// TIA Portal V17 export
// export: Created 2025-07-01T09:59:02.8263122Z, ExportSetting WithDefaults, DisplayName Totally Integrated Automation Portal, DisplayVersion V17 Update 8, DisplayName TIA Portal Openness, DisplayVersion V17 Update 8, DisplayName TIA Portal Version Control Interface, DisplayVersion V17, DisplayName SINAMICS Startdrive Advanced, DisplayVersion V17 SP2, DisplayName SINAMICS Startdrive G110M, G120, G120C, G120D, G120P, G115D, DisplayVersion V17 SP2, DisplayName SINAMICS Startdrive G130, G150, S120, S150, SINAMICS MV, S210, DisplayVersion V17 SP2, DisplayName STEP 7 Professional, DisplayVersion V17 Update 8, DisplayName SINUMERIK ONE STEP 7 Toolbox, DisplayVersion V17 Update 12, DisplayName SINUMERIK ONE PLC Basic Program Plus, DisplayVersion V17 Update 12, DisplayName SINUMERIK 840D sl STEP 7 Toolbox, DisplayVersion V17 Update 12, DisplayName STEP 7 Safety, DisplayVersion V17 Update 6, DisplayName WinCC Advanced, DisplayVersion V17 Update 8
FUNCTION "FC16012_METHOD_CALLS_U1_STA3_COAXIAL" : Void   // FC16012, LAD
{ S7_Optimized_Access := 'FALSE' }
VERSION : 0.1
// PC status values:
// 0-> Idle
// 1-> LaserCalibrating
// 2-> NozzleCalibrating
// 3-> JetCalibrating
// 4-> CladdingCalibrating
// 5-> NozzleAnalysis
// 6-> JetAnalysis
// 7-> CladdingAnalysis
// -1-> Error
// stored: AutoNumber false, IsIECCheckEnabled false, SetENOAutomatically false, UDAEnableTagReadback false
   VAR_TEMP
      AUX_WSTRING_PART_ID_STA3 : WString;
      AUX_WCHARS : Array[0..63] of WChar;
      index : Int;
      ALARM_AUX : Bool;
      STATUS_BLKMOV : Int;   // STATUS BLKMOV
      ZERO : Int;
      retval : Word;
   END_VAR
   VAR CONSTANT
      VERSIONS_MAJOR : UInt := 2;
      VERSIONS_MINOR : UInt := 0;
      FC_NUMBER : DInt := 16012;
   END_VAR
   VAR_TEMP   // added for the SCL form of the ladder/FBD networks
      _w1 : Bool;
      _w2 : Bool;
   END_VAR
BEGIN

REGION Network 1 (SCL): TRANSFORM TO WCHARS
   FOR #index := 0 TO 63 DO
       #AUX_WCHARS[#index] := CHAR_TO_WCHAR("DB8000_PART_STATUS".UNIT_1.STATION_3.PART_A.PART_ID[#index]);
   END_FOR;
END_REGION

REGION Network 2: TRANSFORM TO WSTRING
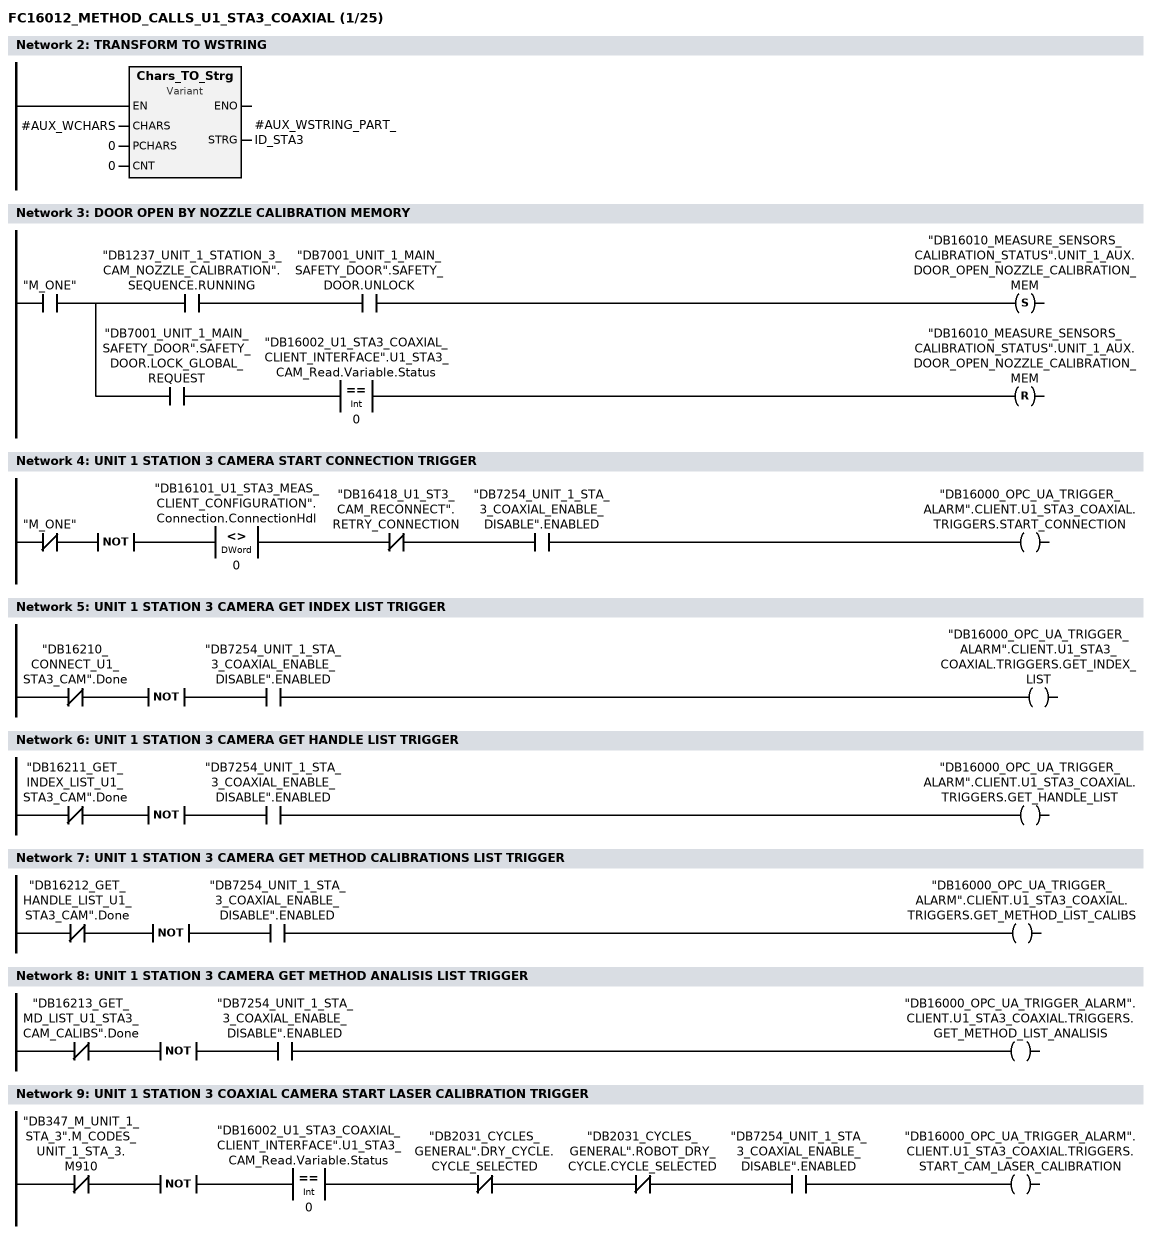
   RUNG wire#powerrail
      { S7_Templates := "[ptr_type := Variant, str_type := WString]" } Chars_TO_Strg(Chars := #AUX_WCHARS, pChars := 0, Cnt := 0, Strg => #AUX_WSTRING_PART_ID_STA3)
   END_RUNG
   // the same network as SCL:
   Chars_TO_Strg(Chars := #AUX_WCHARS, pChars := 0, Cnt := 0, Strg => #AUX_WSTRING_PART_ID_STA3);
END_REGION

REGION Network 3: DOOR OPEN BY NOZZLE CALIBRATION MEMORY
   RUNG wire#powerrail
      Contact( "M_ONE" )
      wire#w1
      Contact( "DB1237_UNIT_1_STATION_3_CAM_NOZZLE_CALIBRATION".SEQUENCE.RUNNING )
      Contact( "DB7001_UNIT_1_MAIN_SAFETY_DOOR".SAFETY_DOOR.UNLOCK )
      S_Coil( "DB16010_MEASURE_SENSORS_CALIBRATION_STATUS".UNIT_1_AUX.DOOR_OPEN_NOZZLE_CALIBRATION_MEM )
   END_RUNG
   RUNG wire#w1
      Contact( "DB7001_UNIT_1_MAIN_SAFETY_DOOR".SAFETY_DOOR.LOCK_GLOBAL_REQUEST )
      { S7_Templates := "SrcType := Int" } EQ_Contact(in1 := "DB16002_U1_STA3_COAXIAL_CLIENT_INTERFACE".U1_STA3_CAM_Read.Variable.Status, in2 := 0)
      R_Coil( "DB16010_MEASURE_SENSORS_CALIBRATION_STATUS".UNIT_1_AUX.DOOR_OPEN_NOZZLE_CALIBRATION_MEM )
   END_RUNG
   // the same network as SCL:
   IF "M_ONE" AND "DB1237_UNIT_1_STATION_3_CAM_NOZZLE_CALIBRATION".SEQUENCE.RUNNING AND "DB7001_UNIT_1_MAIN_SAFETY_DOOR".SAFETY_DOOR.UNLOCK THEN
       "DB16010_MEASURE_SENSORS_CALIBRATION_STATUS".UNIT_1_AUX.DOOR_OPEN_NOZZLE_CALIBRATION_MEM := TRUE;
   END_IF;
   IF "M_ONE" AND "DB7001_UNIT_1_MAIN_SAFETY_DOOR".SAFETY_DOOR.LOCK_GLOBAL_REQUEST AND ("DB16002_U1_STA3_COAXIAL_CLIENT_INTERFACE".U1_STA3_CAM_Read.Variable.Status = 0) THEN
       "DB16010_MEASURE_SENSORS_CALIBRATION_STATUS".UNIT_1_AUX.DOOR_OPEN_NOZZLE_CALIBRATION_MEM := FALSE;
   END_IF;
END_REGION

REGION Network 4: UNIT 1 STATION 3 CAMERA START CONNECTION TRIGGER
   RUNG wire#powerrail
      I_Contact( "M_ONE" )
      Not()
      { S7_Templates := "SrcType := DWord" } NE_Contact(in1 := "DB16101_U1_STA3_MEAS_CLIENT_CONFIGURATION".Connection.ConnectionHdl, in2 := 0)
      I_Contact( "DB16418_U1_ST3_CAM_RECONNECT".RETRY_CONNECTION )
      Contact( "DB7254_UNIT_1_STA_3_COAXIAL_ENABLE_DISABLE".ENABLED )
      Coil( "DB16000_OPC_UA_TRIGGER_ALARM".CLIENT.U1_STA3_COAXIAL.TRIGGERS.START_CONNECTION )
   END_RUNG
   // the same network as SCL:
   "DB16000_OPC_UA_TRIGGER_ALARM".CLIENT.U1_STA3_COAXIAL.TRIGGERS.START_CONNECTION := NOT (NOT "M_ONE") AND ("DB16101_U1_STA3_MEAS_CLIENT_CONFIGURATION".Connection.ConnectionHdl <> 0) AND NOT "DB16418_U1_ST3_CAM_RECONNECT".RETRY_CONNECTION AND "DB7254_UNIT_1_STA_3_COAXIAL_ENABLE_DISABLE".ENABLED;
END_REGION

REGION Network 5: UNIT 1 STATION 3 CAMERA GET INDEX LIST TRIGGER
   RUNG wire#powerrail
      I_Contact( "DB16210_CONNECT_U1_STA3_CAM".Done )
      Not()
      Contact( "DB7254_UNIT_1_STA_3_COAXIAL_ENABLE_DISABLE".ENABLED )
      Coil( "DB16000_OPC_UA_TRIGGER_ALARM".CLIENT.U1_STA3_COAXIAL.TRIGGERS.GET_INDEX_LIST )
   END_RUNG
   // the same network as SCL:
   "DB16000_OPC_UA_TRIGGER_ALARM".CLIENT.U1_STA3_COAXIAL.TRIGGERS.GET_INDEX_LIST := NOT (NOT "DB16210_CONNECT_U1_STA3_CAM".Done) AND "DB7254_UNIT_1_STA_3_COAXIAL_ENABLE_DISABLE".ENABLED;
END_REGION

REGION Network 6: UNIT 1 STATION 3 CAMERA GET HANDLE LIST TRIGGER
   RUNG wire#powerrail
      I_Contact( "DB16211_GET_INDEX_LIST_U1_STA3_CAM".Done )
      Not()
      Contact( "DB7254_UNIT_1_STA_3_COAXIAL_ENABLE_DISABLE".ENABLED )
      Coil( "DB16000_OPC_UA_TRIGGER_ALARM".CLIENT.U1_STA3_COAXIAL.TRIGGERS.GET_HANDLE_LIST )
   END_RUNG
   // the same network as SCL:
   "DB16000_OPC_UA_TRIGGER_ALARM".CLIENT.U1_STA3_COAXIAL.TRIGGERS.GET_HANDLE_LIST := NOT (NOT "DB16211_GET_INDEX_LIST_U1_STA3_CAM".Done) AND "DB7254_UNIT_1_STA_3_COAXIAL_ENABLE_DISABLE".ENABLED;
END_REGION

REGION Network 7: UNIT 1 STATION 3 CAMERA GET METHOD CALIBRATIONS LIST TRIGGER
   RUNG wire#powerrail
      I_Contact( "DB16212_GET_HANDLE_LIST_U1_STA3_CAM".Done )
      Not()
      Contact( "DB7254_UNIT_1_STA_3_COAXIAL_ENABLE_DISABLE".ENABLED )
      Coil( "DB16000_OPC_UA_TRIGGER_ALARM".CLIENT.U1_STA3_COAXIAL.TRIGGERS.GET_METHOD_LIST_CALIBS )
   END_RUNG
   // the same network as SCL:
   "DB16000_OPC_UA_TRIGGER_ALARM".CLIENT.U1_STA3_COAXIAL.TRIGGERS.GET_METHOD_LIST_CALIBS := NOT (NOT "DB16212_GET_HANDLE_LIST_U1_STA3_CAM".Done) AND "DB7254_UNIT_1_STA_3_COAXIAL_ENABLE_DISABLE".ENABLED;
END_REGION

REGION Network 8: UNIT 1 STATION 3 CAMERA GET METHOD ANALISIS LIST TRIGGER
   RUNG wire#powerrail
      I_Contact( "DB16213_GET_MD_LIST_U1_STA3_CAM_CALIBS".Done )
      Not()
      Contact( "DB7254_UNIT_1_STA_3_COAXIAL_ENABLE_DISABLE".ENABLED )
      Coil( "DB16000_OPC_UA_TRIGGER_ALARM".CLIENT.U1_STA3_COAXIAL.TRIGGERS.GET_METHOD_LIST_ANALISIS )
   END_RUNG
   // the same network as SCL:
   "DB16000_OPC_UA_TRIGGER_ALARM".CLIENT.U1_STA3_COAXIAL.TRIGGERS.GET_METHOD_LIST_ANALISIS := NOT (NOT "DB16213_GET_MD_LIST_U1_STA3_CAM_CALIBS".Done) AND "DB7254_UNIT_1_STA_3_COAXIAL_ENABLE_DISABLE".ENABLED;
END_REGION

REGION Network 9: UNIT 1 STATION 3 COAXIAL CAMERA START LASER CALIBRATION TRIGGER
   RUNG wire#powerrail
      I_Contact( "DB347_M_UNIT_1_STA_3".M_CODES_UNIT_1_STA_3.M910 )
      Not()
      { S7_Templates := "SrcType := Int" } EQ_Contact(in1 := "DB16002_U1_STA3_COAXIAL_CLIENT_INTERFACE".U1_STA3_CAM_Read.Variable.Status, in2 := 0)
      I_Contact( "DB2031_CYCLES_GENERAL".DRY_CYCLE.CYCLE_SELECTED )
      I_Contact( "DB2031_CYCLES_GENERAL".ROBOT_DRY_CYCLE.CYCLE_SELECTED )
      Contact( "DB7254_UNIT_1_STA_3_COAXIAL_ENABLE_DISABLE".ENABLED )
      Coil( "DB16000_OPC_UA_TRIGGER_ALARM".CLIENT.U1_STA3_COAXIAL.TRIGGERS.START_CAM_LASER_CALIBRATION )
   END_RUNG
   // the same network as SCL:
   "DB16000_OPC_UA_TRIGGER_ALARM".CLIENT.U1_STA3_COAXIAL.TRIGGERS.START_CAM_LASER_CALIBRATION := NOT (NOT "DB347_M_UNIT_1_STA_3".M_CODES_UNIT_1_STA_3.M910) AND ("DB16002_U1_STA3_COAXIAL_CLIENT_INTERFACE".U1_STA3_CAM_Read.Variable.Status = 0) AND NOT "DB2031_CYCLES_GENERAL".DRY_CYCLE.CYCLE_SELECTED AND NOT "DB2031_CYCLES_GENERAL".ROBOT_DRY_CYCLE.CYCLE_SELECTED AND "DB7254_UNIT_1_STA_3_COAXIAL_ENABLE_DISABLE".ENABLED;
END_REGION

REGION Network 10: UNIT 1 STATION 3 COAXIAL CAMERA START NOZZLE CALIBRATION TRIGGER
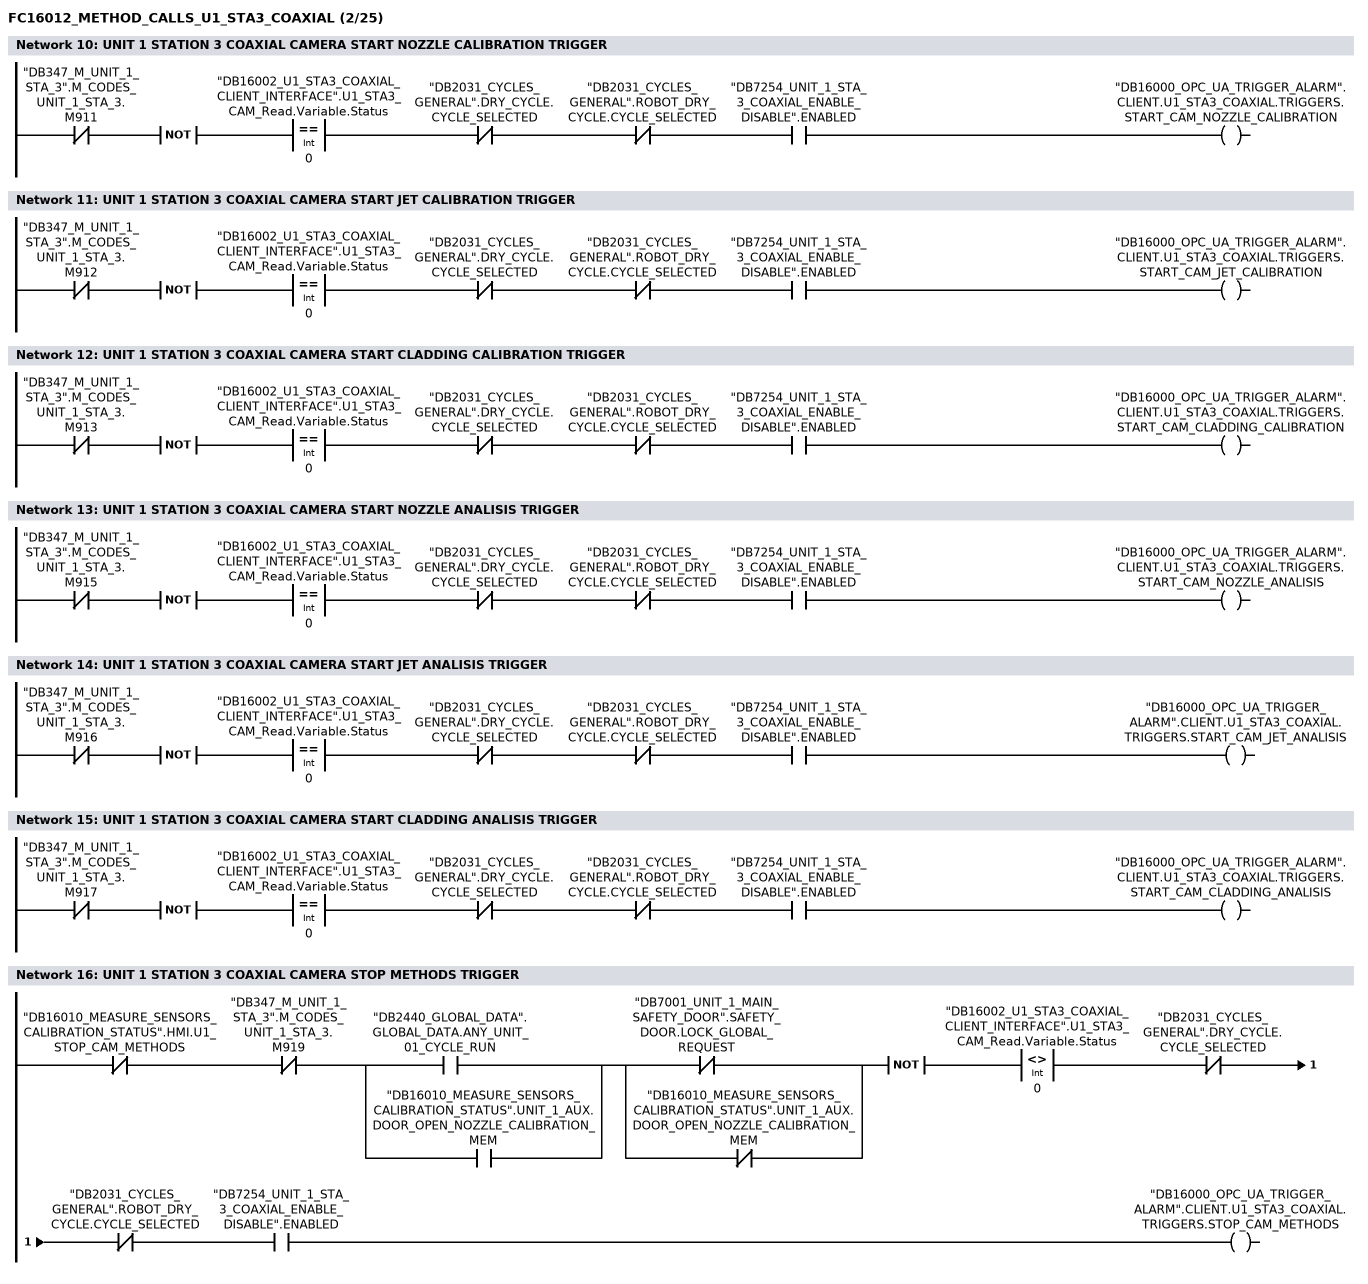
   RUNG wire#powerrail
      I_Contact( "DB347_M_UNIT_1_STA_3".M_CODES_UNIT_1_STA_3.M911 )
      Not()
      { S7_Templates := "SrcType := Int" } EQ_Contact(in1 := "DB16002_U1_STA3_COAXIAL_CLIENT_INTERFACE".U1_STA3_CAM_Read.Variable.Status, in2 := 0)
      I_Contact( "DB2031_CYCLES_GENERAL".DRY_CYCLE.CYCLE_SELECTED )
      I_Contact( "DB2031_CYCLES_GENERAL".ROBOT_DRY_CYCLE.CYCLE_SELECTED )
      Contact( "DB7254_UNIT_1_STA_3_COAXIAL_ENABLE_DISABLE".ENABLED )
      Coil( "DB16000_OPC_UA_TRIGGER_ALARM".CLIENT.U1_STA3_COAXIAL.TRIGGERS.START_CAM_NOZZLE_CALIBRATION )
   END_RUNG
   // the same network as SCL:
   "DB16000_OPC_UA_TRIGGER_ALARM".CLIENT.U1_STA3_COAXIAL.TRIGGERS.START_CAM_NOZZLE_CALIBRATION := NOT (NOT "DB347_M_UNIT_1_STA_3".M_CODES_UNIT_1_STA_3.M911) AND ("DB16002_U1_STA3_COAXIAL_CLIENT_INTERFACE".U1_STA3_CAM_Read.Variable.Status = 0) AND NOT "DB2031_CYCLES_GENERAL".DRY_CYCLE.CYCLE_SELECTED AND NOT "DB2031_CYCLES_GENERAL".ROBOT_DRY_CYCLE.CYCLE_SELECTED AND "DB7254_UNIT_1_STA_3_COAXIAL_ENABLE_DISABLE".ENABLED;
END_REGION

REGION Network 11: UNIT 1 STATION 3 COAXIAL CAMERA START JET CALIBRATION TRIGGER
   RUNG wire#powerrail
      I_Contact( "DB347_M_UNIT_1_STA_3".M_CODES_UNIT_1_STA_3.M912 )
      Not()
      { S7_Templates := "SrcType := Int" } EQ_Contact(in1 := "DB16002_U1_STA3_COAXIAL_CLIENT_INTERFACE".U1_STA3_CAM_Read.Variable.Status, in2 := 0)
      I_Contact( "DB2031_CYCLES_GENERAL".DRY_CYCLE.CYCLE_SELECTED )
      I_Contact( "DB2031_CYCLES_GENERAL".ROBOT_DRY_CYCLE.CYCLE_SELECTED )
      Contact( "DB7254_UNIT_1_STA_3_COAXIAL_ENABLE_DISABLE".ENABLED )
      Coil( "DB16000_OPC_UA_TRIGGER_ALARM".CLIENT.U1_STA3_COAXIAL.TRIGGERS.START_CAM_JET_CALIBRATION )
   END_RUNG
   // the same network as SCL:
   "DB16000_OPC_UA_TRIGGER_ALARM".CLIENT.U1_STA3_COAXIAL.TRIGGERS.START_CAM_JET_CALIBRATION := NOT (NOT "DB347_M_UNIT_1_STA_3".M_CODES_UNIT_1_STA_3.M912) AND ("DB16002_U1_STA3_COAXIAL_CLIENT_INTERFACE".U1_STA3_CAM_Read.Variable.Status = 0) AND NOT "DB2031_CYCLES_GENERAL".DRY_CYCLE.CYCLE_SELECTED AND NOT "DB2031_CYCLES_GENERAL".ROBOT_DRY_CYCLE.CYCLE_SELECTED AND "DB7254_UNIT_1_STA_3_COAXIAL_ENABLE_DISABLE".ENABLED;
END_REGION

REGION Network 12: UNIT 1 STATION 3 COAXIAL CAMERA START CLADDING CALIBRATION TRIGGER
   RUNG wire#powerrail
      I_Contact( "DB347_M_UNIT_1_STA_3".M_CODES_UNIT_1_STA_3.M913 )
      Not()
      { S7_Templates := "SrcType := Int" } EQ_Contact(in1 := "DB16002_U1_STA3_COAXIAL_CLIENT_INTERFACE".U1_STA3_CAM_Read.Variable.Status, in2 := 0)
      I_Contact( "DB2031_CYCLES_GENERAL".DRY_CYCLE.CYCLE_SELECTED )
      I_Contact( "DB2031_CYCLES_GENERAL".ROBOT_DRY_CYCLE.CYCLE_SELECTED )
      Contact( "DB7254_UNIT_1_STA_3_COAXIAL_ENABLE_DISABLE".ENABLED )
      Coil( "DB16000_OPC_UA_TRIGGER_ALARM".CLIENT.U1_STA3_COAXIAL.TRIGGERS.START_CAM_CLADDING_CALIBRATION )
   END_RUNG
   // the same network as SCL:
   "DB16000_OPC_UA_TRIGGER_ALARM".CLIENT.U1_STA3_COAXIAL.TRIGGERS.START_CAM_CLADDING_CALIBRATION := NOT (NOT "DB347_M_UNIT_1_STA_3".M_CODES_UNIT_1_STA_3.M913) AND ("DB16002_U1_STA3_COAXIAL_CLIENT_INTERFACE".U1_STA3_CAM_Read.Variable.Status = 0) AND NOT "DB2031_CYCLES_GENERAL".DRY_CYCLE.CYCLE_SELECTED AND NOT "DB2031_CYCLES_GENERAL".ROBOT_DRY_CYCLE.CYCLE_SELECTED AND "DB7254_UNIT_1_STA_3_COAXIAL_ENABLE_DISABLE".ENABLED;
END_REGION

REGION Network 13: UNIT 1 STATION 3 COAXIAL CAMERA START NOZZLE ANALISIS TRIGGER
   RUNG wire#powerrail
      I_Contact( "DB347_M_UNIT_1_STA_3".M_CODES_UNIT_1_STA_3.M915 )
      Not()
      { S7_Templates := "SrcType := Int" } EQ_Contact(in1 := "DB16002_U1_STA3_COAXIAL_CLIENT_INTERFACE".U1_STA3_CAM_Read.Variable.Status, in2 := 0)
      I_Contact( "DB2031_CYCLES_GENERAL".DRY_CYCLE.CYCLE_SELECTED )
      I_Contact( "DB2031_CYCLES_GENERAL".ROBOT_DRY_CYCLE.CYCLE_SELECTED )
      Contact( "DB7254_UNIT_1_STA_3_COAXIAL_ENABLE_DISABLE".ENABLED )
      Coil( "DB16000_OPC_UA_TRIGGER_ALARM".CLIENT.U1_STA3_COAXIAL.TRIGGERS.START_CAM_NOZZLE_ANALISIS )
   END_RUNG
   // the same network as SCL:
   "DB16000_OPC_UA_TRIGGER_ALARM".CLIENT.U1_STA3_COAXIAL.TRIGGERS.START_CAM_NOZZLE_ANALISIS := NOT (NOT "DB347_M_UNIT_1_STA_3".M_CODES_UNIT_1_STA_3.M915) AND ("DB16002_U1_STA3_COAXIAL_CLIENT_INTERFACE".U1_STA3_CAM_Read.Variable.Status = 0) AND NOT "DB2031_CYCLES_GENERAL".DRY_CYCLE.CYCLE_SELECTED AND NOT "DB2031_CYCLES_GENERAL".ROBOT_DRY_CYCLE.CYCLE_SELECTED AND "DB7254_UNIT_1_STA_3_COAXIAL_ENABLE_DISABLE".ENABLED;
END_REGION

REGION Network 14: UNIT 1 STATION 3 COAXIAL CAMERA START JET ANALISIS TRIGGER
   RUNG wire#powerrail
      I_Contact( "DB347_M_UNIT_1_STA_3".M_CODES_UNIT_1_STA_3.M916 )
      Not()
      { S7_Templates := "SrcType := Int" } EQ_Contact(in1 := "DB16002_U1_STA3_COAXIAL_CLIENT_INTERFACE".U1_STA3_CAM_Read.Variable.Status, in2 := 0)
      I_Contact( "DB2031_CYCLES_GENERAL".DRY_CYCLE.CYCLE_SELECTED )
      I_Contact( "DB2031_CYCLES_GENERAL".ROBOT_DRY_CYCLE.CYCLE_SELECTED )
      Contact( "DB7254_UNIT_1_STA_3_COAXIAL_ENABLE_DISABLE".ENABLED )
      Coil( "DB16000_OPC_UA_TRIGGER_ALARM".CLIENT.U1_STA3_COAXIAL.TRIGGERS.START_CAM_JET_ANALISIS )
   END_RUNG
   // the same network as SCL:
   "DB16000_OPC_UA_TRIGGER_ALARM".CLIENT.U1_STA3_COAXIAL.TRIGGERS.START_CAM_JET_ANALISIS := NOT (NOT "DB347_M_UNIT_1_STA_3".M_CODES_UNIT_1_STA_3.M916) AND ("DB16002_U1_STA3_COAXIAL_CLIENT_INTERFACE".U1_STA3_CAM_Read.Variable.Status = 0) AND NOT "DB2031_CYCLES_GENERAL".DRY_CYCLE.CYCLE_SELECTED AND NOT "DB2031_CYCLES_GENERAL".ROBOT_DRY_CYCLE.CYCLE_SELECTED AND "DB7254_UNIT_1_STA_3_COAXIAL_ENABLE_DISABLE".ENABLED;
END_REGION

REGION Network 15: UNIT 1 STATION 3 COAXIAL CAMERA START CLADDING ANALISIS TRIGGER
   RUNG wire#powerrail
      I_Contact( "DB347_M_UNIT_1_STA_3".M_CODES_UNIT_1_STA_3.M917 )
      Not()
      { S7_Templates := "SrcType := Int" } EQ_Contact(in1 := "DB16002_U1_STA3_COAXIAL_CLIENT_INTERFACE".U1_STA3_CAM_Read.Variable.Status, in2 := 0)
      I_Contact( "DB2031_CYCLES_GENERAL".DRY_CYCLE.CYCLE_SELECTED )
      I_Contact( "DB2031_CYCLES_GENERAL".ROBOT_DRY_CYCLE.CYCLE_SELECTED )
      Contact( "DB7254_UNIT_1_STA_3_COAXIAL_ENABLE_DISABLE".ENABLED )
      Coil( "DB16000_OPC_UA_TRIGGER_ALARM".CLIENT.U1_STA3_COAXIAL.TRIGGERS.START_CAM_CLADDING_ANALISIS )
   END_RUNG
   // the same network as SCL:
   "DB16000_OPC_UA_TRIGGER_ALARM".CLIENT.U1_STA3_COAXIAL.TRIGGERS.START_CAM_CLADDING_ANALISIS := NOT (NOT "DB347_M_UNIT_1_STA_3".M_CODES_UNIT_1_STA_3.M917) AND ("DB16002_U1_STA3_COAXIAL_CLIENT_INTERFACE".U1_STA3_CAM_Read.Variable.Status = 0) AND NOT "DB2031_CYCLES_GENERAL".DRY_CYCLE.CYCLE_SELECTED AND NOT "DB2031_CYCLES_GENERAL".ROBOT_DRY_CYCLE.CYCLE_SELECTED AND "DB7254_UNIT_1_STA_3_COAXIAL_ENABLE_DISABLE".ENABLED;
END_REGION

REGION Network 16: UNIT 1 STATION 3 COAXIAL CAMERA STOP METHODS TRIGGER
   RUNG wire#powerrail
      I_Contact( "DB16010_MEASURE_SENSORS_CALIBRATION_STATUS".HMI.U1_STOP_CAM_METHODS )
      I_Contact( "DB347_M_UNIT_1_STA_3".M_CODES_UNIT_1_STA_3.M919 )
      wire#w1
      Contact( "DB2440_GLOBAL_DATA".GLOBAL_DATA.ANY_UNIT_01_CYCLE_RUN )
      wire#w2
      I_Contact( "DB7001_UNIT_1_MAIN_SAFETY_DOOR".SAFETY_DOOR.LOCK_GLOBAL_REQUEST )
      wire#w3
      Not()
      { S7_Templates := "SrcType := Int" } NE_Contact(in1 := "DB16002_U1_STA3_COAXIAL_CLIENT_INTERFACE".U1_STA3_CAM_Read.Variable.Status, in2 := 0)
      I_Contact( "DB2031_CYCLES_GENERAL".DRY_CYCLE.CYCLE_SELECTED )
      I_Contact( "DB2031_CYCLES_GENERAL".ROBOT_DRY_CYCLE.CYCLE_SELECTED )
      Contact( "DB7254_UNIT_1_STA_3_COAXIAL_ENABLE_DISABLE".ENABLED )
      Coil( "DB16000_OPC_UA_TRIGGER_ALARM".CLIENT.U1_STA3_COAXIAL.TRIGGERS.STOP_CAM_METHODS )
   END_RUNG
   RUNG wire#w1
      Contact( "DB16010_MEASURE_SENSORS_CALIBRATION_STATUS".UNIT_1_AUX.DOOR_OPEN_NOZZLE_CALIBRATION_MEM )
   END_RUNG wire#w2
   RUNG wire#w2
      I_Contact( "DB16010_MEASURE_SENSORS_CALIBRATION_STATUS".UNIT_1_AUX.DOOR_OPEN_NOZZLE_CALIBRATION_MEM )
   END_RUNG wire#w3
   // the same network as SCL:
   "DB16000_OPC_UA_TRIGGER_ALARM".CLIENT.U1_STA3_COAXIAL.TRIGGERS.STOP_CAM_METHODS := NOT (NOT "DB16010_MEASURE_SENSORS_CALIBRATION_STATUS".HMI.U1_STOP_CAM_METHODS AND NOT "DB347_M_UNIT_1_STA_3".M_CODES_UNIT_1_STA_3.M919 AND ("DB2440_GLOBAL_DATA".GLOBAL_DATA.ANY_UNIT_01_CYCLE_RUN OR "DB16010_MEASURE_SENSORS_CALIBRATION_STATUS".UNIT_1_AUX.DOOR_OPEN_NOZZLE_CALIBRATION_MEM) AND (NOT "DB7001_UNIT_1_MAIN_SAFETY_DOOR".SAFETY_DOOR.LOCK_GLOBAL_REQUEST OR NOT "DB16010_MEASURE_SENSORS_CALIBRATION_STATUS".UNIT_1_AUX.DOOR_OPEN_NOZZLE_CALIBRATION_MEM)) AND ("DB16002_U1_STA3_COAXIAL_CLIENT_INTERFACE".U1_STA3_CAM_Read.Variable.Status <> 0) AND NOT "DB2031_CYCLES_GENERAL".DRY_CYCLE.CYCLE_SELECTED AND NOT "DB2031_CYCLES_GENERAL".ROBOT_DRY_CYCLE.CYCLE_SELECTED AND "DB7254_UNIT_1_STA_3_COAXIAL_ENABLE_DISABLE".ENABLED;
END_REGION

REGION Network 17: UNIT 1 STATION 3 COAXIAL CAMERA RESET PC TRIGGER
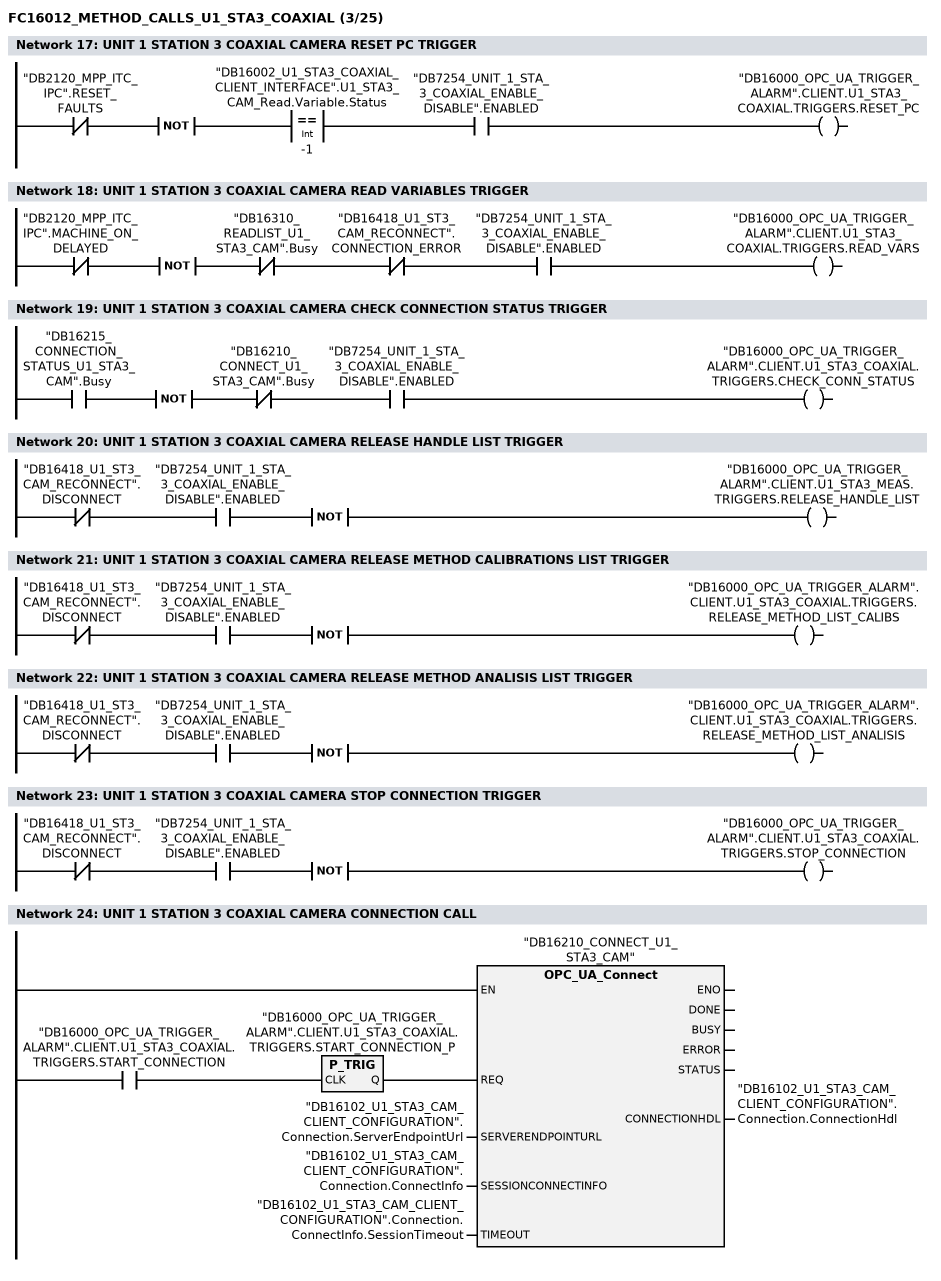
   RUNG wire#powerrail
      I_Contact( "DB2120_MPP_ITC_IPC".RESET_FAULTS )
      Not()
      { S7_Templates := "SrcType := Int" } EQ_Contact(in1 := "DB16002_U1_STA3_COAXIAL_CLIENT_INTERFACE".U1_STA3_CAM_Read.Variable.Status, in2 := -1)
      Contact( "DB7254_UNIT_1_STA_3_COAXIAL_ENABLE_DISABLE".ENABLED )
      Coil( "DB16000_OPC_UA_TRIGGER_ALARM".CLIENT.U1_STA3_COAXIAL.TRIGGERS.RESET_PC )
   END_RUNG
   // the same network as SCL:
   "DB16000_OPC_UA_TRIGGER_ALARM".CLIENT.U1_STA3_COAXIAL.TRIGGERS.RESET_PC := NOT (NOT "DB2120_MPP_ITC_IPC".RESET_FAULTS) AND ("DB16002_U1_STA3_COAXIAL_CLIENT_INTERFACE".U1_STA3_CAM_Read.Variable.Status = (-1)) AND "DB7254_UNIT_1_STA_3_COAXIAL_ENABLE_DISABLE".ENABLED;
END_REGION

REGION Network 18: UNIT 1 STATION 3 COAXIAL CAMERA READ VARIABLES TRIGGER
   RUNG wire#powerrail
      I_Contact( "DB2120_MPP_ITC_IPC".MACHINE_ON_DELAYED )
      Not()
      I_Contact( "DB16310_READLIST_U1_STA3_CAM".Busy )
      I_Contact( "DB16418_U1_ST3_CAM_RECONNECT".CONNECTION_ERROR )
      Contact( "DB7254_UNIT_1_STA_3_COAXIAL_ENABLE_DISABLE".ENABLED )
      Coil( "DB16000_OPC_UA_TRIGGER_ALARM".CLIENT.U1_STA3_COAXIAL.TRIGGERS.READ_VARS )
   END_RUNG
   // the same network as SCL:
   "DB16000_OPC_UA_TRIGGER_ALARM".CLIENT.U1_STA3_COAXIAL.TRIGGERS.READ_VARS := NOT (NOT "DB2120_MPP_ITC_IPC".MACHINE_ON_DELAYED) AND NOT "DB16310_READLIST_U1_STA3_CAM".Busy AND NOT "DB16418_U1_ST3_CAM_RECONNECT".CONNECTION_ERROR AND "DB7254_UNIT_1_STA_3_COAXIAL_ENABLE_DISABLE".ENABLED;
END_REGION

REGION Network 19: UNIT 1 STATION 3 COAXIAL CAMERA CHECK CONNECTION STATUS TRIGGER
   RUNG wire#powerrail
      Contact( "DB16215_CONNECTION_STATUS_U1_STA3_CAM".Busy )
      Not()
      I_Contact( "DB16210_CONNECT_U1_STA3_CAM".Busy )
      Contact( "DB7254_UNIT_1_STA_3_COAXIAL_ENABLE_DISABLE".ENABLED )
      Coil( "DB16000_OPC_UA_TRIGGER_ALARM".CLIENT.U1_STA3_COAXIAL.TRIGGERS.CHECK_CONN_STATUS )
   END_RUNG
   // the same network as SCL:
   "DB16000_OPC_UA_TRIGGER_ALARM".CLIENT.U1_STA3_COAXIAL.TRIGGERS.CHECK_CONN_STATUS := NOT "DB16215_CONNECTION_STATUS_U1_STA3_CAM".Busy AND NOT "DB16210_CONNECT_U1_STA3_CAM".Busy AND "DB7254_UNIT_1_STA_3_COAXIAL_ENABLE_DISABLE".ENABLED;
END_REGION

REGION Network 20: UNIT 1 STATION 3 COAXIAL CAMERA RELEASE HANDLE LIST TRIGGER
   RUNG wire#powerrail
      I_Contact( "DB16418_U1_ST3_CAM_RECONNECT".DISCONNECT )
      Contact( "DB7254_UNIT_1_STA_3_COAXIAL_ENABLE_DISABLE".ENABLED )
      Not()
      Coil( "DB16000_OPC_UA_TRIGGER_ALARM".CLIENT.U1_STA3_MEAS.TRIGGERS.RELEASE_HANDLE_LIST )
   END_RUNG
   // the same network as SCL:
   "DB16000_OPC_UA_TRIGGER_ALARM".CLIENT.U1_STA3_MEAS.TRIGGERS.RELEASE_HANDLE_LIST := NOT (NOT "DB16418_U1_ST3_CAM_RECONNECT".DISCONNECT AND "DB7254_UNIT_1_STA_3_COAXIAL_ENABLE_DISABLE".ENABLED);
END_REGION

REGION Network 21: UNIT 1 STATION 3 COAXIAL CAMERA RELEASE METHOD CALIBRATIONS LIST TRIGGER
   RUNG wire#powerrail
      I_Contact( "DB16418_U1_ST3_CAM_RECONNECT".DISCONNECT )
      Contact( "DB7254_UNIT_1_STA_3_COAXIAL_ENABLE_DISABLE".ENABLED )
      Not()
      Coil( "DB16000_OPC_UA_TRIGGER_ALARM".CLIENT.U1_STA3_COAXIAL.TRIGGERS.RELEASE_METHOD_LIST_CALIBS )
   END_RUNG
   // the same network as SCL:
   "DB16000_OPC_UA_TRIGGER_ALARM".CLIENT.U1_STA3_COAXIAL.TRIGGERS.RELEASE_METHOD_LIST_CALIBS := NOT (NOT "DB16418_U1_ST3_CAM_RECONNECT".DISCONNECT AND "DB7254_UNIT_1_STA_3_COAXIAL_ENABLE_DISABLE".ENABLED);
END_REGION

REGION Network 22: UNIT 1 STATION 3 COAXIAL CAMERA RELEASE METHOD ANALISIS LIST TRIGGER
   RUNG wire#powerrail
      I_Contact( "DB16418_U1_ST3_CAM_RECONNECT".DISCONNECT )
      Contact( "DB7254_UNIT_1_STA_3_COAXIAL_ENABLE_DISABLE".ENABLED )
      Not()
      Coil( "DB16000_OPC_UA_TRIGGER_ALARM".CLIENT.U1_STA3_COAXIAL.TRIGGERS.RELEASE_METHOD_LIST_ANALISIS )
   END_RUNG
   // the same network as SCL:
   "DB16000_OPC_UA_TRIGGER_ALARM".CLIENT.U1_STA3_COAXIAL.TRIGGERS.RELEASE_METHOD_LIST_ANALISIS := NOT (NOT "DB16418_U1_ST3_CAM_RECONNECT".DISCONNECT AND "DB7254_UNIT_1_STA_3_COAXIAL_ENABLE_DISABLE".ENABLED);
END_REGION

REGION Network 23: UNIT 1 STATION 3 COAXIAL CAMERA STOP CONNECTION TRIGGER
   RUNG wire#powerrail
      I_Contact( "DB16418_U1_ST3_CAM_RECONNECT".DISCONNECT )
      Contact( "DB7254_UNIT_1_STA_3_COAXIAL_ENABLE_DISABLE".ENABLED )
      Not()
      Coil( "DB16000_OPC_UA_TRIGGER_ALARM".CLIENT.U1_STA3_COAXIAL.TRIGGERS.STOP_CONNECTION )
   END_RUNG
   // the same network as SCL:
   "DB16000_OPC_UA_TRIGGER_ALARM".CLIENT.U1_STA3_COAXIAL.TRIGGERS.STOP_CONNECTION := NOT (NOT "DB16418_U1_ST3_CAM_RECONNECT".DISCONNECT AND "DB7254_UNIT_1_STA_3_COAXIAL_ENABLE_DISABLE".ENABLED);
END_REGION

REGION Network 24: UNIT 1 STATION 3 COAXIAL CAMERA CONNECTION CALL
   RUNG wire#powerrail
      "DB16210_CONNECT_U1_STA3_CAM".OPC_UA_Connect(REQ := wire#w1, ServerEndpointUrl := "DB16102_U1_STA3_CAM_CLIENT_CONFIGURATION".Connection.ServerEndpointUrl, SessionConnectInfo := "DB16102_U1_STA3_CAM_CLIENT_CONFIGURATION".Connection.ConnectInfo, Timeout := "DB16102_U1_STA3_CAM_CLIENT_CONFIGURATION".Connection.ConnectInfo.SessionTimeout, Done =>, Busy =>, Error =>, Status =>, ConnectionHdl => "DB16102_U1_STA3_CAM_CLIENT_CONFIGURATION".Connection.ConnectionHdl)
   END_RUNG
   RUNG wire#powerrail
      Contact( "DB16000_OPC_UA_TRIGGER_ALARM".CLIENT.U1_STA3_COAXIAL.TRIGGERS.START_CONNECTION )
      P_Trig( "DB16000_OPC_UA_TRIGGER_ALARM".CLIENT.U1_STA3_COAXIAL.TRIGGERS.START_CONNECTION_P )
   END_RUNG wire#w1
   // the same network as SCL:
   #_w1 := "DB16000_OPC_UA_TRIGGER_ALARM".CLIENT.U1_STA3_COAXIAL.TRIGGERS.START_CONNECTION AND NOT "DB16000_OPC_UA_TRIGGER_ALARM".CLIENT.U1_STA3_COAXIAL.TRIGGERS.START_CONNECTION_P;   // rising edge
   "DB16000_OPC_UA_TRIGGER_ALARM".CLIENT.U1_STA3_COAXIAL.TRIGGERS.START_CONNECTION_P := "DB16000_OPC_UA_TRIGGER_ALARM".CLIENT.U1_STA3_COAXIAL.TRIGGERS.START_CONNECTION;
   "DB16210_CONNECT_U1_STA3_CAM"(REQ := #_w1,   // OPC_UA_Connect
                           ServerEndpointUrl := "DB16102_U1_STA3_CAM_CLIENT_CONFIGURATION".Connection.ServerEndpointUrl,
                           SessionConnectInfo := "DB16102_U1_STA3_CAM_CLIENT_CONFIGURATION".Connection.ConnectInfo,
                           Timeout := "DB16102_U1_STA3_CAM_CLIENT_CONFIGURATION".Connection.ConnectInfo.SessionTimeout,
                           ConnectionHdl => "DB16102_U1_STA3_CAM_CLIENT_CONFIGURATION".Connection.ConnectionHdl);
END_REGION

REGION Network 25: UNIT 1 STATION 3 COAXIAL CAMERA GET INDEX LIST CALL
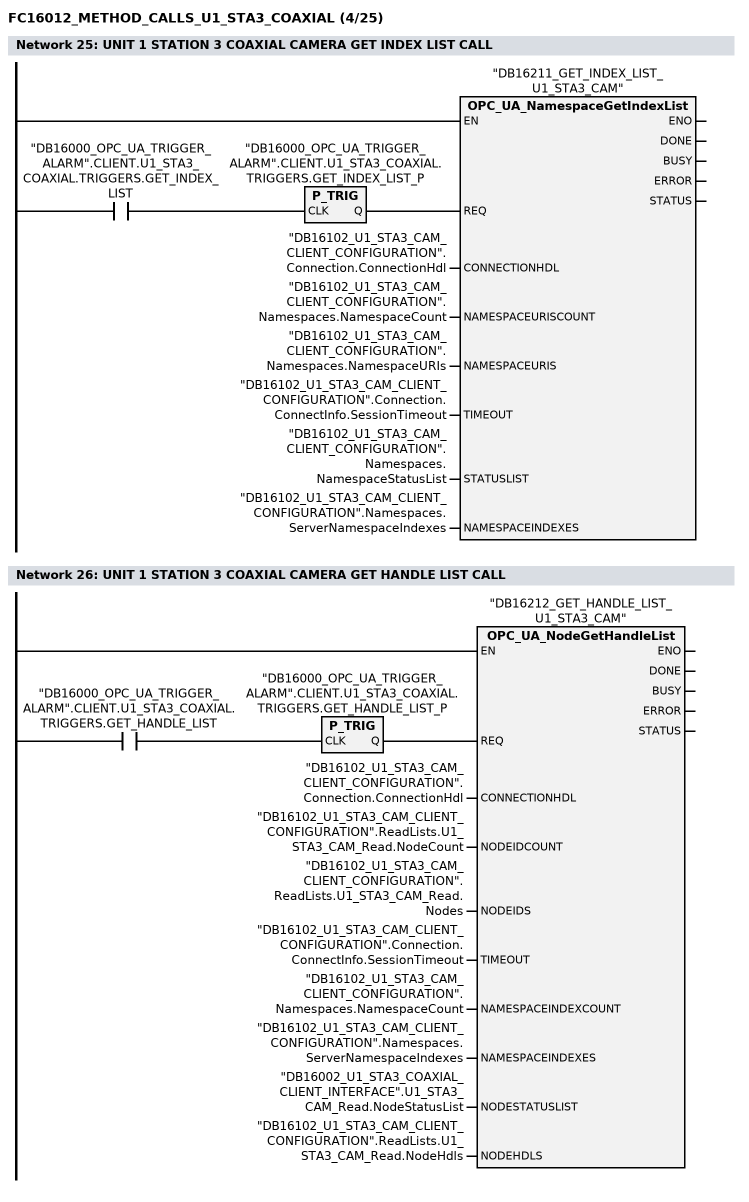
   RUNG wire#powerrail
      "DB16211_GET_INDEX_LIST_U1_STA3_CAM".OPC_UA_NamespaceGetIndexList(REQ := wire#w1, ConnectionHdl := "DB16102_U1_STA3_CAM_CLIENT_CONFIGURATION".Connection.ConnectionHdl, NamespaceUrisCount := "DB16102_U1_STA3_CAM_CLIENT_CONFIGURATION".Namespaces.NamespaceCount, NamespaceUris := "DB16102_U1_STA3_CAM_CLIENT_CONFIGURATION".Namespaces.NamespaceURIs, Timeout := "DB16102_U1_STA3_CAM_CLIENT_CONFIGURATION".Connection.ConnectInfo.SessionTimeout, StatusList := "DB16102_U1_STA3_CAM_CLIENT_CONFIGURATION".Namespaces.NamespaceStatusList, NamespaceIndexes := "DB16102_U1_STA3_CAM_CLIENT_CONFIGURATION".Namespaces.ServerNamespaceIndexes, Done =>, Busy =>, Error =>, Status =>)
   END_RUNG
   RUNG wire#powerrail
      Contact( "DB16000_OPC_UA_TRIGGER_ALARM".CLIENT.U1_STA3_COAXIAL.TRIGGERS.GET_INDEX_LIST )
      P_Trig( "DB16000_OPC_UA_TRIGGER_ALARM".CLIENT.U1_STA3_COAXIAL.TRIGGERS.GET_INDEX_LIST_P )
   END_RUNG wire#w1
   // the same network as SCL:
   #_w1 := "DB16000_OPC_UA_TRIGGER_ALARM".CLIENT.U1_STA3_COAXIAL.TRIGGERS.GET_INDEX_LIST AND NOT "DB16000_OPC_UA_TRIGGER_ALARM".CLIENT.U1_STA3_COAXIAL.TRIGGERS.GET_INDEX_LIST_P;   // rising edge
   "DB16000_OPC_UA_TRIGGER_ALARM".CLIENT.U1_STA3_COAXIAL.TRIGGERS.GET_INDEX_LIST_P := "DB16000_OPC_UA_TRIGGER_ALARM".CLIENT.U1_STA3_COAXIAL.TRIGGERS.GET_INDEX_LIST;
   "DB16211_GET_INDEX_LIST_U1_STA3_CAM"(REQ := #_w1,   // OPC_UA_NamespaceGetIndexList
                           ConnectionHdl := "DB16102_U1_STA3_CAM_CLIENT_CONFIGURATION".Connection.ConnectionHdl,
                           NamespaceUrisCount := "DB16102_U1_STA3_CAM_CLIENT_CONFIGURATION".Namespaces.NamespaceCount,
                           NamespaceUris := "DB16102_U1_STA3_CAM_CLIENT_CONFIGURATION".Namespaces.NamespaceURIs,
                           Timeout := "DB16102_U1_STA3_CAM_CLIENT_CONFIGURATION".Connection.ConnectInfo.SessionTimeout,
                           StatusList := "DB16102_U1_STA3_CAM_CLIENT_CONFIGURATION".Namespaces.NamespaceStatusList,
                           NamespaceIndexes := "DB16102_U1_STA3_CAM_CLIENT_CONFIGURATION".Namespaces.ServerNamespaceIndexes);
END_REGION

REGION Network 26: UNIT 1 STATION 3 COAXIAL CAMERA GET HANDLE LIST CALL
   RUNG wire#powerrail
      "DB16212_GET_HANDLE_LIST_U1_STA3_CAM".OPC_UA_NodeGetHandleList(REQ := wire#w1, ConnectionHdl := "DB16102_U1_STA3_CAM_CLIENT_CONFIGURATION".Connection.ConnectionHdl, NodeIDCount := "DB16102_U1_STA3_CAM_CLIENT_CONFIGURATION".ReadLists.U1_STA3_CAM_Read.NodeCount, NodeIDs := "DB16102_U1_STA3_CAM_CLIENT_CONFIGURATION".ReadLists.U1_STA3_CAM_Read.Nodes, Timeout := "DB16102_U1_STA3_CAM_CLIENT_CONFIGURATION".Connection.ConnectInfo.SessionTimeout, NamespaceIndexCount := "DB16102_U1_STA3_CAM_CLIENT_CONFIGURATION".Namespaces.NamespaceCount, NamespaceIndexes := "DB16102_U1_STA3_CAM_CLIENT_CONFIGURATION".Namespaces.ServerNamespaceIndexes, NodeStatusList := "DB16002_U1_STA3_COAXIAL_CLIENT_INTERFACE".U1_STA3_CAM_Read.NodeStatusList, NodeHdls := "DB16102_U1_STA3_CAM_CLIENT_CONFIGURATION".ReadLists.U1_STA3_CAM_Read.NodeHdls, Done =>, Busy =>, Error =>, Status =>)
   END_RUNG
   RUNG wire#powerrail
      Contact( "DB16000_OPC_UA_TRIGGER_ALARM".CLIENT.U1_STA3_COAXIAL.TRIGGERS.GET_HANDLE_LIST )
      P_Trig( "DB16000_OPC_UA_TRIGGER_ALARM".CLIENT.U1_STA3_COAXIAL.TRIGGERS.GET_HANDLE_LIST_P )
   END_RUNG wire#w1
   // the same network as SCL:
   #_w1 := "DB16000_OPC_UA_TRIGGER_ALARM".CLIENT.U1_STA3_COAXIAL.TRIGGERS.GET_HANDLE_LIST AND NOT "DB16000_OPC_UA_TRIGGER_ALARM".CLIENT.U1_STA3_COAXIAL.TRIGGERS.GET_HANDLE_LIST_P;   // rising edge
   "DB16000_OPC_UA_TRIGGER_ALARM".CLIENT.U1_STA3_COAXIAL.TRIGGERS.GET_HANDLE_LIST_P := "DB16000_OPC_UA_TRIGGER_ALARM".CLIENT.U1_STA3_COAXIAL.TRIGGERS.GET_HANDLE_LIST;
   "DB16212_GET_HANDLE_LIST_U1_STA3_CAM"(REQ := #_w1,   // OPC_UA_NodeGetHandleList
                           ConnectionHdl := "DB16102_U1_STA3_CAM_CLIENT_CONFIGURATION".Connection.ConnectionHdl,
                           NodeIDCount := "DB16102_U1_STA3_CAM_CLIENT_CONFIGURATION".ReadLists.U1_STA3_CAM_Read.NodeCount,
                           NodeIDs := "DB16102_U1_STA3_CAM_CLIENT_CONFIGURATION".ReadLists.U1_STA3_CAM_Read.Nodes,
                           Timeout := "DB16102_U1_STA3_CAM_CLIENT_CONFIGURATION".Connection.ConnectInfo.SessionTimeout,
                           NamespaceIndexCount := "DB16102_U1_STA3_CAM_CLIENT_CONFIGURATION".Namespaces.NamespaceCount,
                           NamespaceIndexes := "DB16102_U1_STA3_CAM_CLIENT_CONFIGURATION".Namespaces.ServerNamespaceIndexes,
                           NodeStatusList := "DB16002_U1_STA3_COAXIAL_CLIENT_INTERFACE".U1_STA3_CAM_Read.NodeStatusList,
                           NodeHdls := "DB16102_U1_STA3_CAM_CLIENT_CONFIGURATION".ReadLists.U1_STA3_CAM_Read.NodeHdls);
END_REGION

REGION Network 27: UNIT 1 STATION 3 COAXIAL CAMERA GET METHOD CALIBRATIONS LIST CALL
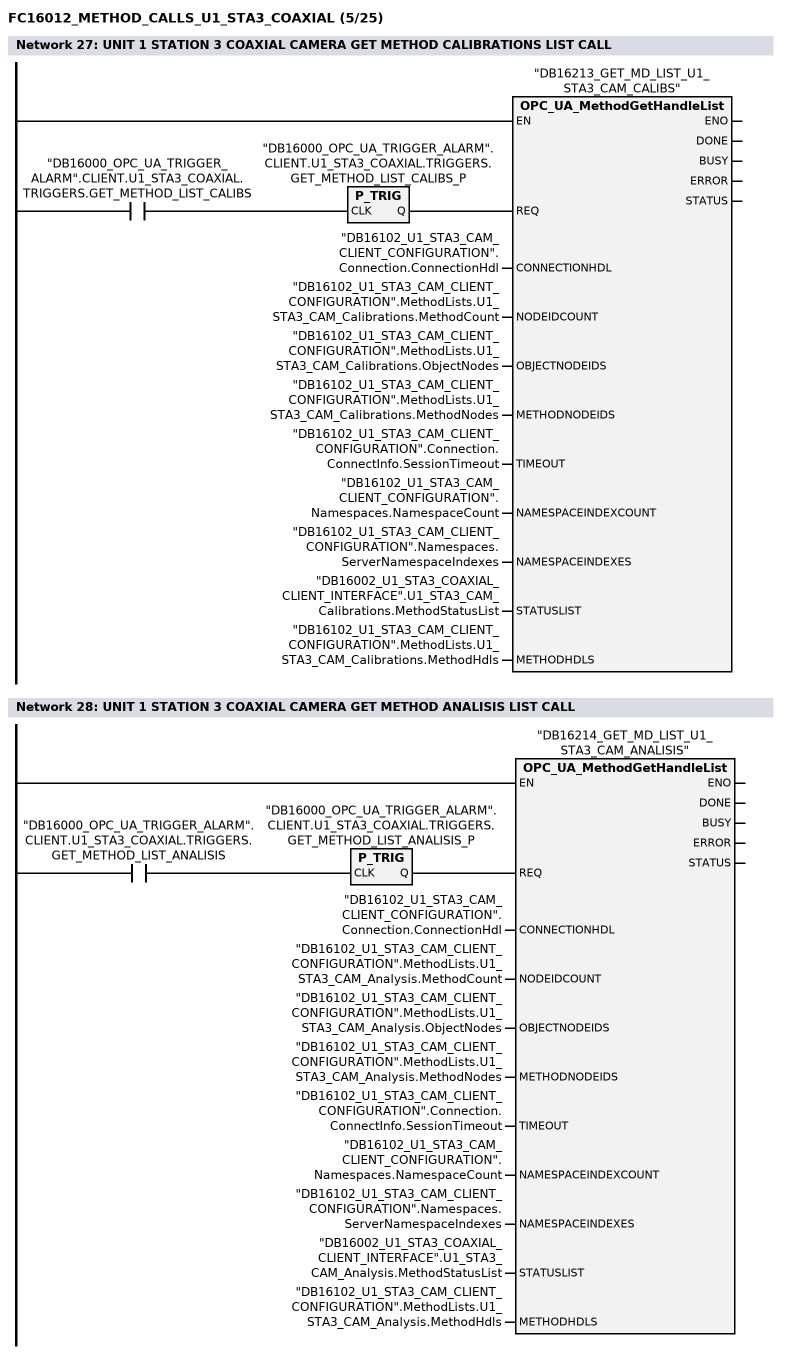
   RUNG wire#powerrail
      "DB16213_GET_MD_LIST_U1_STA3_CAM_CALIBS".OPC_UA_MethodGetHandleList(REQ := wire#w1, ConnectionHdl := "DB16102_U1_STA3_CAM_CLIENT_CONFIGURATION".Connection.ConnectionHdl, NodeIDCount := "DB16102_U1_STA3_CAM_CLIENT_CONFIGURATION".MethodLists.U1_STA3_CAM_Calibrations.MethodCount, ObjectNodeIDs := "DB16102_U1_STA3_CAM_CLIENT_CONFIGURATION".MethodLists.U1_STA3_CAM_Calibrations.ObjectNodes, MethodNodeIDs := "DB16102_U1_STA3_CAM_CLIENT_CONFIGURATION".MethodLists.U1_STA3_CAM_Calibrations.MethodNodes, Timeout := "DB16102_U1_STA3_CAM_CLIENT_CONFIGURATION".Connection.ConnectInfo.SessionTimeout, NamespaceIndexCount := "DB16102_U1_STA3_CAM_CLIENT_CONFIGURATION".Namespaces.NamespaceCount, NamespaceIndexes := "DB16102_U1_STA3_CAM_CLIENT_CONFIGURATION".Namespaces.ServerNamespaceIndexes, StatusList := "DB16002_U1_STA3_COAXIAL_CLIENT_INTERFACE".U1_STA3_CAM_Calibrations.MethodStatusList, MethodHdls := "DB16102_U1_STA3_CAM_CLIENT_CONFIGURATION".MethodLists.U1_STA3_CAM_Calibrations.MethodHdls, Done =>, Busy =>, Error =>, Status =>)
   END_RUNG
   RUNG wire#powerrail
      Contact( "DB16000_OPC_UA_TRIGGER_ALARM".CLIENT.U1_STA3_COAXIAL.TRIGGERS.GET_METHOD_LIST_CALIBS )
      P_Trig( "DB16000_OPC_UA_TRIGGER_ALARM".CLIENT.U1_STA3_COAXIAL.TRIGGERS.GET_METHOD_LIST_CALIBS_P )
   END_RUNG wire#w1
   // the same network as SCL:
   #_w1 := "DB16000_OPC_UA_TRIGGER_ALARM".CLIENT.U1_STA3_COAXIAL.TRIGGERS.GET_METHOD_LIST_CALIBS AND NOT "DB16000_OPC_UA_TRIGGER_ALARM".CLIENT.U1_STA3_COAXIAL.TRIGGERS.GET_METHOD_LIST_CALIBS_P;   // rising edge
   "DB16000_OPC_UA_TRIGGER_ALARM".CLIENT.U1_STA3_COAXIAL.TRIGGERS.GET_METHOD_LIST_CALIBS_P := "DB16000_OPC_UA_TRIGGER_ALARM".CLIENT.U1_STA3_COAXIAL.TRIGGERS.GET_METHOD_LIST_CALIBS;
   "DB16213_GET_MD_LIST_U1_STA3_CAM_CALIBS"(REQ := #_w1,   // OPC_UA_MethodGetHandleList
                           ConnectionHdl := "DB16102_U1_STA3_CAM_CLIENT_CONFIGURATION".Connection.ConnectionHdl,
                           NodeIDCount := "DB16102_U1_STA3_CAM_CLIENT_CONFIGURATION".MethodLists.U1_STA3_CAM_Calibrations.MethodCount,
                           ObjectNodeIDs := "DB16102_U1_STA3_CAM_CLIENT_CONFIGURATION".MethodLists.U1_STA3_CAM_Calibrations.ObjectNodes,
                           MethodNodeIDs := "DB16102_U1_STA3_CAM_CLIENT_CONFIGURATION".MethodLists.U1_STA3_CAM_Calibrations.MethodNodes,
                           Timeout := "DB16102_U1_STA3_CAM_CLIENT_CONFIGURATION".Connection.ConnectInfo.SessionTimeout,
                           NamespaceIndexCount := "DB16102_U1_STA3_CAM_CLIENT_CONFIGURATION".Namespaces.NamespaceCount,
                           NamespaceIndexes := "DB16102_U1_STA3_CAM_CLIENT_CONFIGURATION".Namespaces.ServerNamespaceIndexes,
                           StatusList := "DB16002_U1_STA3_COAXIAL_CLIENT_INTERFACE".U1_STA3_CAM_Calibrations.MethodStatusList,
                           MethodHdls := "DB16102_U1_STA3_CAM_CLIENT_CONFIGURATION".MethodLists.U1_STA3_CAM_Calibrations.MethodHdls);
END_REGION

REGION Network 28: UNIT 1 STATION 3 COAXIAL CAMERA GET METHOD ANALISIS LIST CALL
   RUNG wire#powerrail
      "DB16214_GET_MD_LIST_U1_STA3_CAM_ANALISIS".OPC_UA_MethodGetHandleList(REQ := wire#w1, ConnectionHdl := "DB16102_U1_STA3_CAM_CLIENT_CONFIGURATION".Connection.ConnectionHdl, NodeIDCount := "DB16102_U1_STA3_CAM_CLIENT_CONFIGURATION".MethodLists.U1_STA3_CAM_Analysis.MethodCount, ObjectNodeIDs := "DB16102_U1_STA3_CAM_CLIENT_CONFIGURATION".MethodLists.U1_STA3_CAM_Analysis.ObjectNodes, MethodNodeIDs := "DB16102_U1_STA3_CAM_CLIENT_CONFIGURATION".MethodLists.U1_STA3_CAM_Analysis.MethodNodes, Timeout := "DB16102_U1_STA3_CAM_CLIENT_CONFIGURATION".Connection.ConnectInfo.SessionTimeout, NamespaceIndexCount := "DB16102_U1_STA3_CAM_CLIENT_CONFIGURATION".Namespaces.NamespaceCount, NamespaceIndexes := "DB16102_U1_STA3_CAM_CLIENT_CONFIGURATION".Namespaces.ServerNamespaceIndexes, StatusList := "DB16002_U1_STA3_COAXIAL_CLIENT_INTERFACE".U1_STA3_CAM_Analysis.MethodStatusList, MethodHdls := "DB16102_U1_STA3_CAM_CLIENT_CONFIGURATION".MethodLists.U1_STA3_CAM_Analysis.MethodHdls, Done =>, Busy =>, Error =>, Status =>)
   END_RUNG
   RUNG wire#powerrail
      Contact( "DB16000_OPC_UA_TRIGGER_ALARM".CLIENT.U1_STA3_COAXIAL.TRIGGERS.GET_METHOD_LIST_ANALISIS )
      P_Trig( "DB16000_OPC_UA_TRIGGER_ALARM".CLIENT.U1_STA3_COAXIAL.TRIGGERS.GET_METHOD_LIST_ANALISIS_P )
   END_RUNG wire#w1
   // the same network as SCL:
   #_w1 := "DB16000_OPC_UA_TRIGGER_ALARM".CLIENT.U1_STA3_COAXIAL.TRIGGERS.GET_METHOD_LIST_ANALISIS AND NOT "DB16000_OPC_UA_TRIGGER_ALARM".CLIENT.U1_STA3_COAXIAL.TRIGGERS.GET_METHOD_LIST_ANALISIS_P;   // rising edge
   "DB16000_OPC_UA_TRIGGER_ALARM".CLIENT.U1_STA3_COAXIAL.TRIGGERS.GET_METHOD_LIST_ANALISIS_P := "DB16000_OPC_UA_TRIGGER_ALARM".CLIENT.U1_STA3_COAXIAL.TRIGGERS.GET_METHOD_LIST_ANALISIS;
   "DB16214_GET_MD_LIST_U1_STA3_CAM_ANALISIS"(REQ := #_w1,   // OPC_UA_MethodGetHandleList
                           ConnectionHdl := "DB16102_U1_STA3_CAM_CLIENT_CONFIGURATION".Connection.ConnectionHdl,
                           NodeIDCount := "DB16102_U1_STA3_CAM_CLIENT_CONFIGURATION".MethodLists.U1_STA3_CAM_Analysis.MethodCount,
                           ObjectNodeIDs := "DB16102_U1_STA3_CAM_CLIENT_CONFIGURATION".MethodLists.U1_STA3_CAM_Analysis.ObjectNodes,
                           MethodNodeIDs := "DB16102_U1_STA3_CAM_CLIENT_CONFIGURATION".MethodLists.U1_STA3_CAM_Analysis.MethodNodes,
                           Timeout := "DB16102_U1_STA3_CAM_CLIENT_CONFIGURATION".Connection.ConnectInfo.SessionTimeout,
                           NamespaceIndexCount := "DB16102_U1_STA3_CAM_CLIENT_CONFIGURATION".Namespaces.NamespaceCount,
                           NamespaceIndexes := "DB16102_U1_STA3_CAM_CLIENT_CONFIGURATION".Namespaces.ServerNamespaceIndexes,
                           StatusList := "DB16002_U1_STA3_COAXIAL_CLIENT_INTERFACE".U1_STA3_CAM_Analysis.MethodStatusList,
                           MethodHdls := "DB16102_U1_STA3_CAM_CLIENT_CONFIGURATION".MethodLists.U1_STA3_CAM_Analysis.MethodHdls);
END_REGION

REGION Network 29: UNIT 1 STATION 3 COAXIAL CAMERA START LASER CALIBRATION TRIGGER CALL
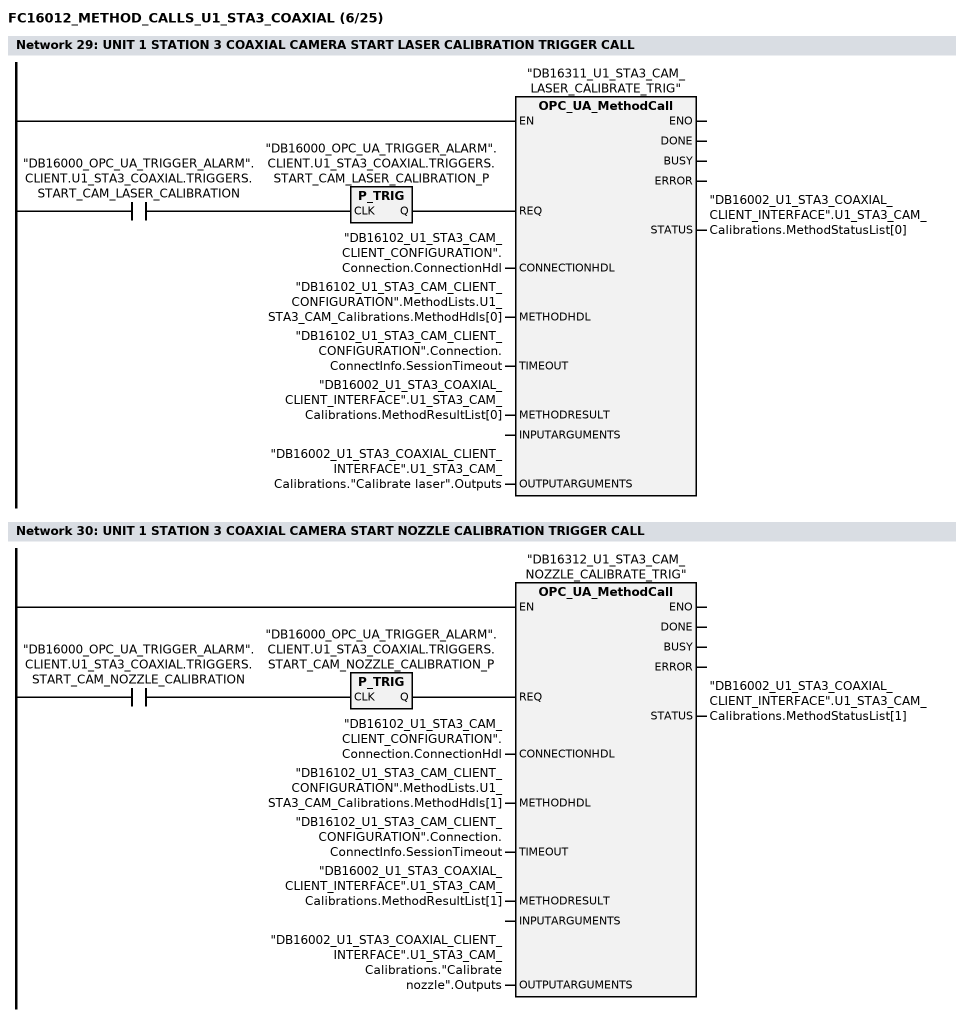
   RUNG wire#powerrail
      "DB16311_U1_STA3_CAM_LASER_CALIBRATE_TRIG".OPC_UA_MethodCall(REQ := wire#w1, ConnectionHdl := "DB16102_U1_STA3_CAM_CLIENT_CONFIGURATION".Connection.ConnectionHdl, MethodHdl := "DB16102_U1_STA3_CAM_CLIENT_CONFIGURATION".MethodLists.U1_STA3_CAM_Calibrations.MethodHdls[0], Timeout := "DB16102_U1_STA3_CAM_CLIENT_CONFIGURATION".Connection.ConnectInfo.SessionTimeout, MethodResult := "DB16002_U1_STA3_COAXIAL_CLIENT_INTERFACE".U1_STA3_CAM_Calibrations.MethodResultList[0], InputArguments :=, OutputArguments := "DB16002_U1_STA3_COAXIAL_CLIENT_INTERFACE".U1_STA3_CAM_Calibrations."Calibrate laser".Outputs, Done =>, Busy =>, Error =>, Status => "DB16002_U1_STA3_COAXIAL_CLIENT_INTERFACE".U1_STA3_CAM_Calibrations.MethodStatusList[0])
   END_RUNG
   RUNG wire#powerrail
      Contact( "DB16000_OPC_UA_TRIGGER_ALARM".CLIENT.U1_STA3_COAXIAL.TRIGGERS.START_CAM_LASER_CALIBRATION )
      P_Trig( "DB16000_OPC_UA_TRIGGER_ALARM".CLIENT.U1_STA3_COAXIAL.TRIGGERS.START_CAM_LASER_CALIBRATION_P )
   END_RUNG wire#w1
   // the same network as SCL:
   #_w1 := "DB16000_OPC_UA_TRIGGER_ALARM".CLIENT.U1_STA3_COAXIAL.TRIGGERS.START_CAM_LASER_CALIBRATION AND NOT "DB16000_OPC_UA_TRIGGER_ALARM".CLIENT.U1_STA3_COAXIAL.TRIGGERS.START_CAM_LASER_CALIBRATION_P;   // rising edge
   "DB16000_OPC_UA_TRIGGER_ALARM".CLIENT.U1_STA3_COAXIAL.TRIGGERS.START_CAM_LASER_CALIBRATION_P := "DB16000_OPC_UA_TRIGGER_ALARM".CLIENT.U1_STA3_COAXIAL.TRIGGERS.START_CAM_LASER_CALIBRATION;
   "DB16311_U1_STA3_CAM_LASER_CALIBRATE_TRIG"(REQ := #_w1,   // OPC_UA_MethodCall
                           ConnectionHdl := "DB16102_U1_STA3_CAM_CLIENT_CONFIGURATION".Connection.ConnectionHdl,
                           MethodHdl := "DB16102_U1_STA3_CAM_CLIENT_CONFIGURATION".MethodLists.U1_STA3_CAM_Calibrations.MethodHdls[0],
                           Timeout := "DB16102_U1_STA3_CAM_CLIENT_CONFIGURATION".Connection.ConnectInfo.SessionTimeout,
                           MethodResult := "DB16002_U1_STA3_COAXIAL_CLIENT_INTERFACE".U1_STA3_CAM_Calibrations.MethodResultList[0],
                           OutputArguments := "DB16002_U1_STA3_COAXIAL_CLIENT_INTERFACE".U1_STA3_CAM_Calibrations."Calibrate laser".Outputs,
                           Status => "DB16002_U1_STA3_COAXIAL_CLIENT_INTERFACE".U1_STA3_CAM_Calibrations.MethodStatusList[0]);
END_REGION

REGION Network 30: UNIT 1 STATION 3 COAXIAL CAMERA START NOZZLE CALIBRATION TRIGGER CALL
   RUNG wire#powerrail
      "DB16312_U1_STA3_CAM_NOZZLE_CALIBRATE_TRIG".OPC_UA_MethodCall(REQ := wire#w1, ConnectionHdl := "DB16102_U1_STA3_CAM_CLIENT_CONFIGURATION".Connection.ConnectionHdl, MethodHdl := "DB16102_U1_STA3_CAM_CLIENT_CONFIGURATION".MethodLists.U1_STA3_CAM_Calibrations.MethodHdls[1], Timeout := "DB16102_U1_STA3_CAM_CLIENT_CONFIGURATION".Connection.ConnectInfo.SessionTimeout, MethodResult := "DB16002_U1_STA3_COAXIAL_CLIENT_INTERFACE".U1_STA3_CAM_Calibrations.MethodResultList[1], InputArguments :=, OutputArguments := "DB16002_U1_STA3_COAXIAL_CLIENT_INTERFACE".U1_STA3_CAM_Calibrations."Calibrate nozzle".Outputs, Done =>, Busy =>, Error =>, Status => "DB16002_U1_STA3_COAXIAL_CLIENT_INTERFACE".U1_STA3_CAM_Calibrations.MethodStatusList[1])
   END_RUNG
   RUNG wire#powerrail
      Contact( "DB16000_OPC_UA_TRIGGER_ALARM".CLIENT.U1_STA3_COAXIAL.TRIGGERS.START_CAM_NOZZLE_CALIBRATION )
      P_Trig( "DB16000_OPC_UA_TRIGGER_ALARM".CLIENT.U1_STA3_COAXIAL.TRIGGERS.START_CAM_NOZZLE_CALIBRATION_P )
   END_RUNG wire#w1
   // the same network as SCL:
   #_w1 := "DB16000_OPC_UA_TRIGGER_ALARM".CLIENT.U1_STA3_COAXIAL.TRIGGERS.START_CAM_NOZZLE_CALIBRATION AND NOT "DB16000_OPC_UA_TRIGGER_ALARM".CLIENT.U1_STA3_COAXIAL.TRIGGERS.START_CAM_NOZZLE_CALIBRATION_P;   // rising edge
   "DB16000_OPC_UA_TRIGGER_ALARM".CLIENT.U1_STA3_COAXIAL.TRIGGERS.START_CAM_NOZZLE_CALIBRATION_P := "DB16000_OPC_UA_TRIGGER_ALARM".CLIENT.U1_STA3_COAXIAL.TRIGGERS.START_CAM_NOZZLE_CALIBRATION;
   "DB16312_U1_STA3_CAM_NOZZLE_CALIBRATE_TRIG"(REQ := #_w1,   // OPC_UA_MethodCall
                           ConnectionHdl := "DB16102_U1_STA3_CAM_CLIENT_CONFIGURATION".Connection.ConnectionHdl,
                           MethodHdl := "DB16102_U1_STA3_CAM_CLIENT_CONFIGURATION".MethodLists.U1_STA3_CAM_Calibrations.MethodHdls[1],
                           Timeout := "DB16102_U1_STA3_CAM_CLIENT_CONFIGURATION".Connection.ConnectInfo.SessionTimeout,
                           MethodResult := "DB16002_U1_STA3_COAXIAL_CLIENT_INTERFACE".U1_STA3_CAM_Calibrations.MethodResultList[1],
                           OutputArguments := "DB16002_U1_STA3_COAXIAL_CLIENT_INTERFACE".U1_STA3_CAM_Calibrations."Calibrate nozzle".Outputs,
                           Status => "DB16002_U1_STA3_COAXIAL_CLIENT_INTERFACE".U1_STA3_CAM_Calibrations.MethodStatusList[1]);
END_REGION

REGION Network 31: UNIT 1 STATION 3 COAXIAL CAMERA START JET CALIBRATION TRIGGER CALL
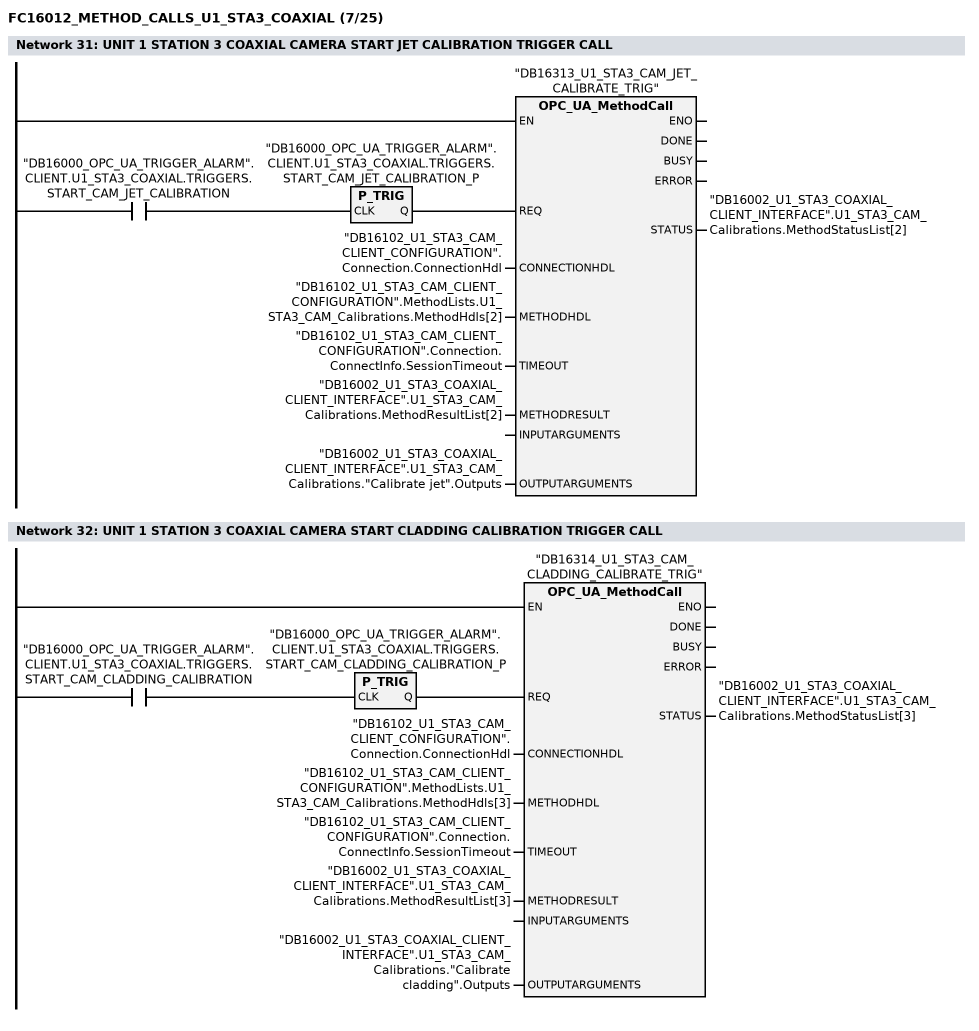
   RUNG wire#powerrail
      "DB16313_U1_STA3_CAM_JET_CALIBRATE_TRIG".OPC_UA_MethodCall(REQ := wire#w1, ConnectionHdl := "DB16102_U1_STA3_CAM_CLIENT_CONFIGURATION".Connection.ConnectionHdl, MethodHdl := "DB16102_U1_STA3_CAM_CLIENT_CONFIGURATION".MethodLists.U1_STA3_CAM_Calibrations.MethodHdls[2], Timeout := "DB16102_U1_STA3_CAM_CLIENT_CONFIGURATION".Connection.ConnectInfo.SessionTimeout, MethodResult := "DB16002_U1_STA3_COAXIAL_CLIENT_INTERFACE".U1_STA3_CAM_Calibrations.MethodResultList[2], InputArguments :=, OutputArguments := "DB16002_U1_STA3_COAXIAL_CLIENT_INTERFACE".U1_STA3_CAM_Calibrations."Calibrate jet".Outputs, Done =>, Busy =>, Error =>, Status => "DB16002_U1_STA3_COAXIAL_CLIENT_INTERFACE".U1_STA3_CAM_Calibrations.MethodStatusList[2])
   END_RUNG
   RUNG wire#powerrail
      Contact( "DB16000_OPC_UA_TRIGGER_ALARM".CLIENT.U1_STA3_COAXIAL.TRIGGERS.START_CAM_JET_CALIBRATION )
      P_Trig( "DB16000_OPC_UA_TRIGGER_ALARM".CLIENT.U1_STA3_COAXIAL.TRIGGERS.START_CAM_JET_CALIBRATION_P )
   END_RUNG wire#w1
   // the same network as SCL:
   #_w1 := "DB16000_OPC_UA_TRIGGER_ALARM".CLIENT.U1_STA3_COAXIAL.TRIGGERS.START_CAM_JET_CALIBRATION AND NOT "DB16000_OPC_UA_TRIGGER_ALARM".CLIENT.U1_STA3_COAXIAL.TRIGGERS.START_CAM_JET_CALIBRATION_P;   // rising edge
   "DB16000_OPC_UA_TRIGGER_ALARM".CLIENT.U1_STA3_COAXIAL.TRIGGERS.START_CAM_JET_CALIBRATION_P := "DB16000_OPC_UA_TRIGGER_ALARM".CLIENT.U1_STA3_COAXIAL.TRIGGERS.START_CAM_JET_CALIBRATION;
   "DB16313_U1_STA3_CAM_JET_CALIBRATE_TRIG"(REQ := #_w1,   // OPC_UA_MethodCall
                           ConnectionHdl := "DB16102_U1_STA3_CAM_CLIENT_CONFIGURATION".Connection.ConnectionHdl,
                           MethodHdl := "DB16102_U1_STA3_CAM_CLIENT_CONFIGURATION".MethodLists.U1_STA3_CAM_Calibrations.MethodHdls[2],
                           Timeout := "DB16102_U1_STA3_CAM_CLIENT_CONFIGURATION".Connection.ConnectInfo.SessionTimeout,
                           MethodResult := "DB16002_U1_STA3_COAXIAL_CLIENT_INTERFACE".U1_STA3_CAM_Calibrations.MethodResultList[2],
                           OutputArguments := "DB16002_U1_STA3_COAXIAL_CLIENT_INTERFACE".U1_STA3_CAM_Calibrations."Calibrate jet".Outputs,
                           Status => "DB16002_U1_STA3_COAXIAL_CLIENT_INTERFACE".U1_STA3_CAM_Calibrations.MethodStatusList[2]);
END_REGION

REGION Network 32: UNIT 1 STATION 3 COAXIAL CAMERA START CLADDING CALIBRATION TRIGGER CALL
   RUNG wire#powerrail
      "DB16314_U1_STA3_CAM_CLADDING_CALIBRATE_TRIG".OPC_UA_MethodCall(REQ := wire#w1, ConnectionHdl := "DB16102_U1_STA3_CAM_CLIENT_CONFIGURATION".Connection.ConnectionHdl, MethodHdl := "DB16102_U1_STA3_CAM_CLIENT_CONFIGURATION".MethodLists.U1_STA3_CAM_Calibrations.MethodHdls[3], Timeout := "DB16102_U1_STA3_CAM_CLIENT_CONFIGURATION".Connection.ConnectInfo.SessionTimeout, MethodResult := "DB16002_U1_STA3_COAXIAL_CLIENT_INTERFACE".U1_STA3_CAM_Calibrations.MethodResultList[3], InputArguments :=, OutputArguments := "DB16002_U1_STA3_COAXIAL_CLIENT_INTERFACE".U1_STA3_CAM_Calibrations."Calibrate cladding".Outputs, Done =>, Busy =>, Error =>, Status => "DB16002_U1_STA3_COAXIAL_CLIENT_INTERFACE".U1_STA3_CAM_Calibrations.MethodStatusList[3])
   END_RUNG
   RUNG wire#powerrail
      Contact( "DB16000_OPC_UA_TRIGGER_ALARM".CLIENT.U1_STA3_COAXIAL.TRIGGERS.START_CAM_CLADDING_CALIBRATION )
      P_Trig( "DB16000_OPC_UA_TRIGGER_ALARM".CLIENT.U1_STA3_COAXIAL.TRIGGERS.START_CAM_CLADDING_CALIBRATION_P )
   END_RUNG wire#w1
   // the same network as SCL:
   #_w1 := "DB16000_OPC_UA_TRIGGER_ALARM".CLIENT.U1_STA3_COAXIAL.TRIGGERS.START_CAM_CLADDING_CALIBRATION AND NOT "DB16000_OPC_UA_TRIGGER_ALARM".CLIENT.U1_STA3_COAXIAL.TRIGGERS.START_CAM_CLADDING_CALIBRATION_P;   // rising edge
   "DB16000_OPC_UA_TRIGGER_ALARM".CLIENT.U1_STA3_COAXIAL.TRIGGERS.START_CAM_CLADDING_CALIBRATION_P := "DB16000_OPC_UA_TRIGGER_ALARM".CLIENT.U1_STA3_COAXIAL.TRIGGERS.START_CAM_CLADDING_CALIBRATION;
   "DB16314_U1_STA3_CAM_CLADDING_CALIBRATE_TRIG"(REQ := #_w1,   // OPC_UA_MethodCall
                           ConnectionHdl := "DB16102_U1_STA3_CAM_CLIENT_CONFIGURATION".Connection.ConnectionHdl,
                           MethodHdl := "DB16102_U1_STA3_CAM_CLIENT_CONFIGURATION".MethodLists.U1_STA3_CAM_Calibrations.MethodHdls[3],
                           Timeout := "DB16102_U1_STA3_CAM_CLIENT_CONFIGURATION".Connection.ConnectInfo.SessionTimeout,
                           MethodResult := "DB16002_U1_STA3_COAXIAL_CLIENT_INTERFACE".U1_STA3_CAM_Calibrations.MethodResultList[3],
                           OutputArguments := "DB16002_U1_STA3_COAXIAL_CLIENT_INTERFACE".U1_STA3_CAM_Calibrations."Calibrate cladding".Outputs,
                           Status => "DB16002_U1_STA3_COAXIAL_CLIENT_INTERFACE".U1_STA3_CAM_Calibrations.MethodStatusList[3]);
END_REGION

REGION Network 33: UNIT 1 STATION 3 COAXIAL CAMERA START NOZZLE ANALISIS TRIGGER CALL
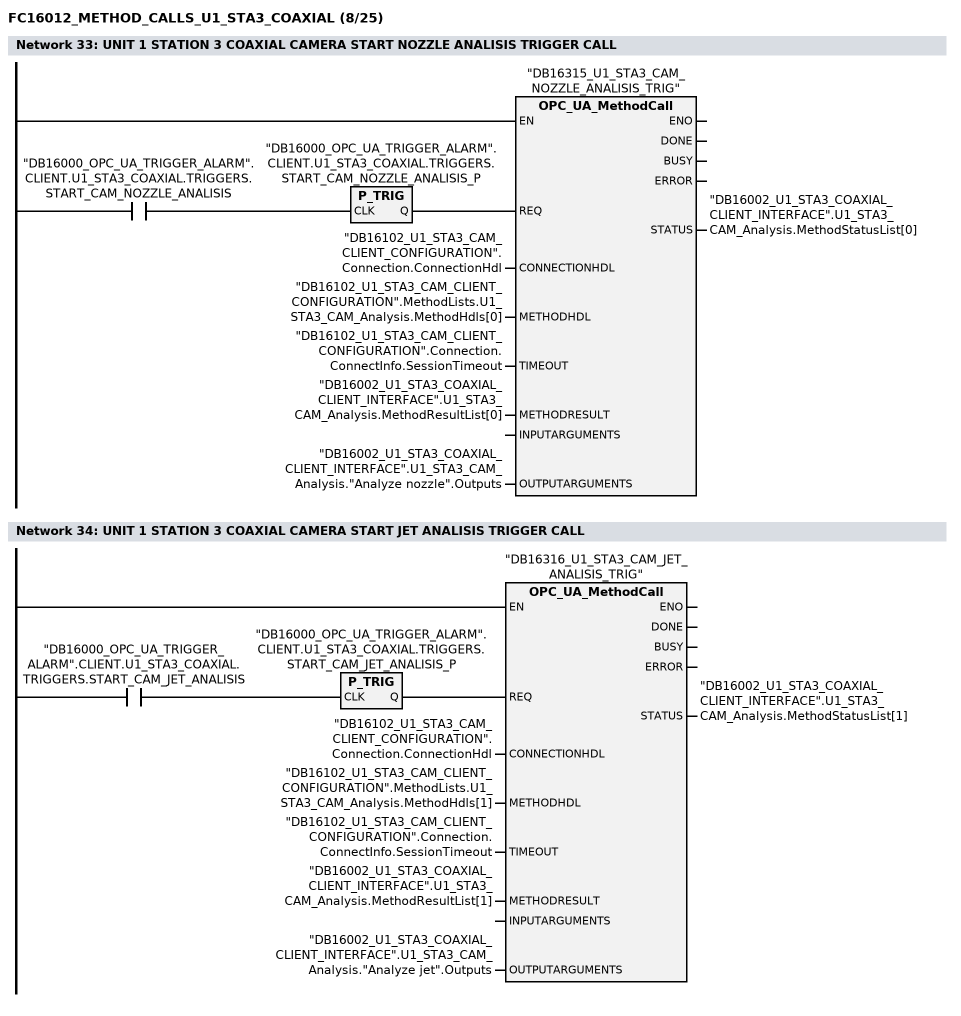
   RUNG wire#powerrail
      "DB16315_U1_STA3_CAM_NOZZLE_ANALISIS_TRIG".OPC_UA_MethodCall(REQ := wire#w1, ConnectionHdl := "DB16102_U1_STA3_CAM_CLIENT_CONFIGURATION".Connection.ConnectionHdl, MethodHdl := "DB16102_U1_STA3_CAM_CLIENT_CONFIGURATION".MethodLists.U1_STA3_CAM_Analysis.MethodHdls[0], Timeout := "DB16102_U1_STA3_CAM_CLIENT_CONFIGURATION".Connection.ConnectInfo.SessionTimeout, MethodResult := "DB16002_U1_STA3_COAXIAL_CLIENT_INTERFACE".U1_STA3_CAM_Analysis.MethodResultList[0], InputArguments :=, OutputArguments := "DB16002_U1_STA3_COAXIAL_CLIENT_INTERFACE".U1_STA3_CAM_Analysis."Analyze nozzle".Outputs, Done =>, Busy =>, Error =>, Status => "DB16002_U1_STA3_COAXIAL_CLIENT_INTERFACE".U1_STA3_CAM_Analysis.MethodStatusList[0])
   END_RUNG
   RUNG wire#powerrail
      Contact( "DB16000_OPC_UA_TRIGGER_ALARM".CLIENT.U1_STA3_COAXIAL.TRIGGERS.START_CAM_NOZZLE_ANALISIS )
      P_Trig( "DB16000_OPC_UA_TRIGGER_ALARM".CLIENT.U1_STA3_COAXIAL.TRIGGERS.START_CAM_NOZZLE_ANALISIS_P )
   END_RUNG wire#w1
   // the same network as SCL:
   #_w1 := "DB16000_OPC_UA_TRIGGER_ALARM".CLIENT.U1_STA3_COAXIAL.TRIGGERS.START_CAM_NOZZLE_ANALISIS AND NOT "DB16000_OPC_UA_TRIGGER_ALARM".CLIENT.U1_STA3_COAXIAL.TRIGGERS.START_CAM_NOZZLE_ANALISIS_P;   // rising edge
   "DB16000_OPC_UA_TRIGGER_ALARM".CLIENT.U1_STA3_COAXIAL.TRIGGERS.START_CAM_NOZZLE_ANALISIS_P := "DB16000_OPC_UA_TRIGGER_ALARM".CLIENT.U1_STA3_COAXIAL.TRIGGERS.START_CAM_NOZZLE_ANALISIS;
   "DB16315_U1_STA3_CAM_NOZZLE_ANALISIS_TRIG"(REQ := #_w1,   // OPC_UA_MethodCall
                           ConnectionHdl := "DB16102_U1_STA3_CAM_CLIENT_CONFIGURATION".Connection.ConnectionHdl,
                           MethodHdl := "DB16102_U1_STA3_CAM_CLIENT_CONFIGURATION".MethodLists.U1_STA3_CAM_Analysis.MethodHdls[0],
                           Timeout := "DB16102_U1_STA3_CAM_CLIENT_CONFIGURATION".Connection.ConnectInfo.SessionTimeout,
                           MethodResult := "DB16002_U1_STA3_COAXIAL_CLIENT_INTERFACE".U1_STA3_CAM_Analysis.MethodResultList[0],
                           OutputArguments := "DB16002_U1_STA3_COAXIAL_CLIENT_INTERFACE".U1_STA3_CAM_Analysis."Analyze nozzle".Outputs,
                           Status => "DB16002_U1_STA3_COAXIAL_CLIENT_INTERFACE".U1_STA3_CAM_Analysis.MethodStatusList[0]);
END_REGION

REGION Network 34: UNIT 1 STATION 3 COAXIAL CAMERA START JET ANALISIS TRIGGER CALL
   RUNG wire#powerrail
      "DB16316_U1_STA3_CAM_JET_ANALISIS_TRIG".OPC_UA_MethodCall(REQ := wire#w1, ConnectionHdl := "DB16102_U1_STA3_CAM_CLIENT_CONFIGURATION".Connection.ConnectionHdl, MethodHdl := "DB16102_U1_STA3_CAM_CLIENT_CONFIGURATION".MethodLists.U1_STA3_CAM_Analysis.MethodHdls[1], Timeout := "DB16102_U1_STA3_CAM_CLIENT_CONFIGURATION".Connection.ConnectInfo.SessionTimeout, MethodResult := "DB16002_U1_STA3_COAXIAL_CLIENT_INTERFACE".U1_STA3_CAM_Analysis.MethodResultList[1], InputArguments :=, OutputArguments := "DB16002_U1_STA3_COAXIAL_CLIENT_INTERFACE".U1_STA3_CAM_Analysis."Analyze jet".Outputs, Done =>, Busy =>, Error =>, Status => "DB16002_U1_STA3_COAXIAL_CLIENT_INTERFACE".U1_STA3_CAM_Analysis.MethodStatusList[1])
   END_RUNG
   RUNG wire#powerrail
      Contact( "DB16000_OPC_UA_TRIGGER_ALARM".CLIENT.U1_STA3_COAXIAL.TRIGGERS.START_CAM_JET_ANALISIS )
      P_Trig( "DB16000_OPC_UA_TRIGGER_ALARM".CLIENT.U1_STA3_COAXIAL.TRIGGERS.START_CAM_JET_ANALISIS_P )
   END_RUNG wire#w1
   // the same network as SCL:
   #_w1 := "DB16000_OPC_UA_TRIGGER_ALARM".CLIENT.U1_STA3_COAXIAL.TRIGGERS.START_CAM_JET_ANALISIS AND NOT "DB16000_OPC_UA_TRIGGER_ALARM".CLIENT.U1_STA3_COAXIAL.TRIGGERS.START_CAM_JET_ANALISIS_P;   // rising edge
   "DB16000_OPC_UA_TRIGGER_ALARM".CLIENT.U1_STA3_COAXIAL.TRIGGERS.START_CAM_JET_ANALISIS_P := "DB16000_OPC_UA_TRIGGER_ALARM".CLIENT.U1_STA3_COAXIAL.TRIGGERS.START_CAM_JET_ANALISIS;
   "DB16316_U1_STA3_CAM_JET_ANALISIS_TRIG"(REQ := #_w1,   // OPC_UA_MethodCall
                           ConnectionHdl := "DB16102_U1_STA3_CAM_CLIENT_CONFIGURATION".Connection.ConnectionHdl,
                           MethodHdl := "DB16102_U1_STA3_CAM_CLIENT_CONFIGURATION".MethodLists.U1_STA3_CAM_Analysis.MethodHdls[1],
                           Timeout := "DB16102_U1_STA3_CAM_CLIENT_CONFIGURATION".Connection.ConnectInfo.SessionTimeout,
                           MethodResult := "DB16002_U1_STA3_COAXIAL_CLIENT_INTERFACE".U1_STA3_CAM_Analysis.MethodResultList[1],
                           OutputArguments := "DB16002_U1_STA3_COAXIAL_CLIENT_INTERFACE".U1_STA3_CAM_Analysis."Analyze jet".Outputs,
                           Status => "DB16002_U1_STA3_COAXIAL_CLIENT_INTERFACE".U1_STA3_CAM_Analysis.MethodStatusList[1]);
END_REGION

REGION Network 35: UNIT 1 STATION 3 COAXIAL CAMERA START CLADDING ANALISIS TRIGGER CALL
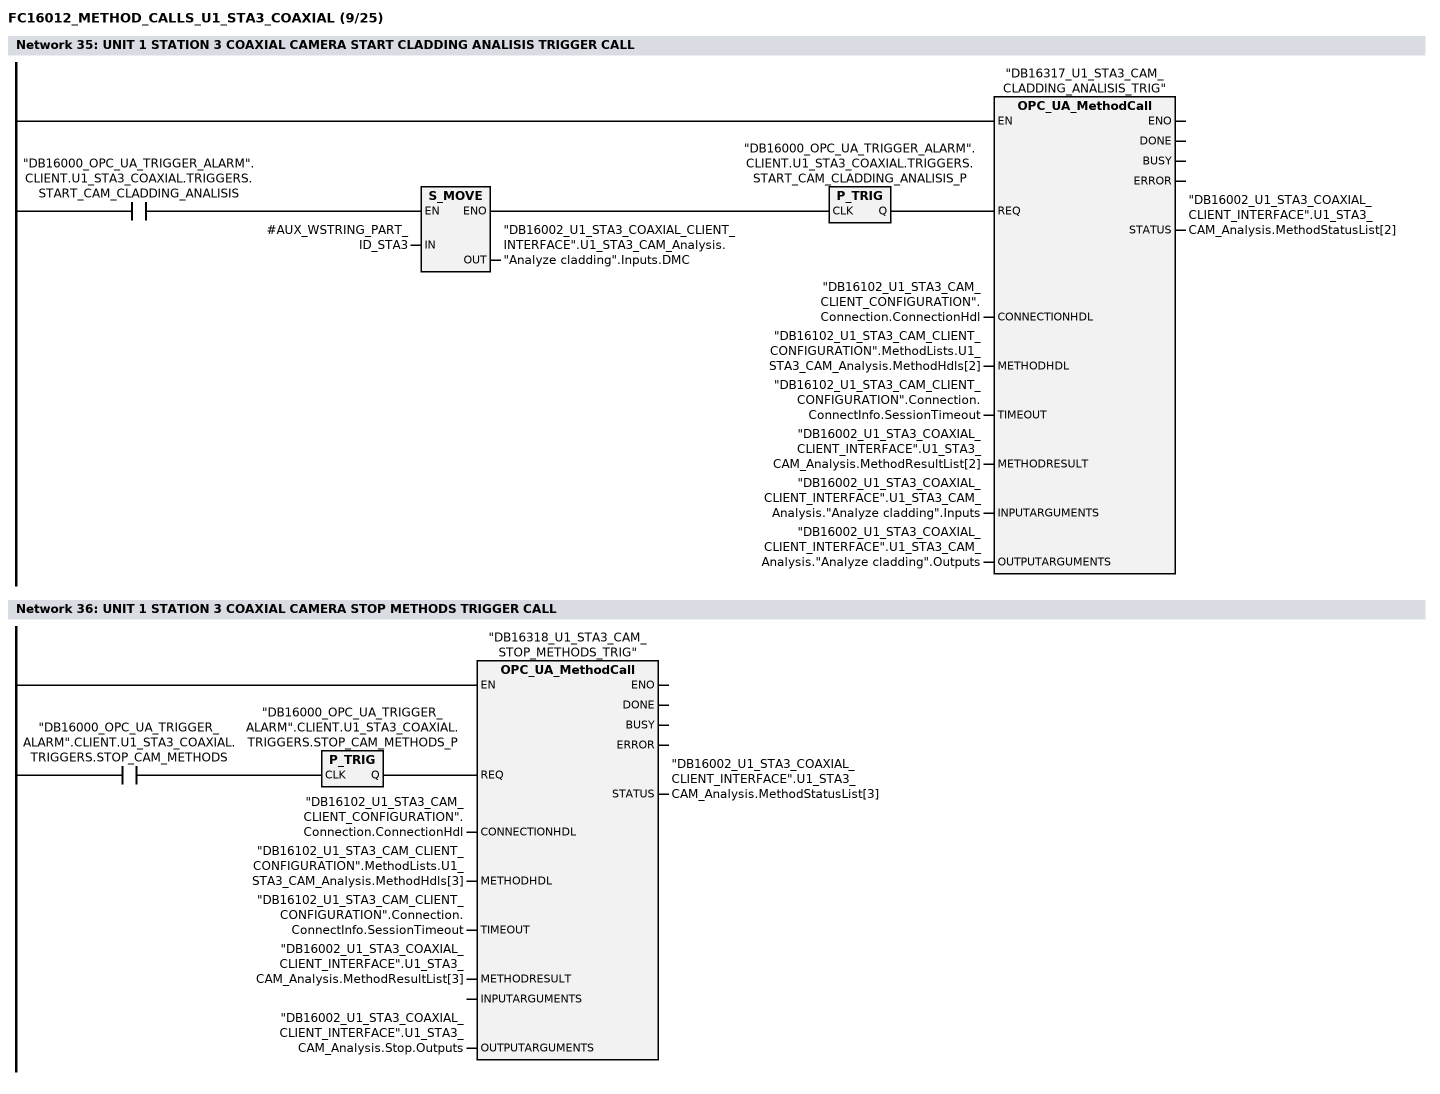
   RUNG wire#powerrail
      "DB16317_U1_STA3_CAM_CLADDING_ANALISIS_TRIG".OPC_UA_MethodCall(REQ := wire#w1, ConnectionHdl := "DB16102_U1_STA3_CAM_CLIENT_CONFIGURATION".Connection.ConnectionHdl, MethodHdl := "DB16102_U1_STA3_CAM_CLIENT_CONFIGURATION".MethodLists.U1_STA3_CAM_Analysis.MethodHdls[2], Timeout := "DB16102_U1_STA3_CAM_CLIENT_CONFIGURATION".Connection.ConnectInfo.SessionTimeout, MethodResult := "DB16002_U1_STA3_COAXIAL_CLIENT_INTERFACE".U1_STA3_CAM_Analysis.MethodResultList[2], InputArguments := "DB16002_U1_STA3_COAXIAL_CLIENT_INTERFACE".U1_STA3_CAM_Analysis."Analyze cladding".Inputs, OutputArguments := "DB16002_U1_STA3_COAXIAL_CLIENT_INTERFACE".U1_STA3_CAM_Analysis."Analyze cladding".Outputs, Done =>, Busy =>, Error =>, Status => "DB16002_U1_STA3_COAXIAL_CLIENT_INTERFACE".U1_STA3_CAM_Analysis.MethodStatusList[2])
   END_RUNG
   RUNG wire#powerrail
      Contact( "DB16000_OPC_UA_TRIGGER_ALARM".CLIENT.U1_STA3_COAXIAL.TRIGGERS.START_CAM_CLADDING_ANALISIS )
      S_Move(in := #AUX_WSTRING_PART_ID_STA3, out => "DB16002_U1_STA3_COAXIAL_CLIENT_INTERFACE".U1_STA3_CAM_Analysis."Analyze cladding".Inputs.DMC)
      P_Trig( "DB16000_OPC_UA_TRIGGER_ALARM".CLIENT.U1_STA3_COAXIAL.TRIGGERS.START_CAM_CLADDING_ANALISIS_P )
   END_RUNG wire#w1
   // the same network as SCL:
   IF "DB16000_OPC_UA_TRIGGER_ALARM".CLIENT.U1_STA3_COAXIAL.TRIGGERS.START_CAM_CLADDING_ANALISIS THEN
       "DB16002_U1_STA3_COAXIAL_CLIENT_INTERFACE".U1_STA3_CAM_Analysis."Analyze cladding".Inputs.DMC := #AUX_WSTRING_PART_ID_STA3;
   END_IF;
   #_w1 := "DB16000_OPC_UA_TRIGGER_ALARM".CLIENT.U1_STA3_COAXIAL.TRIGGERS.START_CAM_CLADDING_ANALISIS AND NOT "DB16000_OPC_UA_TRIGGER_ALARM".CLIENT.U1_STA3_COAXIAL.TRIGGERS.START_CAM_CLADDING_ANALISIS_P;   // rising edge
   "DB16000_OPC_UA_TRIGGER_ALARM".CLIENT.U1_STA3_COAXIAL.TRIGGERS.START_CAM_CLADDING_ANALISIS_P := "DB16000_OPC_UA_TRIGGER_ALARM".CLIENT.U1_STA3_COAXIAL.TRIGGERS.START_CAM_CLADDING_ANALISIS;
   "DB16317_U1_STA3_CAM_CLADDING_ANALISIS_TRIG"(REQ := #_w1,   // OPC_UA_MethodCall
                           ConnectionHdl := "DB16102_U1_STA3_CAM_CLIENT_CONFIGURATION".Connection.ConnectionHdl,
                           MethodHdl := "DB16102_U1_STA3_CAM_CLIENT_CONFIGURATION".MethodLists.U1_STA3_CAM_Analysis.MethodHdls[2],
                           Timeout := "DB16102_U1_STA3_CAM_CLIENT_CONFIGURATION".Connection.ConnectInfo.SessionTimeout,
                           MethodResult := "DB16002_U1_STA3_COAXIAL_CLIENT_INTERFACE".U1_STA3_CAM_Analysis.MethodResultList[2],
                           InputArguments := "DB16002_U1_STA3_COAXIAL_CLIENT_INTERFACE".U1_STA3_CAM_Analysis."Analyze cladding".Inputs,
                           OutputArguments := "DB16002_U1_STA3_COAXIAL_CLIENT_INTERFACE".U1_STA3_CAM_Analysis."Analyze cladding".Outputs,
                           Status => "DB16002_U1_STA3_COAXIAL_CLIENT_INTERFACE".U1_STA3_CAM_Analysis.MethodStatusList[2]);
END_REGION

REGION Network 36: UNIT 1 STATION 3 COAXIAL CAMERA STOP METHODS TRIGGER CALL
   RUNG wire#powerrail
      "DB16318_U1_STA3_CAM_STOP_METHODS_TRIG".OPC_UA_MethodCall(REQ := wire#w1, ConnectionHdl := "DB16102_U1_STA3_CAM_CLIENT_CONFIGURATION".Connection.ConnectionHdl, MethodHdl := "DB16102_U1_STA3_CAM_CLIENT_CONFIGURATION".MethodLists.U1_STA3_CAM_Analysis.MethodHdls[3], Timeout := "DB16102_U1_STA3_CAM_CLIENT_CONFIGURATION".Connection.ConnectInfo.SessionTimeout, MethodResult := "DB16002_U1_STA3_COAXIAL_CLIENT_INTERFACE".U1_STA3_CAM_Analysis.MethodResultList[3], InputArguments :=, OutputArguments := "DB16002_U1_STA3_COAXIAL_CLIENT_INTERFACE".U1_STA3_CAM_Analysis.Stop.Outputs, Done =>, Busy =>, Error =>, Status => "DB16002_U1_STA3_COAXIAL_CLIENT_INTERFACE".U1_STA3_CAM_Analysis.MethodStatusList[3])
   END_RUNG
   RUNG wire#powerrail
      Contact( "DB16000_OPC_UA_TRIGGER_ALARM".CLIENT.U1_STA3_COAXIAL.TRIGGERS.STOP_CAM_METHODS )
      P_Trig( "DB16000_OPC_UA_TRIGGER_ALARM".CLIENT.U1_STA3_COAXIAL.TRIGGERS.STOP_CAM_METHODS_P )
   END_RUNG wire#w1
   // the same network as SCL:
   #_w1 := "DB16000_OPC_UA_TRIGGER_ALARM".CLIENT.U1_STA3_COAXIAL.TRIGGERS.STOP_CAM_METHODS AND NOT "DB16000_OPC_UA_TRIGGER_ALARM".CLIENT.U1_STA3_COAXIAL.TRIGGERS.STOP_CAM_METHODS_P;   // rising edge
   "DB16000_OPC_UA_TRIGGER_ALARM".CLIENT.U1_STA3_COAXIAL.TRIGGERS.STOP_CAM_METHODS_P := "DB16000_OPC_UA_TRIGGER_ALARM".CLIENT.U1_STA3_COAXIAL.TRIGGERS.STOP_CAM_METHODS;
   "DB16318_U1_STA3_CAM_STOP_METHODS_TRIG"(REQ := #_w1,   // OPC_UA_MethodCall
                           ConnectionHdl := "DB16102_U1_STA3_CAM_CLIENT_CONFIGURATION".Connection.ConnectionHdl,
                           MethodHdl := "DB16102_U1_STA3_CAM_CLIENT_CONFIGURATION".MethodLists.U1_STA3_CAM_Analysis.MethodHdls[3],
                           Timeout := "DB16102_U1_STA3_CAM_CLIENT_CONFIGURATION".Connection.ConnectInfo.SessionTimeout,
                           MethodResult := "DB16002_U1_STA3_COAXIAL_CLIENT_INTERFACE".U1_STA3_CAM_Analysis.MethodResultList[3],
                           OutputArguments := "DB16002_U1_STA3_COAXIAL_CLIENT_INTERFACE".U1_STA3_CAM_Analysis.Stop.Outputs,
                           Status => "DB16002_U1_STA3_COAXIAL_CLIENT_INTERFACE".U1_STA3_CAM_Analysis.MethodStatusList[3]);
END_REGION

REGION Network 37: UNIT 1 STATION 3 COAXIAL CAMERA RESET PC TRIGGER CALL
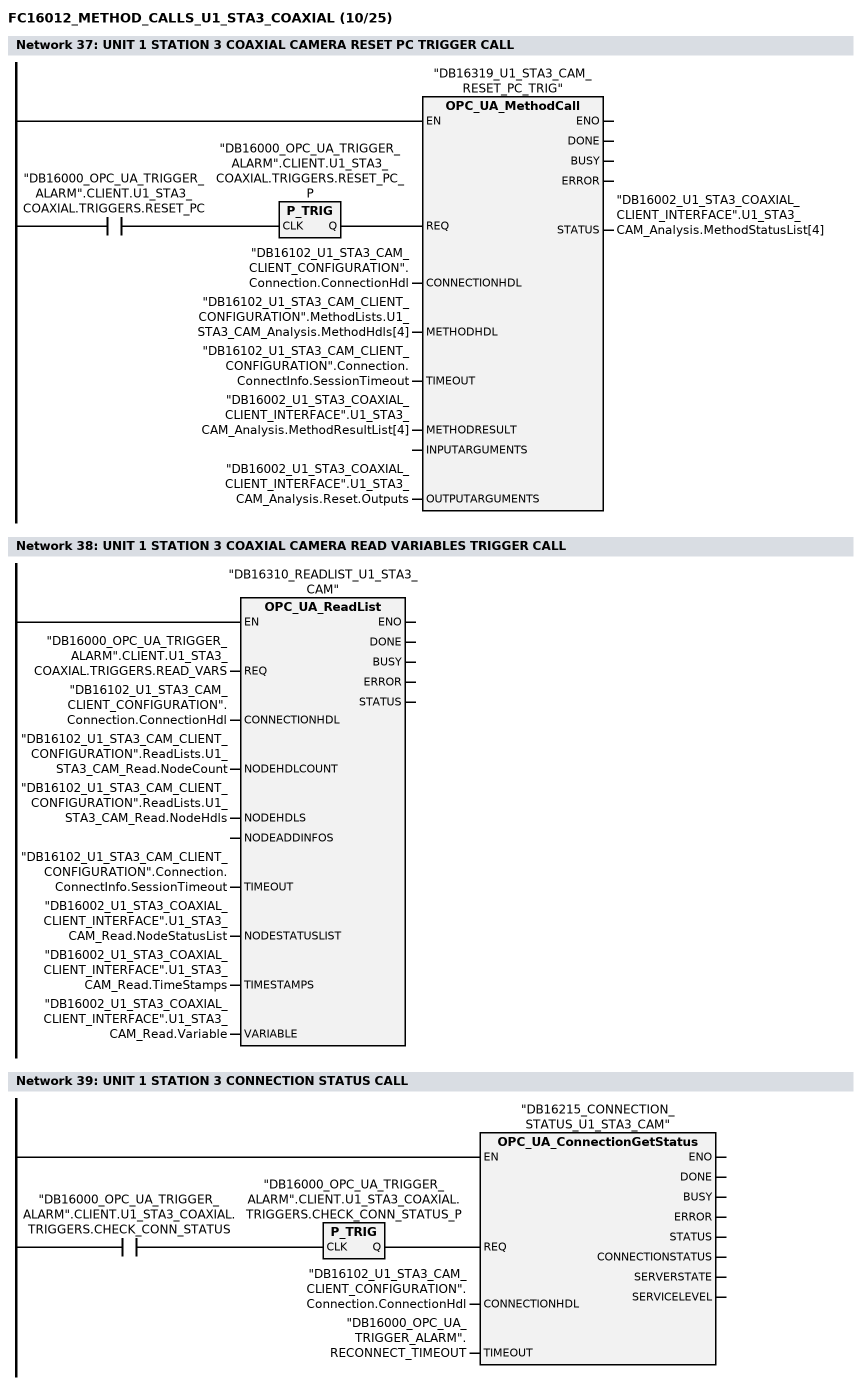
   RUNG wire#powerrail
      "DB16319_U1_STA3_CAM_RESET_PC_TRIG".OPC_UA_MethodCall(REQ := wire#w1, ConnectionHdl := "DB16102_U1_STA3_CAM_CLIENT_CONFIGURATION".Connection.ConnectionHdl, MethodHdl := "DB16102_U1_STA3_CAM_CLIENT_CONFIGURATION".MethodLists.U1_STA3_CAM_Analysis.MethodHdls[4], Timeout := "DB16102_U1_STA3_CAM_CLIENT_CONFIGURATION".Connection.ConnectInfo.SessionTimeout, MethodResult := "DB16002_U1_STA3_COAXIAL_CLIENT_INTERFACE".U1_STA3_CAM_Analysis.MethodResultList[4], InputArguments :=, OutputArguments := "DB16002_U1_STA3_COAXIAL_CLIENT_INTERFACE".U1_STA3_CAM_Analysis.Reset.Outputs, Done =>, Busy =>, Error =>, Status => "DB16002_U1_STA3_COAXIAL_CLIENT_INTERFACE".U1_STA3_CAM_Analysis.MethodStatusList[4])
   END_RUNG
   RUNG wire#powerrail
      Contact( "DB16000_OPC_UA_TRIGGER_ALARM".CLIENT.U1_STA3_COAXIAL.TRIGGERS.RESET_PC )
      P_Trig( "DB16000_OPC_UA_TRIGGER_ALARM".CLIENT.U1_STA3_COAXIAL.TRIGGERS.RESET_PC_P )
   END_RUNG wire#w1
   // the same network as SCL:
   #_w1 := "DB16000_OPC_UA_TRIGGER_ALARM".CLIENT.U1_STA3_COAXIAL.TRIGGERS.RESET_PC AND NOT "DB16000_OPC_UA_TRIGGER_ALARM".CLIENT.U1_STA3_COAXIAL.TRIGGERS.RESET_PC_P;   // rising edge
   "DB16000_OPC_UA_TRIGGER_ALARM".CLIENT.U1_STA3_COAXIAL.TRIGGERS.RESET_PC_P := "DB16000_OPC_UA_TRIGGER_ALARM".CLIENT.U1_STA3_COAXIAL.TRIGGERS.RESET_PC;
   "DB16319_U1_STA3_CAM_RESET_PC_TRIG"(REQ := #_w1,   // OPC_UA_MethodCall
                           ConnectionHdl := "DB16102_U1_STA3_CAM_CLIENT_CONFIGURATION".Connection.ConnectionHdl,
                           MethodHdl := "DB16102_U1_STA3_CAM_CLIENT_CONFIGURATION".MethodLists.U1_STA3_CAM_Analysis.MethodHdls[4],
                           Timeout := "DB16102_U1_STA3_CAM_CLIENT_CONFIGURATION".Connection.ConnectInfo.SessionTimeout,
                           MethodResult := "DB16002_U1_STA3_COAXIAL_CLIENT_INTERFACE".U1_STA3_CAM_Analysis.MethodResultList[4],
                           OutputArguments := "DB16002_U1_STA3_COAXIAL_CLIENT_INTERFACE".U1_STA3_CAM_Analysis.Reset.Outputs,
                           Status => "DB16002_U1_STA3_COAXIAL_CLIENT_INTERFACE".U1_STA3_CAM_Analysis.MethodStatusList[4]);
END_REGION

REGION Network 38: UNIT 1 STATION 3 COAXIAL CAMERA READ VARIABLES TRIGGER CALL
   RUNG wire#powerrail
      "DB16310_READLIST_U1_STA3_CAM".OPC_UA_ReadList(REQ := "DB16000_OPC_UA_TRIGGER_ALARM".CLIENT.U1_STA3_COAXIAL.TRIGGERS.READ_VARS, ConnectionHdl := "DB16102_U1_STA3_CAM_CLIENT_CONFIGURATION".Connection.ConnectionHdl, NodeHdlCount := "DB16102_U1_STA3_CAM_CLIENT_CONFIGURATION".ReadLists.U1_STA3_CAM_Read.NodeCount, NodeHdls := "DB16102_U1_STA3_CAM_CLIENT_CONFIGURATION".ReadLists.U1_STA3_CAM_Read.NodeHdls, NodeAddInfos :=, Timeout := "DB16102_U1_STA3_CAM_CLIENT_CONFIGURATION".Connection.ConnectInfo.SessionTimeout, NodeStatusList := "DB16002_U1_STA3_COAXIAL_CLIENT_INTERFACE".U1_STA3_CAM_Read.NodeStatusList, TimeStamps := "DB16002_U1_STA3_COAXIAL_CLIENT_INTERFACE".U1_STA3_CAM_Read.TimeStamps, Variable := "DB16002_U1_STA3_COAXIAL_CLIENT_INTERFACE".U1_STA3_CAM_Read.Variable, Done =>, Busy =>, Error =>, Status =>)
   END_RUNG
   // the same network as SCL:
   "DB16310_READLIST_U1_STA3_CAM"(REQ := "DB16000_OPC_UA_TRIGGER_ALARM".CLIENT.U1_STA3_COAXIAL.TRIGGERS.READ_VARS,   // OPC_UA_ReadList
                           ConnectionHdl := "DB16102_U1_STA3_CAM_CLIENT_CONFIGURATION".Connection.ConnectionHdl,
                           NodeHdlCount := "DB16102_U1_STA3_CAM_CLIENT_CONFIGURATION".ReadLists.U1_STA3_CAM_Read.NodeCount,
                           NodeHdls := "DB16102_U1_STA3_CAM_CLIENT_CONFIGURATION".ReadLists.U1_STA3_CAM_Read.NodeHdls,
                           Timeout := "DB16102_U1_STA3_CAM_CLIENT_CONFIGURATION".Connection.ConnectInfo.SessionTimeout,
                           NodeStatusList := "DB16002_U1_STA3_COAXIAL_CLIENT_INTERFACE".U1_STA3_CAM_Read.NodeStatusList,
                           TimeStamps := "DB16002_U1_STA3_COAXIAL_CLIENT_INTERFACE".U1_STA3_CAM_Read.TimeStamps,
                           Variable := "DB16002_U1_STA3_COAXIAL_CLIENT_INTERFACE".U1_STA3_CAM_Read.Variable);
END_REGION

REGION Network 39: UNIT 1 STATION 3 CONNECTION STATUS CALL
   RUNG wire#powerrail
      "DB16215_CONNECTION_STATUS_U1_STA3_CAM".OPC_UA_ConnectionGetStatus(REQ := wire#w1, ConnectionHdl := "DB16102_U1_STA3_CAM_CLIENT_CONFIGURATION".Connection.ConnectionHdl, Timeout := "DB16000_OPC_UA_TRIGGER_ALARM".RECONNECT_TIMEOUT, Done =>, Busy =>, Error =>, Status =>, ConnectionStatus =>, ServerState =>, ServiceLevel =>)
   END_RUNG
   RUNG wire#powerrail
      Contact( "DB16000_OPC_UA_TRIGGER_ALARM".CLIENT.U1_STA3_COAXIAL.TRIGGERS.CHECK_CONN_STATUS )
      P_Trig( "DB16000_OPC_UA_TRIGGER_ALARM".CLIENT.U1_STA3_COAXIAL.TRIGGERS.CHECK_CONN_STATUS_P )
   END_RUNG wire#w1
   // the same network as SCL:
   #_w1 := "DB16000_OPC_UA_TRIGGER_ALARM".CLIENT.U1_STA3_COAXIAL.TRIGGERS.CHECK_CONN_STATUS AND NOT "DB16000_OPC_UA_TRIGGER_ALARM".CLIENT.U1_STA3_COAXIAL.TRIGGERS.CHECK_CONN_STATUS_P;   // rising edge
   "DB16000_OPC_UA_TRIGGER_ALARM".CLIENT.U1_STA3_COAXIAL.TRIGGERS.CHECK_CONN_STATUS_P := "DB16000_OPC_UA_TRIGGER_ALARM".CLIENT.U1_STA3_COAXIAL.TRIGGERS.CHECK_CONN_STATUS;
   "DB16215_CONNECTION_STATUS_U1_STA3_CAM"(REQ := #_w1,   // OPC_UA_ConnectionGetStatus
                           ConnectionHdl := "DB16102_U1_STA3_CAM_CLIENT_CONFIGURATION".Connection.ConnectionHdl,
                           Timeout := "DB16000_OPC_UA_TRIGGER_ALARM".RECONNECT_TIMEOUT);
END_REGION

REGION Network 40: UNIT 1 STATION 3 RELEASE HANDLE LIST CALL
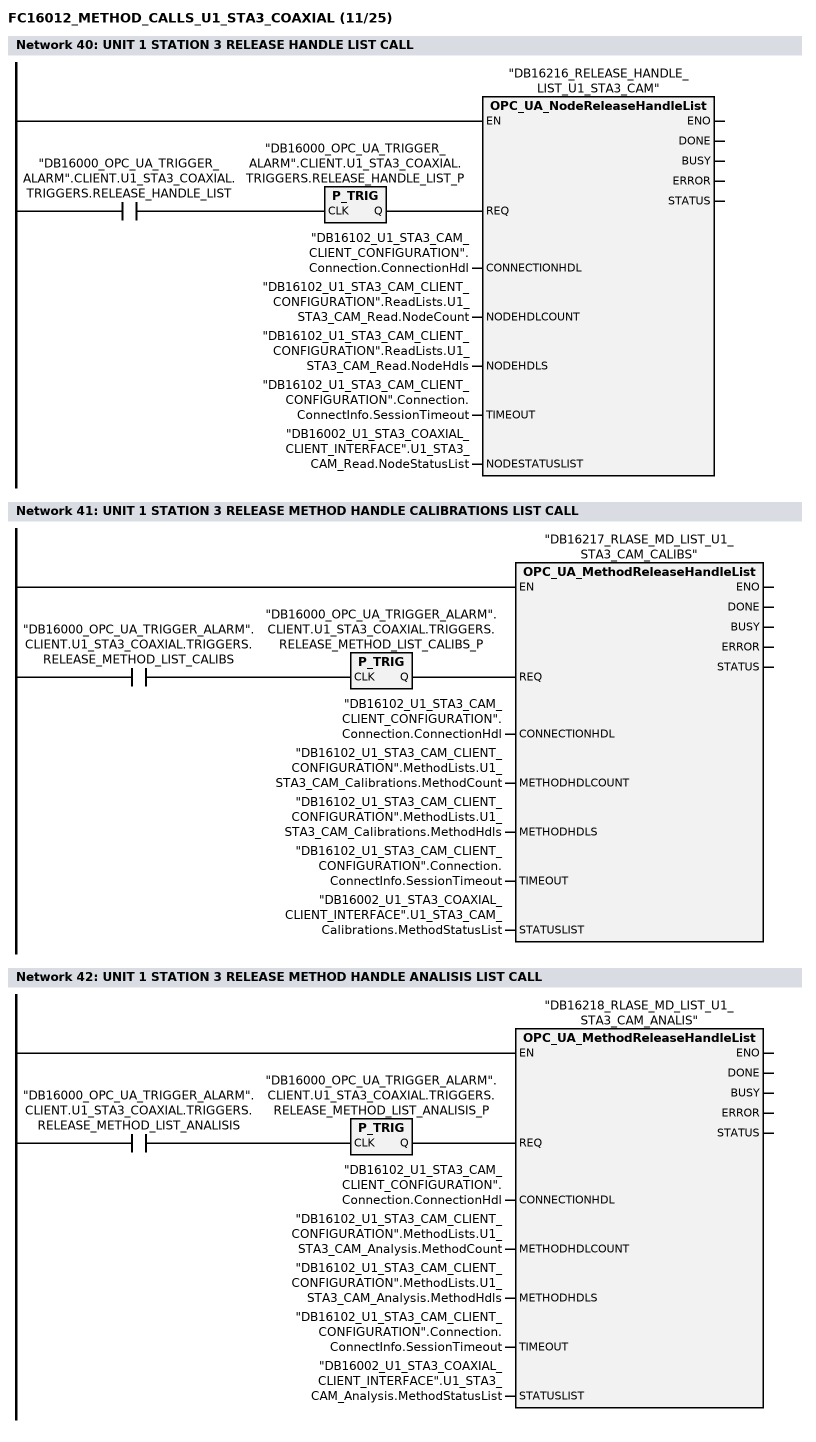
   RUNG wire#powerrail
      "DB16216_RELEASE_HANDLE_LIST_U1_STA3_CAM".OPC_UA_NodeReleaseHandleList(REQ := wire#w1, ConnectionHdl := "DB16102_U1_STA3_CAM_CLIENT_CONFIGURATION".Connection.ConnectionHdl, NodeHdlCount := "DB16102_U1_STA3_CAM_CLIENT_CONFIGURATION".ReadLists.U1_STA3_CAM_Read.NodeCount, NodeHdls := "DB16102_U1_STA3_CAM_CLIENT_CONFIGURATION".ReadLists.U1_STA3_CAM_Read.NodeHdls, Timeout := "DB16102_U1_STA3_CAM_CLIENT_CONFIGURATION".Connection.ConnectInfo.SessionTimeout, NodeStatusList := "DB16002_U1_STA3_COAXIAL_CLIENT_INTERFACE".U1_STA3_CAM_Read.NodeStatusList, Done =>, Busy =>, Error =>, Status =>)
   END_RUNG
   RUNG wire#powerrail
      Contact( "DB16000_OPC_UA_TRIGGER_ALARM".CLIENT.U1_STA3_COAXIAL.TRIGGERS.RELEASE_HANDLE_LIST )
      P_Trig( "DB16000_OPC_UA_TRIGGER_ALARM".CLIENT.U1_STA3_COAXIAL.TRIGGERS.RELEASE_HANDLE_LIST_P )
   END_RUNG wire#w1
   // the same network as SCL:
   #_w1 := "DB16000_OPC_UA_TRIGGER_ALARM".CLIENT.U1_STA3_COAXIAL.TRIGGERS.RELEASE_HANDLE_LIST AND NOT "DB16000_OPC_UA_TRIGGER_ALARM".CLIENT.U1_STA3_COAXIAL.TRIGGERS.RELEASE_HANDLE_LIST_P;   // rising edge
   "DB16000_OPC_UA_TRIGGER_ALARM".CLIENT.U1_STA3_COAXIAL.TRIGGERS.RELEASE_HANDLE_LIST_P := "DB16000_OPC_UA_TRIGGER_ALARM".CLIENT.U1_STA3_COAXIAL.TRIGGERS.RELEASE_HANDLE_LIST;
   "DB16216_RELEASE_HANDLE_LIST_U1_STA3_CAM"(REQ := #_w1,   // OPC_UA_NodeReleaseHandleList
                           ConnectionHdl := "DB16102_U1_STA3_CAM_CLIENT_CONFIGURATION".Connection.ConnectionHdl,
                           NodeHdlCount := "DB16102_U1_STA3_CAM_CLIENT_CONFIGURATION".ReadLists.U1_STA3_CAM_Read.NodeCount,
                           NodeHdls := "DB16102_U1_STA3_CAM_CLIENT_CONFIGURATION".ReadLists.U1_STA3_CAM_Read.NodeHdls,
                           Timeout := "DB16102_U1_STA3_CAM_CLIENT_CONFIGURATION".Connection.ConnectInfo.SessionTimeout,
                           NodeStatusList := "DB16002_U1_STA3_COAXIAL_CLIENT_INTERFACE".U1_STA3_CAM_Read.NodeStatusList);
END_REGION

REGION Network 41: UNIT 1 STATION 3 RELEASE METHOD HANDLE CALIBRATIONS LIST CALL
   RUNG wire#powerrail
      "DB16217_RLASE_MD_LIST_U1_STA3_CAM_CALIBS".OPC_UA_MethodReleaseHandleList(REQ := wire#w1, ConnectionHdl := "DB16102_U1_STA3_CAM_CLIENT_CONFIGURATION".Connection.ConnectionHdl, MethodHdlCount := "DB16102_U1_STA3_CAM_CLIENT_CONFIGURATION".MethodLists.U1_STA3_CAM_Calibrations.MethodCount, MethodHdls := "DB16102_U1_STA3_CAM_CLIENT_CONFIGURATION".MethodLists.U1_STA3_CAM_Calibrations.MethodHdls, Timeout := "DB16102_U1_STA3_CAM_CLIENT_CONFIGURATION".Connection.ConnectInfo.SessionTimeout, StatusList := "DB16002_U1_STA3_COAXIAL_CLIENT_INTERFACE".U1_STA3_CAM_Calibrations.MethodStatusList, Done =>, Busy =>, Error =>, Status =>)
   END_RUNG
   RUNG wire#powerrail
      Contact( "DB16000_OPC_UA_TRIGGER_ALARM".CLIENT.U1_STA3_COAXIAL.TRIGGERS.RELEASE_METHOD_LIST_CALIBS )
      P_Trig( "DB16000_OPC_UA_TRIGGER_ALARM".CLIENT.U1_STA3_COAXIAL.TRIGGERS.RELEASE_METHOD_LIST_CALIBS_P )
   END_RUNG wire#w1
   // the same network as SCL:
   #_w1 := "DB16000_OPC_UA_TRIGGER_ALARM".CLIENT.U1_STA3_COAXIAL.TRIGGERS.RELEASE_METHOD_LIST_CALIBS AND NOT "DB16000_OPC_UA_TRIGGER_ALARM".CLIENT.U1_STA3_COAXIAL.TRIGGERS.RELEASE_METHOD_LIST_CALIBS_P;   // rising edge
   "DB16000_OPC_UA_TRIGGER_ALARM".CLIENT.U1_STA3_COAXIAL.TRIGGERS.RELEASE_METHOD_LIST_CALIBS_P := "DB16000_OPC_UA_TRIGGER_ALARM".CLIENT.U1_STA3_COAXIAL.TRIGGERS.RELEASE_METHOD_LIST_CALIBS;
   "DB16217_RLASE_MD_LIST_U1_STA3_CAM_CALIBS"(REQ := #_w1,   // OPC_UA_MethodReleaseHandleList
                           ConnectionHdl := "DB16102_U1_STA3_CAM_CLIENT_CONFIGURATION".Connection.ConnectionHdl,
                           MethodHdlCount := "DB16102_U1_STA3_CAM_CLIENT_CONFIGURATION".MethodLists.U1_STA3_CAM_Calibrations.MethodCount,
                           MethodHdls := "DB16102_U1_STA3_CAM_CLIENT_CONFIGURATION".MethodLists.U1_STA3_CAM_Calibrations.MethodHdls,
                           Timeout := "DB16102_U1_STA3_CAM_CLIENT_CONFIGURATION".Connection.ConnectInfo.SessionTimeout,
                           StatusList := "DB16002_U1_STA3_COAXIAL_CLIENT_INTERFACE".U1_STA3_CAM_Calibrations.MethodStatusList);
END_REGION

REGION Network 42: UNIT 1 STATION 3 RELEASE METHOD HANDLE ANALISIS LIST CALL
   RUNG wire#powerrail
      "DB16218_RLASE_MD_LIST_U1_STA3_CAM_ANALIS".OPC_UA_MethodReleaseHandleList(REQ := wire#w1, ConnectionHdl := "DB16102_U1_STA3_CAM_CLIENT_CONFIGURATION".Connection.ConnectionHdl, MethodHdlCount := "DB16102_U1_STA3_CAM_CLIENT_CONFIGURATION".MethodLists.U1_STA3_CAM_Analysis.MethodCount, MethodHdls := "DB16102_U1_STA3_CAM_CLIENT_CONFIGURATION".MethodLists.U1_STA3_CAM_Analysis.MethodHdls, Timeout := "DB16102_U1_STA3_CAM_CLIENT_CONFIGURATION".Connection.ConnectInfo.SessionTimeout, StatusList := "DB16002_U1_STA3_COAXIAL_CLIENT_INTERFACE".U1_STA3_CAM_Analysis.MethodStatusList, Done =>, Busy =>, Error =>, Status =>)
   END_RUNG
   RUNG wire#powerrail
      Contact( "DB16000_OPC_UA_TRIGGER_ALARM".CLIENT.U1_STA3_COAXIAL.TRIGGERS.RELEASE_METHOD_LIST_ANALISIS )
      P_Trig( "DB16000_OPC_UA_TRIGGER_ALARM".CLIENT.U1_STA3_COAXIAL.TRIGGERS.RELEASE_METHOD_LIST_ANALISIS_P )
   END_RUNG wire#w1
   // the same network as SCL:
   #_w1 := "DB16000_OPC_UA_TRIGGER_ALARM".CLIENT.U1_STA3_COAXIAL.TRIGGERS.RELEASE_METHOD_LIST_ANALISIS AND NOT "DB16000_OPC_UA_TRIGGER_ALARM".CLIENT.U1_STA3_COAXIAL.TRIGGERS.RELEASE_METHOD_LIST_ANALISIS_P;   // rising edge
   "DB16000_OPC_UA_TRIGGER_ALARM".CLIENT.U1_STA3_COAXIAL.TRIGGERS.RELEASE_METHOD_LIST_ANALISIS_P := "DB16000_OPC_UA_TRIGGER_ALARM".CLIENT.U1_STA3_COAXIAL.TRIGGERS.RELEASE_METHOD_LIST_ANALISIS;
   "DB16218_RLASE_MD_LIST_U1_STA3_CAM_ANALIS"(REQ := #_w1,   // OPC_UA_MethodReleaseHandleList
                           ConnectionHdl := "DB16102_U1_STA3_CAM_CLIENT_CONFIGURATION".Connection.ConnectionHdl,
                           MethodHdlCount := "DB16102_U1_STA3_CAM_CLIENT_CONFIGURATION".MethodLists.U1_STA3_CAM_Analysis.MethodCount,
                           MethodHdls := "DB16102_U1_STA3_CAM_CLIENT_CONFIGURATION".MethodLists.U1_STA3_CAM_Analysis.MethodHdls,
                           Timeout := "DB16102_U1_STA3_CAM_CLIENT_CONFIGURATION".Connection.ConnectInfo.SessionTimeout,
                           StatusList := "DB16002_U1_STA3_COAXIAL_CLIENT_INTERFACE".U1_STA3_CAM_Analysis.MethodStatusList);
END_REGION

REGION Network 43: UNIT 1 STATION 3 DISCONNECT CALL
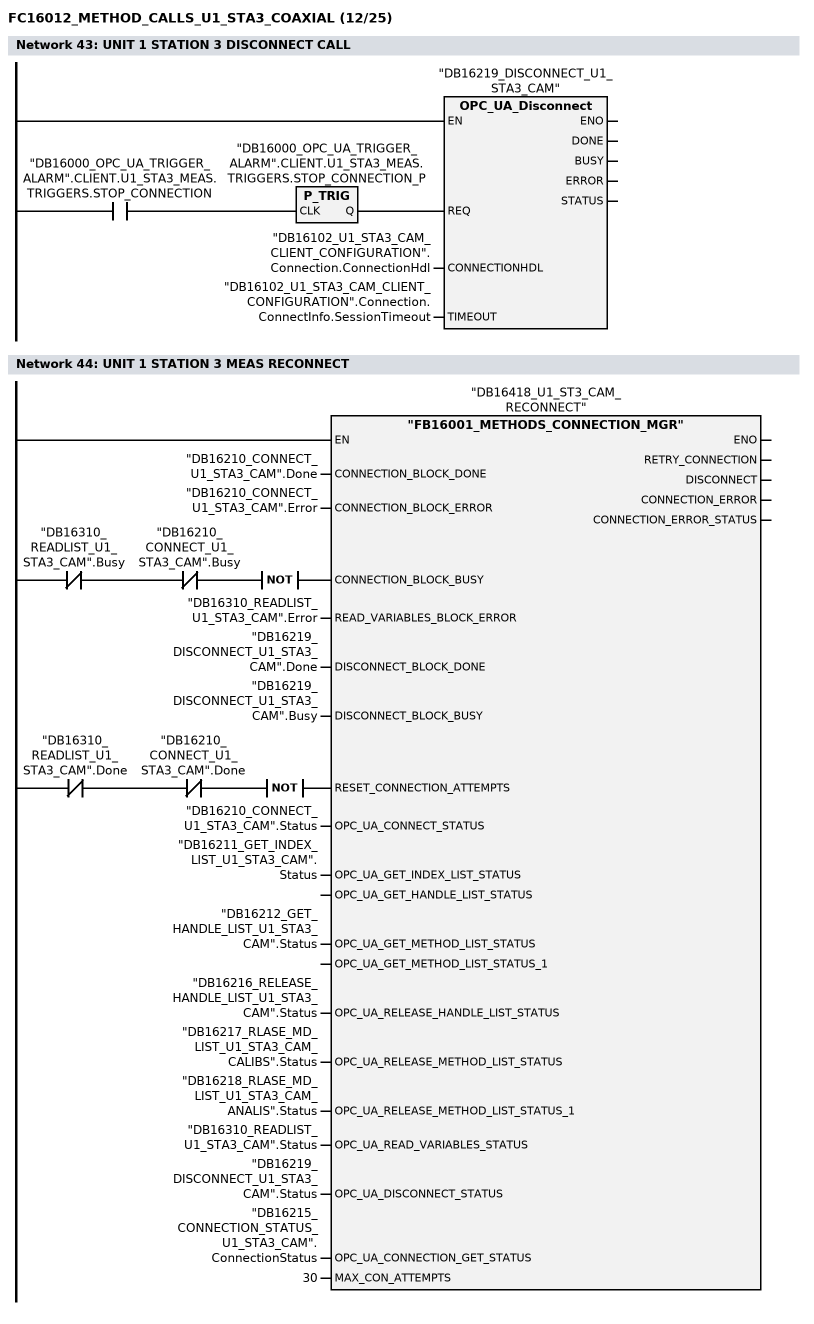
   RUNG wire#powerrail
      "DB16219_DISCONNECT_U1_STA3_CAM".OPC_UA_Disconnect(REQ := wire#w1, ConnectionHdl := "DB16102_U1_STA3_CAM_CLIENT_CONFIGURATION".Connection.ConnectionHdl, Timeout := "DB16102_U1_STA3_CAM_CLIENT_CONFIGURATION".Connection.ConnectInfo.SessionTimeout, Done =>, Busy =>, Error =>, Status =>)
   END_RUNG
   RUNG wire#powerrail
      Contact( "DB16000_OPC_UA_TRIGGER_ALARM".CLIENT.U1_STA3_MEAS.TRIGGERS.STOP_CONNECTION )
      P_Trig( "DB16000_OPC_UA_TRIGGER_ALARM".CLIENT.U1_STA3_MEAS.TRIGGERS.STOP_CONNECTION_P )
   END_RUNG wire#w1
   // the same network as SCL:
   #_w1 := "DB16000_OPC_UA_TRIGGER_ALARM".CLIENT.U1_STA3_MEAS.TRIGGERS.STOP_CONNECTION AND NOT "DB16000_OPC_UA_TRIGGER_ALARM".CLIENT.U1_STA3_MEAS.TRIGGERS.STOP_CONNECTION_P;   // rising edge
   "DB16000_OPC_UA_TRIGGER_ALARM".CLIENT.U1_STA3_MEAS.TRIGGERS.STOP_CONNECTION_P := "DB16000_OPC_UA_TRIGGER_ALARM".CLIENT.U1_STA3_MEAS.TRIGGERS.STOP_CONNECTION;
   "DB16219_DISCONNECT_U1_STA3_CAM"(REQ := #_w1,   // OPC_UA_Disconnect
                           ConnectionHdl := "DB16102_U1_STA3_CAM_CLIENT_CONFIGURATION".Connection.ConnectionHdl,
                           Timeout := "DB16102_U1_STA3_CAM_CLIENT_CONFIGURATION".Connection.ConnectInfo.SessionTimeout);
END_REGION

REGION Network 44: UNIT 1 STATION 3 MEAS RECONNECT
   RUNG wire#powerrail
      "DB16418_U1_ST3_CAM_RECONNECT"(CONNECTION_BLOCK_BUSY := wire#w1, RESET_CONNECTION_ATTEMPTS := wire#w2, CONNECTION_BLOCK_DONE := "DB16210_CONNECT_U1_STA3_CAM".Done, CONNECTION_BLOCK_ERROR := "DB16210_CONNECT_U1_STA3_CAM".Error, READ_VARIABLES_BLOCK_ERROR := "DB16310_READLIST_U1_STA3_CAM".Error, DISCONNECT_BLOCK_DONE := "DB16219_DISCONNECT_U1_STA3_CAM".Done, DISCONNECT_BLOCK_BUSY := "DB16219_DISCONNECT_U1_STA3_CAM".Busy, OPC_UA_CONNECT_STATUS := "DB16210_CONNECT_U1_STA3_CAM".Status, OPC_UA_GET_INDEX_LIST_STATUS := "DB16211_GET_INDEX_LIST_U1_STA3_CAM".Status, OPC_UA_GET_HANDLE_LIST_STATUS :=, OPC_UA_GET_METHOD_LIST_STATUS := "DB16212_GET_HANDLE_LIST_U1_STA3_CAM".Status, OPC_UA_GET_METHOD_LIST_STATUS_1 :=, OPC_UA_RELEASE_HANDLE_LIST_STATUS := "DB16216_RELEASE_HANDLE_LIST_U1_STA3_CAM".Status, OPC_UA_RELEASE_METHOD_LIST_STATUS := "DB16217_RLASE_MD_LIST_U1_STA3_CAM_CALIBS".Status, OPC_UA_RELEASE_METHOD_LIST_STATUS_1 := "DB16218_RLASE_MD_LIST_U1_STA3_CAM_ANALIS".Status, OPC_UA_READ_VARIABLES_STATUS := "DB16310_READLIST_U1_STA3_CAM".Status, OPC_UA_DISCONNECT_STATUS := "DB16219_DISCONNECT_U1_STA3_CAM".Status, OPC_UA_CONNECTION_GET_STATUS := "DB16215_CONNECTION_STATUS_U1_STA3_CAM".ConnectionStatus, MAX_CON_ATTEMPTS := 30, RETRY_CONNECTION =>, DISCONNECT =>, CONNECTION_ERROR =>, CONNECTION_ERROR_STATUS =>)
   END_RUNG
   RUNG wire#powerrail
      I_Contact( "DB16310_READLIST_U1_STA3_CAM".Busy )
      I_Contact( "DB16210_CONNECT_U1_STA3_CAM".Busy )
      Not()
   END_RUNG wire#w1
   RUNG wire#powerrail
      I_Contact( "DB16310_READLIST_U1_STA3_CAM".Done )
      I_Contact( "DB16210_CONNECT_U1_STA3_CAM".Done )
      Not()
   END_RUNG wire#w2
   // the same network as SCL:
   "DB16418_U1_ST3_CAM_RECONNECT"(CONNECTION_BLOCK_DONE := "DB16210_CONNECT_U1_STA3_CAM".Done,   // "FB16001_METHODS_CONNECTION_MGR"
                           CONNECTION_BLOCK_ERROR := "DB16210_CONNECT_U1_STA3_CAM".Error,
                           CONNECTION_BLOCK_BUSY := NOT (NOT "DB16310_READLIST_U1_STA3_CAM".Busy AND NOT "DB16210_CONNECT_U1_STA3_CAM".Busy),
                           READ_VARIABLES_BLOCK_ERROR := "DB16310_READLIST_U1_STA3_CAM".Error,
                           DISCONNECT_BLOCK_DONE := "DB16219_DISCONNECT_U1_STA3_CAM".Done,
                           DISCONNECT_BLOCK_BUSY := "DB16219_DISCONNECT_U1_STA3_CAM".Busy,
                           RESET_CONNECTION_ATTEMPTS := NOT (NOT "DB16310_READLIST_U1_STA3_CAM".Done AND NOT "DB16210_CONNECT_U1_STA3_CAM".Done),
                           OPC_UA_CONNECT_STATUS := "DB16210_CONNECT_U1_STA3_CAM".Status,
                           OPC_UA_GET_INDEX_LIST_STATUS := "DB16211_GET_INDEX_LIST_U1_STA3_CAM".Status,
                           OPC_UA_GET_METHOD_LIST_STATUS := "DB16212_GET_HANDLE_LIST_U1_STA3_CAM".Status,
                           OPC_UA_RELEASE_HANDLE_LIST_STATUS := "DB16216_RELEASE_HANDLE_LIST_U1_STA3_CAM".Status,
                           OPC_UA_RELEASE_METHOD_LIST_STATUS := "DB16217_RLASE_MD_LIST_U1_STA3_CAM_CALIBS".Status,
                           OPC_UA_RELEASE_METHOD_LIST_STATUS_1 := "DB16218_RLASE_MD_LIST_U1_STA3_CAM_ANALIS".Status,
                           OPC_UA_READ_VARIABLES_STATUS := "DB16310_READLIST_U1_STA3_CAM".Status,
                           OPC_UA_DISCONNECT_STATUS := "DB16219_DISCONNECT_U1_STA3_CAM".Status,
                           OPC_UA_CONNECTION_GET_STATUS := "DB16215_CONNECTION_STATUS_U1_STA3_CAM".ConnectionStatus,
                           MAX_CON_ATTEMPTS := 30);
END_REGION

REGION Network 45: UNIT 1 PC STATUS UPDATE
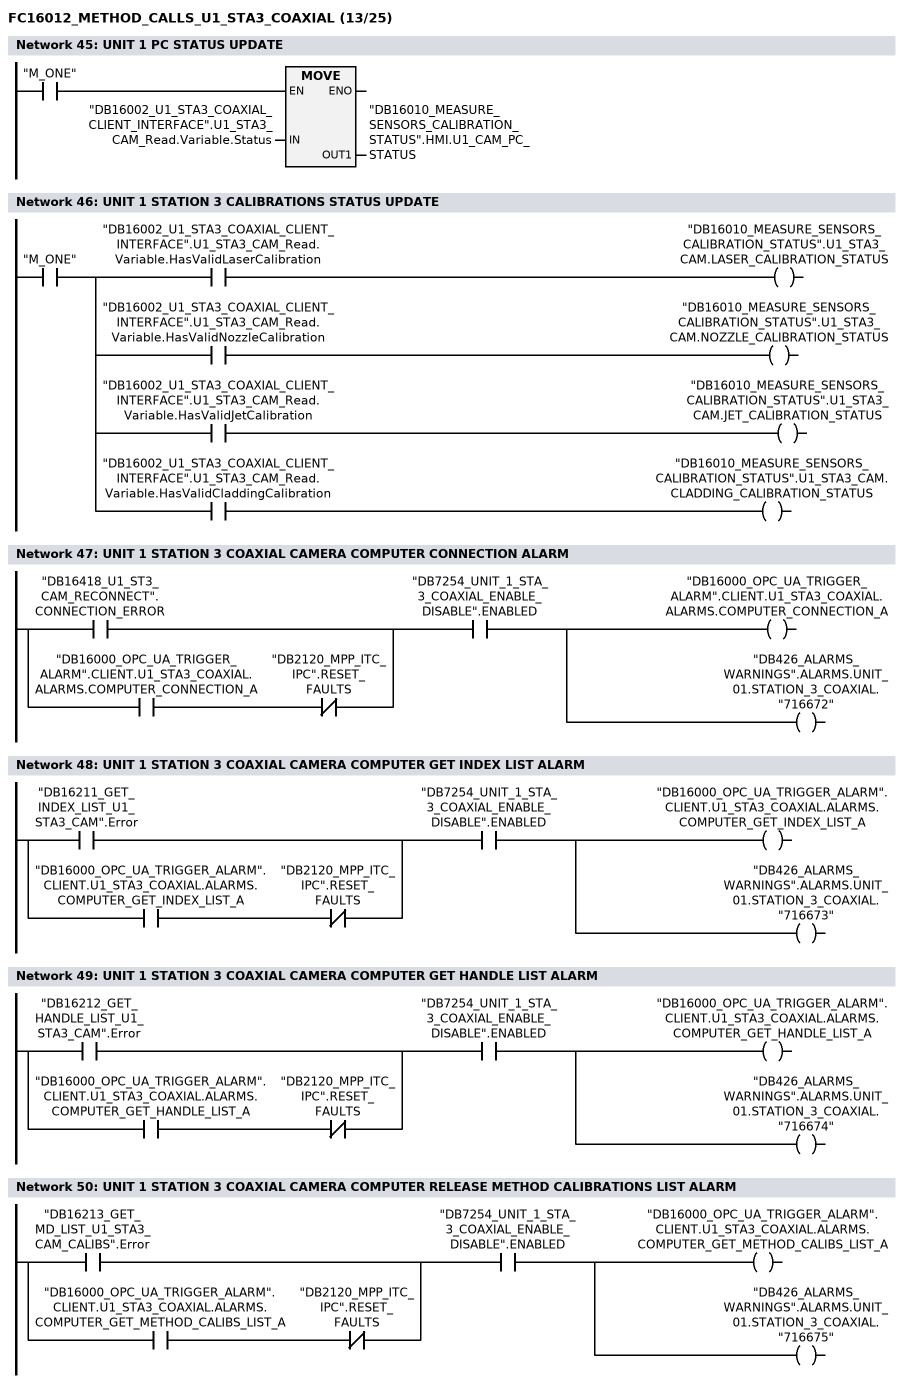
   RUNG wire#powerrail
      Contact( "M_ONE" )
      Move(in := "DB16002_U1_STA3_COAXIAL_CLIENT_INTERFACE".U1_STA3_CAM_Read.Variable.Status, out1 => "DB16010_MEASURE_SENSORS_CALIBRATION_STATUS".HMI.U1_CAM_PC_STATUS)
   END_RUNG
   // the same network as SCL:
   IF "M_ONE" THEN
       "DB16010_MEASURE_SENSORS_CALIBRATION_STATUS".HMI.U1_CAM_PC_STATUS := "DB16002_U1_STA3_COAXIAL_CLIENT_INTERFACE".U1_STA3_CAM_Read.Variable.Status;
   END_IF;
END_REGION

REGION Network 46: UNIT 1 STATION 3 CALIBRATIONS STATUS UPDATE
   RUNG wire#powerrail
      Contact( "M_ONE" )
      wire#w1
      Contact( "DB16002_U1_STA3_COAXIAL_CLIENT_INTERFACE".U1_STA3_CAM_Read.Variable.HasValidLaserCalibration )
      Coil( "DB16010_MEASURE_SENSORS_CALIBRATION_STATUS".U1_STA3_CAM.LASER_CALIBRATION_STATUS )
   END_RUNG
   RUNG wire#w1
      Contact( "DB16002_U1_STA3_COAXIAL_CLIENT_INTERFACE".U1_STA3_CAM_Read.Variable.HasValidNozzleCalibration )
      Coil( "DB16010_MEASURE_SENSORS_CALIBRATION_STATUS".U1_STA3_CAM.NOZZLE_CALIBRATION_STATUS )
   END_RUNG
   RUNG wire#w1
      Contact( "DB16002_U1_STA3_COAXIAL_CLIENT_INTERFACE".U1_STA3_CAM_Read.Variable.HasValidJetCalibration )
      Coil( "DB16010_MEASURE_SENSORS_CALIBRATION_STATUS".U1_STA3_CAM.JET_CALIBRATION_STATUS )
   END_RUNG
   RUNG wire#w1
      Contact( "DB16002_U1_STA3_COAXIAL_CLIENT_INTERFACE".U1_STA3_CAM_Read.Variable.HasValidCladdingCalibration )
      Coil( "DB16010_MEASURE_SENSORS_CALIBRATION_STATUS".U1_STA3_CAM.CLADDING_CALIBRATION_STATUS )
   END_RUNG
   // the same network as SCL:
   "DB16010_MEASURE_SENSORS_CALIBRATION_STATUS".U1_STA3_CAM.LASER_CALIBRATION_STATUS := "M_ONE" AND "DB16002_U1_STA3_COAXIAL_CLIENT_INTERFACE".U1_STA3_CAM_Read.Variable.HasValidLaserCalibration;
   "DB16010_MEASURE_SENSORS_CALIBRATION_STATUS".U1_STA3_CAM.NOZZLE_CALIBRATION_STATUS := "M_ONE" AND "DB16002_U1_STA3_COAXIAL_CLIENT_INTERFACE".U1_STA3_CAM_Read.Variable.HasValidNozzleCalibration;
   "DB16010_MEASURE_SENSORS_CALIBRATION_STATUS".U1_STA3_CAM.JET_CALIBRATION_STATUS := "M_ONE" AND "DB16002_U1_STA3_COAXIAL_CLIENT_INTERFACE".U1_STA3_CAM_Read.Variable.HasValidJetCalibration;
   "DB16010_MEASURE_SENSORS_CALIBRATION_STATUS".U1_STA3_CAM.CLADDING_CALIBRATION_STATUS := "M_ONE" AND "DB16002_U1_STA3_COAXIAL_CLIENT_INTERFACE".U1_STA3_CAM_Read.Variable.HasValidCladdingCalibration;
END_REGION

REGION Network 47: UNIT 1 STATION 3 COAXIAL CAMERA COMPUTER CONNECTION ALARM
   RUNG wire#powerrail
      Contact( "DB16418_U1_ST3_CAM_RECONNECT".CONNECTION_ERROR )
      wire#w1
      Contact( "DB7254_UNIT_1_STA_3_COAXIAL_ENABLE_DISABLE".ENABLED )
      wire#w2
      Coil( "DB16000_OPC_UA_TRIGGER_ALARM".CLIENT.U1_STA3_COAXIAL.ALARMS.COMPUTER_CONNECTION_A )
   END_RUNG
   RUNG wire#powerrail
      Contact( "DB16000_OPC_UA_TRIGGER_ALARM".CLIENT.U1_STA3_COAXIAL.ALARMS.COMPUTER_CONNECTION_A )
      I_Contact( "DB2120_MPP_ITC_IPC".RESET_FAULTS )
   END_RUNG wire#w1
   RUNG wire#w2
      Coil( "DB426_ALARMS_WARNINGS".ALARMS.UNIT_01.STATION_3_COAXIAL."716672" )
   END_RUNG
   // the same network as SCL:
   "DB16000_OPC_UA_TRIGGER_ALARM".CLIENT.U1_STA3_COAXIAL.ALARMS.COMPUTER_CONNECTION_A := ("DB16418_U1_ST3_CAM_RECONNECT".CONNECTION_ERROR OR ("DB16000_OPC_UA_TRIGGER_ALARM".CLIENT.U1_STA3_COAXIAL.ALARMS.COMPUTER_CONNECTION_A AND NOT "DB2120_MPP_ITC_IPC".RESET_FAULTS)) AND "DB7254_UNIT_1_STA_3_COAXIAL_ENABLE_DISABLE".ENABLED;
   "DB426_ALARMS_WARNINGS".ALARMS.UNIT_01.STATION_3_COAXIAL."716672" := "DB16000_OPC_UA_TRIGGER_ALARM".CLIENT.U1_STA3_COAXIAL.ALARMS.COMPUTER_CONNECTION_A;
END_REGION

REGION Network 48: UNIT 1 STATION 3 COAXIAL CAMERA COMPUTER GET INDEX LIST ALARM
   RUNG wire#powerrail
      Contact( "DB16211_GET_INDEX_LIST_U1_STA3_CAM".Error )
      wire#w1
      Contact( "DB7254_UNIT_1_STA_3_COAXIAL_ENABLE_DISABLE".ENABLED )
      wire#w2
      Coil( "DB16000_OPC_UA_TRIGGER_ALARM".CLIENT.U1_STA3_COAXIAL.ALARMS.COMPUTER_GET_INDEX_LIST_A )
   END_RUNG
   RUNG wire#powerrail
      Contact( "DB16000_OPC_UA_TRIGGER_ALARM".CLIENT.U1_STA3_COAXIAL.ALARMS.COMPUTER_GET_INDEX_LIST_A )
      I_Contact( "DB2120_MPP_ITC_IPC".RESET_FAULTS )
   END_RUNG wire#w1
   RUNG wire#w2
      Coil( "DB426_ALARMS_WARNINGS".ALARMS.UNIT_01.STATION_3_COAXIAL."716673" )
   END_RUNG
   // the same network as SCL:
   "DB16000_OPC_UA_TRIGGER_ALARM".CLIENT.U1_STA3_COAXIAL.ALARMS.COMPUTER_GET_INDEX_LIST_A := ("DB16211_GET_INDEX_LIST_U1_STA3_CAM".Error OR ("DB16000_OPC_UA_TRIGGER_ALARM".CLIENT.U1_STA3_COAXIAL.ALARMS.COMPUTER_GET_INDEX_LIST_A AND NOT "DB2120_MPP_ITC_IPC".RESET_FAULTS)) AND "DB7254_UNIT_1_STA_3_COAXIAL_ENABLE_DISABLE".ENABLED;
   "DB426_ALARMS_WARNINGS".ALARMS.UNIT_01.STATION_3_COAXIAL."716673" := "DB16000_OPC_UA_TRIGGER_ALARM".CLIENT.U1_STA3_COAXIAL.ALARMS.COMPUTER_GET_INDEX_LIST_A;
END_REGION

REGION Network 49: UNIT 1 STATION 3 COAXIAL CAMERA COMPUTER GET HANDLE LIST ALARM
   RUNG wire#powerrail
      Contact( "DB16212_GET_HANDLE_LIST_U1_STA3_CAM".Error )
      wire#w1
      Contact( "DB7254_UNIT_1_STA_3_COAXIAL_ENABLE_DISABLE".ENABLED )
      wire#w2
      Coil( "DB16000_OPC_UA_TRIGGER_ALARM".CLIENT.U1_STA3_COAXIAL.ALARMS.COMPUTER_GET_HANDLE_LIST_A )
   END_RUNG
   RUNG wire#powerrail
      Contact( "DB16000_OPC_UA_TRIGGER_ALARM".CLIENT.U1_STA3_COAXIAL.ALARMS.COMPUTER_GET_HANDLE_LIST_A )
      I_Contact( "DB2120_MPP_ITC_IPC".RESET_FAULTS )
   END_RUNG wire#w1
   RUNG wire#w2
      Coil( "DB426_ALARMS_WARNINGS".ALARMS.UNIT_01.STATION_3_COAXIAL."716674" )
   END_RUNG
   // the same network as SCL:
   "DB16000_OPC_UA_TRIGGER_ALARM".CLIENT.U1_STA3_COAXIAL.ALARMS.COMPUTER_GET_HANDLE_LIST_A := ("DB16212_GET_HANDLE_LIST_U1_STA3_CAM".Error OR ("DB16000_OPC_UA_TRIGGER_ALARM".CLIENT.U1_STA3_COAXIAL.ALARMS.COMPUTER_GET_HANDLE_LIST_A AND NOT "DB2120_MPP_ITC_IPC".RESET_FAULTS)) AND "DB7254_UNIT_1_STA_3_COAXIAL_ENABLE_DISABLE".ENABLED;
   "DB426_ALARMS_WARNINGS".ALARMS.UNIT_01.STATION_3_COAXIAL."716674" := "DB16000_OPC_UA_TRIGGER_ALARM".CLIENT.U1_STA3_COAXIAL.ALARMS.COMPUTER_GET_HANDLE_LIST_A;
END_REGION

REGION Network 50: UNIT 1 STATION 3 COAXIAL CAMERA COMPUTER RELEASE METHOD CALIBRATIONS LIST ALARM
   RUNG wire#powerrail
      Contact( "DB16213_GET_MD_LIST_U1_STA3_CAM_CALIBS".Error )
      wire#w1
      Contact( "DB7254_UNIT_1_STA_3_COAXIAL_ENABLE_DISABLE".ENABLED )
      wire#w2
      Coil( "DB16000_OPC_UA_TRIGGER_ALARM".CLIENT.U1_STA3_COAXIAL.ALARMS.COMPUTER_GET_METHOD_CALIBS_LIST_A )
   END_RUNG
   RUNG wire#powerrail
      Contact( "DB16000_OPC_UA_TRIGGER_ALARM".CLIENT.U1_STA3_COAXIAL.ALARMS.COMPUTER_GET_METHOD_CALIBS_LIST_A )
      I_Contact( "DB2120_MPP_ITC_IPC".RESET_FAULTS )
   END_RUNG wire#w1
   RUNG wire#w2
      Coil( "DB426_ALARMS_WARNINGS".ALARMS.UNIT_01.STATION_3_COAXIAL."716675" )
   END_RUNG
   // the same network as SCL:
   "DB16000_OPC_UA_TRIGGER_ALARM".CLIENT.U1_STA3_COAXIAL.ALARMS.COMPUTER_GET_METHOD_CALIBS_LIST_A := ("DB16213_GET_MD_LIST_U1_STA3_CAM_CALIBS".Error OR ("DB16000_OPC_UA_TRIGGER_ALARM".CLIENT.U1_STA3_COAXIAL.ALARMS.COMPUTER_GET_METHOD_CALIBS_LIST_A AND NOT "DB2120_MPP_ITC_IPC".RESET_FAULTS)) AND "DB7254_UNIT_1_STA_3_COAXIAL_ENABLE_DISABLE".ENABLED;
   "DB426_ALARMS_WARNINGS".ALARMS.UNIT_01.STATION_3_COAXIAL."716675" := "DB16000_OPC_UA_TRIGGER_ALARM".CLIENT.U1_STA3_COAXIAL.ALARMS.COMPUTER_GET_METHOD_CALIBS_LIST_A;
END_REGION

REGION Network 51: UNIT 1 STATION 3 COAXIAL CAMERA COMPUTER RELEASE METHOD ANALISIS LIST ALARM
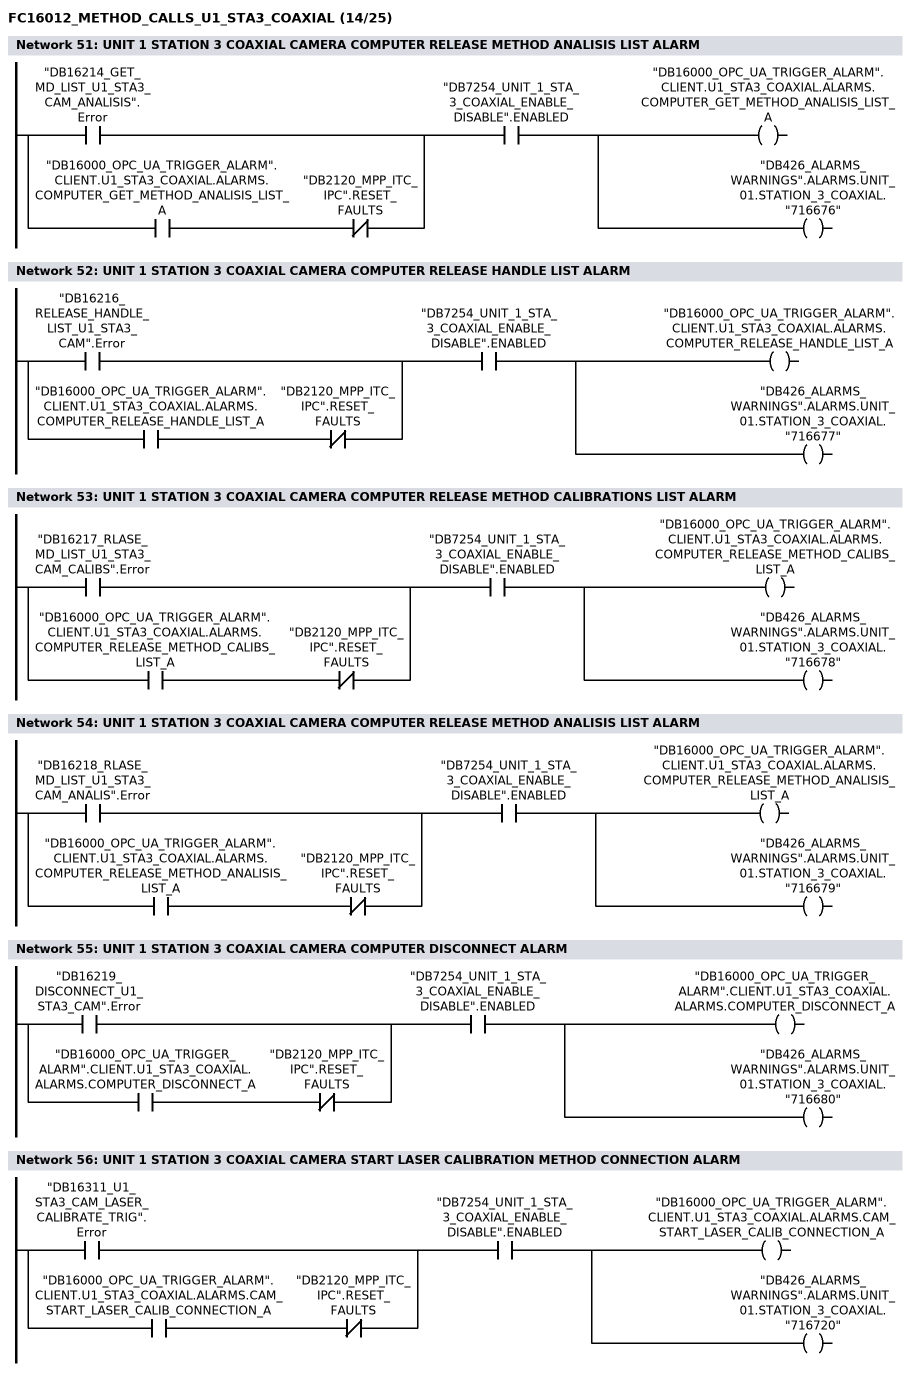
   RUNG wire#powerrail
      Contact( "DB16214_GET_MD_LIST_U1_STA3_CAM_ANALISIS".Error )
      wire#w1
      Contact( "DB7254_UNIT_1_STA_3_COAXIAL_ENABLE_DISABLE".ENABLED )
      wire#w2
      Coil( "DB16000_OPC_UA_TRIGGER_ALARM".CLIENT.U1_STA3_COAXIAL.ALARMS.COMPUTER_GET_METHOD_ANALISIS_LIST_A )
   END_RUNG
   RUNG wire#powerrail
      Contact( "DB16000_OPC_UA_TRIGGER_ALARM".CLIENT.U1_STA3_COAXIAL.ALARMS.COMPUTER_GET_METHOD_ANALISIS_LIST_A )
      I_Contact( "DB2120_MPP_ITC_IPC".RESET_FAULTS )
   END_RUNG wire#w1
   RUNG wire#w2
      Coil( "DB426_ALARMS_WARNINGS".ALARMS.UNIT_01.STATION_3_COAXIAL."716676" )
   END_RUNG
   // the same network as SCL:
   "DB16000_OPC_UA_TRIGGER_ALARM".CLIENT.U1_STA3_COAXIAL.ALARMS.COMPUTER_GET_METHOD_ANALISIS_LIST_A := ("DB16214_GET_MD_LIST_U1_STA3_CAM_ANALISIS".Error OR ("DB16000_OPC_UA_TRIGGER_ALARM".CLIENT.U1_STA3_COAXIAL.ALARMS.COMPUTER_GET_METHOD_ANALISIS_LIST_A AND NOT "DB2120_MPP_ITC_IPC".RESET_FAULTS)) AND "DB7254_UNIT_1_STA_3_COAXIAL_ENABLE_DISABLE".ENABLED;
   "DB426_ALARMS_WARNINGS".ALARMS.UNIT_01.STATION_3_COAXIAL."716676" := "DB16000_OPC_UA_TRIGGER_ALARM".CLIENT.U1_STA3_COAXIAL.ALARMS.COMPUTER_GET_METHOD_ANALISIS_LIST_A;
END_REGION

REGION Network 52: UNIT 1 STATION 3 COAXIAL CAMERA COMPUTER RELEASE HANDLE LIST ALARM
   RUNG wire#powerrail
      Contact( "DB16216_RELEASE_HANDLE_LIST_U1_STA3_CAM".Error )
      wire#w1
      Contact( "DB7254_UNIT_1_STA_3_COAXIAL_ENABLE_DISABLE".ENABLED )
      wire#w2
      Coil( "DB16000_OPC_UA_TRIGGER_ALARM".CLIENT.U1_STA3_COAXIAL.ALARMS.COMPUTER_RELEASE_HANDLE_LIST_A )
   END_RUNG
   RUNG wire#powerrail
      Contact( "DB16000_OPC_UA_TRIGGER_ALARM".CLIENT.U1_STA3_COAXIAL.ALARMS.COMPUTER_RELEASE_HANDLE_LIST_A )
      I_Contact( "DB2120_MPP_ITC_IPC".RESET_FAULTS )
   END_RUNG wire#w1
   RUNG wire#w2
      Coil( "DB426_ALARMS_WARNINGS".ALARMS.UNIT_01.STATION_3_COAXIAL."716677" )
   END_RUNG
   // the same network as SCL:
   "DB16000_OPC_UA_TRIGGER_ALARM".CLIENT.U1_STA3_COAXIAL.ALARMS.COMPUTER_RELEASE_HANDLE_LIST_A := ("DB16216_RELEASE_HANDLE_LIST_U1_STA3_CAM".Error OR ("DB16000_OPC_UA_TRIGGER_ALARM".CLIENT.U1_STA3_COAXIAL.ALARMS.COMPUTER_RELEASE_HANDLE_LIST_A AND NOT "DB2120_MPP_ITC_IPC".RESET_FAULTS)) AND "DB7254_UNIT_1_STA_3_COAXIAL_ENABLE_DISABLE".ENABLED;
   "DB426_ALARMS_WARNINGS".ALARMS.UNIT_01.STATION_3_COAXIAL."716677" := "DB16000_OPC_UA_TRIGGER_ALARM".CLIENT.U1_STA3_COAXIAL.ALARMS.COMPUTER_RELEASE_HANDLE_LIST_A;
END_REGION

REGION Network 53: UNIT 1 STATION 3 COAXIAL CAMERA COMPUTER RELEASE METHOD CALIBRATIONS LIST ALARM
   RUNG wire#powerrail
      Contact( "DB16217_RLASE_MD_LIST_U1_STA3_CAM_CALIBS".Error )
      wire#w1
      Contact( "DB7254_UNIT_1_STA_3_COAXIAL_ENABLE_DISABLE".ENABLED )
      wire#w2
      Coil( "DB16000_OPC_UA_TRIGGER_ALARM".CLIENT.U1_STA3_COAXIAL.ALARMS.COMPUTER_RELEASE_METHOD_CALIBS_LIST_A )
   END_RUNG
   RUNG wire#powerrail
      Contact( "DB16000_OPC_UA_TRIGGER_ALARM".CLIENT.U1_STA3_COAXIAL.ALARMS.COMPUTER_RELEASE_METHOD_CALIBS_LIST_A )
      I_Contact( "DB2120_MPP_ITC_IPC".RESET_FAULTS )
   END_RUNG wire#w1
   RUNG wire#w2
      Coil( "DB426_ALARMS_WARNINGS".ALARMS.UNIT_01.STATION_3_COAXIAL."716678" )
   END_RUNG
   // the same network as SCL:
   "DB16000_OPC_UA_TRIGGER_ALARM".CLIENT.U1_STA3_COAXIAL.ALARMS.COMPUTER_RELEASE_METHOD_CALIBS_LIST_A := ("DB16217_RLASE_MD_LIST_U1_STA3_CAM_CALIBS".Error OR ("DB16000_OPC_UA_TRIGGER_ALARM".CLIENT.U1_STA3_COAXIAL.ALARMS.COMPUTER_RELEASE_METHOD_CALIBS_LIST_A AND NOT "DB2120_MPP_ITC_IPC".RESET_FAULTS)) AND "DB7254_UNIT_1_STA_3_COAXIAL_ENABLE_DISABLE".ENABLED;
   "DB426_ALARMS_WARNINGS".ALARMS.UNIT_01.STATION_3_COAXIAL."716678" := "DB16000_OPC_UA_TRIGGER_ALARM".CLIENT.U1_STA3_COAXIAL.ALARMS.COMPUTER_RELEASE_METHOD_CALIBS_LIST_A;
END_REGION

REGION Network 54: UNIT 1 STATION 3 COAXIAL CAMERA COMPUTER RELEASE METHOD ANALISIS LIST ALARM
   RUNG wire#powerrail
      Contact( "DB16218_RLASE_MD_LIST_U1_STA3_CAM_ANALIS".Error )
      wire#w1
      Contact( "DB7254_UNIT_1_STA_3_COAXIAL_ENABLE_DISABLE".ENABLED )
      wire#w2
      Coil( "DB16000_OPC_UA_TRIGGER_ALARM".CLIENT.U1_STA3_COAXIAL.ALARMS.COMPUTER_RELEASE_METHOD_ANALISIS_LIST_A )
   END_RUNG
   RUNG wire#powerrail
      Contact( "DB16000_OPC_UA_TRIGGER_ALARM".CLIENT.U1_STA3_COAXIAL.ALARMS.COMPUTER_RELEASE_METHOD_ANALISIS_LIST_A )
      I_Contact( "DB2120_MPP_ITC_IPC".RESET_FAULTS )
   END_RUNG wire#w1
   RUNG wire#w2
      Coil( "DB426_ALARMS_WARNINGS".ALARMS.UNIT_01.STATION_3_COAXIAL."716679" )
   END_RUNG
   // the same network as SCL:
   "DB16000_OPC_UA_TRIGGER_ALARM".CLIENT.U1_STA3_COAXIAL.ALARMS.COMPUTER_RELEASE_METHOD_ANALISIS_LIST_A := ("DB16218_RLASE_MD_LIST_U1_STA3_CAM_ANALIS".Error OR ("DB16000_OPC_UA_TRIGGER_ALARM".CLIENT.U1_STA3_COAXIAL.ALARMS.COMPUTER_RELEASE_METHOD_ANALISIS_LIST_A AND NOT "DB2120_MPP_ITC_IPC".RESET_FAULTS)) AND "DB7254_UNIT_1_STA_3_COAXIAL_ENABLE_DISABLE".ENABLED;
   "DB426_ALARMS_WARNINGS".ALARMS.UNIT_01.STATION_3_COAXIAL."716679" := "DB16000_OPC_UA_TRIGGER_ALARM".CLIENT.U1_STA3_COAXIAL.ALARMS.COMPUTER_RELEASE_METHOD_ANALISIS_LIST_A;
END_REGION

REGION Network 55: UNIT 1 STATION 3 COAXIAL CAMERA COMPUTER DISCONNECT ALARM
   RUNG wire#powerrail
      Contact( "DB16219_DISCONNECT_U1_STA3_CAM".Error )
      wire#w1
      Contact( "DB7254_UNIT_1_STA_3_COAXIAL_ENABLE_DISABLE".ENABLED )
      wire#w2
      Coil( "DB16000_OPC_UA_TRIGGER_ALARM".CLIENT.U1_STA3_COAXIAL.ALARMS.COMPUTER_DISCONNECT_A )
   END_RUNG
   RUNG wire#powerrail
      Contact( "DB16000_OPC_UA_TRIGGER_ALARM".CLIENT.U1_STA3_COAXIAL.ALARMS.COMPUTER_DISCONNECT_A )
      I_Contact( "DB2120_MPP_ITC_IPC".RESET_FAULTS )
   END_RUNG wire#w1
   RUNG wire#w2
      Coil( "DB426_ALARMS_WARNINGS".ALARMS.UNIT_01.STATION_3_COAXIAL."716680" )
   END_RUNG
   // the same network as SCL:
   "DB16000_OPC_UA_TRIGGER_ALARM".CLIENT.U1_STA3_COAXIAL.ALARMS.COMPUTER_DISCONNECT_A := ("DB16219_DISCONNECT_U1_STA3_CAM".Error OR ("DB16000_OPC_UA_TRIGGER_ALARM".CLIENT.U1_STA3_COAXIAL.ALARMS.COMPUTER_DISCONNECT_A AND NOT "DB2120_MPP_ITC_IPC".RESET_FAULTS)) AND "DB7254_UNIT_1_STA_3_COAXIAL_ENABLE_DISABLE".ENABLED;
   "DB426_ALARMS_WARNINGS".ALARMS.UNIT_01.STATION_3_COAXIAL."716680" := "DB16000_OPC_UA_TRIGGER_ALARM".CLIENT.U1_STA3_COAXIAL.ALARMS.COMPUTER_DISCONNECT_A;
END_REGION

REGION Network 56: UNIT 1 STATION 3 COAXIAL CAMERA START LASER CALIBRATION METHOD CONNECTION ALARM
   RUNG wire#powerrail
      Contact( "DB16311_U1_STA3_CAM_LASER_CALIBRATE_TRIG".Error )
      wire#w1
      Contact( "DB7254_UNIT_1_STA_3_COAXIAL_ENABLE_DISABLE".ENABLED )
      wire#w2
      Coil( "DB16000_OPC_UA_TRIGGER_ALARM".CLIENT.U1_STA3_COAXIAL.ALARMS.CAM_START_LASER_CALIB_CONNECTION_A )
   END_RUNG
   RUNG wire#powerrail
      Contact( "DB16000_OPC_UA_TRIGGER_ALARM".CLIENT.U1_STA3_COAXIAL.ALARMS.CAM_START_LASER_CALIB_CONNECTION_A )
      I_Contact( "DB2120_MPP_ITC_IPC".RESET_FAULTS )
   END_RUNG wire#w1
   RUNG wire#w2
      Coil( "DB426_ALARMS_WARNINGS".ALARMS.UNIT_01.STATION_3_COAXIAL."716720" )
   END_RUNG
   // the same network as SCL:
   "DB16000_OPC_UA_TRIGGER_ALARM".CLIENT.U1_STA3_COAXIAL.ALARMS.CAM_START_LASER_CALIB_CONNECTION_A := ("DB16311_U1_STA3_CAM_LASER_CALIBRATE_TRIG".Error OR ("DB16000_OPC_UA_TRIGGER_ALARM".CLIENT.U1_STA3_COAXIAL.ALARMS.CAM_START_LASER_CALIB_CONNECTION_A AND NOT "DB2120_MPP_ITC_IPC".RESET_FAULTS)) AND "DB7254_UNIT_1_STA_3_COAXIAL_ENABLE_DISABLE".ENABLED;
   "DB426_ALARMS_WARNINGS".ALARMS.UNIT_01.STATION_3_COAXIAL."716720" := "DB16000_OPC_UA_TRIGGER_ALARM".CLIENT.U1_STA3_COAXIAL.ALARMS.CAM_START_LASER_CALIB_CONNECTION_A;
END_REGION

REGION Network 57: UNIT 1 STATION 3 COAXIAL CAMERA START LASER CALIBRATION METHOD WORKING OR BLOCKED ALARM
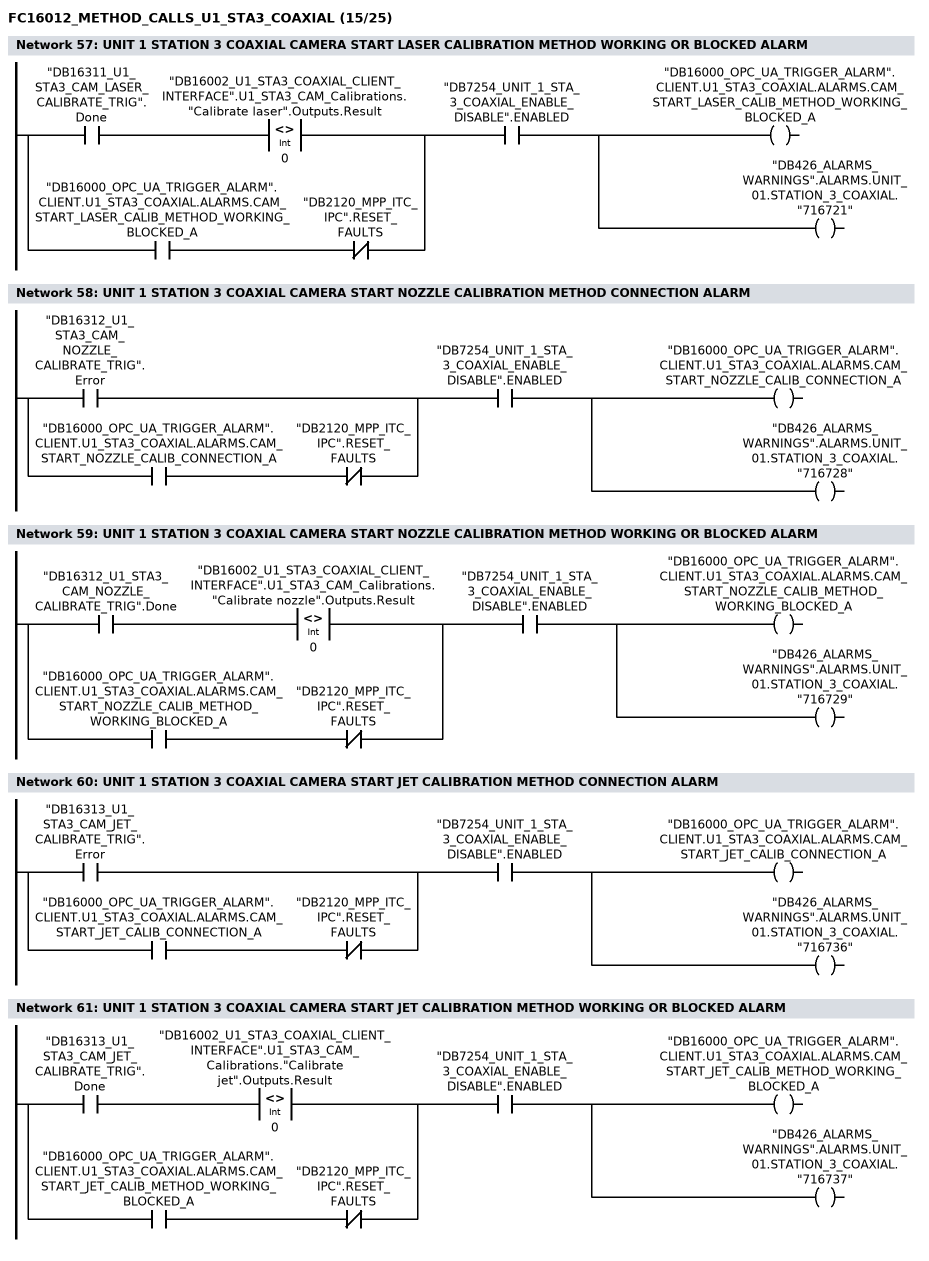
   RUNG wire#powerrail
      Contact( "DB16311_U1_STA3_CAM_LASER_CALIBRATE_TRIG".Done )
      { S7_Templates := "SrcType := Int" } NE_Contact(in1 := "DB16002_U1_STA3_COAXIAL_CLIENT_INTERFACE".U1_STA3_CAM_Calibrations."Calibrate laser".Outputs.Result, in2 := 0)
      wire#w1
      Contact( "DB7254_UNIT_1_STA_3_COAXIAL_ENABLE_DISABLE".ENABLED )
      wire#w2
      Coil( "DB16000_OPC_UA_TRIGGER_ALARM".CLIENT.U1_STA3_COAXIAL.ALARMS.CAM_START_LASER_CALIB_METHOD_WORKING_BLOCKED_A )
   END_RUNG
   RUNG wire#powerrail
      Contact( "DB16000_OPC_UA_TRIGGER_ALARM".CLIENT.U1_STA3_COAXIAL.ALARMS.CAM_START_LASER_CALIB_METHOD_WORKING_BLOCKED_A )
      I_Contact( "DB2120_MPP_ITC_IPC".RESET_FAULTS )
   END_RUNG wire#w1
   RUNG wire#w2
      Coil( "DB426_ALARMS_WARNINGS".ALARMS.UNIT_01.STATION_3_COAXIAL."716721" )
   END_RUNG
   // the same network as SCL:
   "DB16000_OPC_UA_TRIGGER_ALARM".CLIENT.U1_STA3_COAXIAL.ALARMS.CAM_START_LASER_CALIB_METHOD_WORKING_BLOCKED_A := (("DB16311_U1_STA3_CAM_LASER_CALIBRATE_TRIG".Done AND ("DB16002_U1_STA3_COAXIAL_CLIENT_INTERFACE".U1_STA3_CAM_Calibrations."Calibrate laser".Outputs.Result <> 0)) OR ("DB16000_OPC_UA_TRIGGER_ALARM".CLIENT.U1_STA3_COAXIAL.ALARMS.CAM_START_LASER_CALIB_METHOD_WORKING_BLOCKED_A AND NOT "DB2120_MPP_ITC_IPC".RESET_FAULTS)) AND "DB7254_UNIT_1_STA_3_COAXIAL_ENABLE_DISABLE".ENABLED;
   "DB426_ALARMS_WARNINGS".ALARMS.UNIT_01.STATION_3_COAXIAL."716721" := "DB16000_OPC_UA_TRIGGER_ALARM".CLIENT.U1_STA3_COAXIAL.ALARMS.CAM_START_LASER_CALIB_METHOD_WORKING_BLOCKED_A;
END_REGION

REGION Network 58: UNIT 1 STATION 3 COAXIAL CAMERA START NOZZLE CALIBRATION METHOD CONNECTION ALARM
   RUNG wire#powerrail
      Contact( "DB16312_U1_STA3_CAM_NOZZLE_CALIBRATE_TRIG".Error )
      wire#w1
      Contact( "DB7254_UNIT_1_STA_3_COAXIAL_ENABLE_DISABLE".ENABLED )
      wire#w2
      Coil( "DB16000_OPC_UA_TRIGGER_ALARM".CLIENT.U1_STA3_COAXIAL.ALARMS.CAM_START_NOZZLE_CALIB_CONNECTION_A )
   END_RUNG
   RUNG wire#powerrail
      Contact( "DB16000_OPC_UA_TRIGGER_ALARM".CLIENT.U1_STA3_COAXIAL.ALARMS.CAM_START_NOZZLE_CALIB_CONNECTION_A )
      I_Contact( "DB2120_MPP_ITC_IPC".RESET_FAULTS )
   END_RUNG wire#w1
   RUNG wire#w2
      Coil( "DB426_ALARMS_WARNINGS".ALARMS.UNIT_01.STATION_3_COAXIAL."716728" )
   END_RUNG
   // the same network as SCL:
   "DB16000_OPC_UA_TRIGGER_ALARM".CLIENT.U1_STA3_COAXIAL.ALARMS.CAM_START_NOZZLE_CALIB_CONNECTION_A := ("DB16312_U1_STA3_CAM_NOZZLE_CALIBRATE_TRIG".Error OR ("DB16000_OPC_UA_TRIGGER_ALARM".CLIENT.U1_STA3_COAXIAL.ALARMS.CAM_START_NOZZLE_CALIB_CONNECTION_A AND NOT "DB2120_MPP_ITC_IPC".RESET_FAULTS)) AND "DB7254_UNIT_1_STA_3_COAXIAL_ENABLE_DISABLE".ENABLED;
   "DB426_ALARMS_WARNINGS".ALARMS.UNIT_01.STATION_3_COAXIAL."716728" := "DB16000_OPC_UA_TRIGGER_ALARM".CLIENT.U1_STA3_COAXIAL.ALARMS.CAM_START_NOZZLE_CALIB_CONNECTION_A;
END_REGION

REGION Network 59: UNIT 1 STATION 3 COAXIAL CAMERA START NOZZLE CALIBRATION METHOD WORKING OR BLOCKED ALARM
   RUNG wire#powerrail
      Contact( "DB16312_U1_STA3_CAM_NOZZLE_CALIBRATE_TRIG".Done )
      { S7_Templates := "SrcType := Int" } NE_Contact(in1 := "DB16002_U1_STA3_COAXIAL_CLIENT_INTERFACE".U1_STA3_CAM_Calibrations."Calibrate nozzle".Outputs.Result, in2 := 0)
      wire#w1
      Contact( "DB7254_UNIT_1_STA_3_COAXIAL_ENABLE_DISABLE".ENABLED )
      wire#w2
      Coil( "DB16000_OPC_UA_TRIGGER_ALARM".CLIENT.U1_STA3_COAXIAL.ALARMS.CAM_START_NOZZLE_CALIB_METHOD_WORKING_BLOCKED_A )
   END_RUNG
   RUNG wire#powerrail
      Contact( "DB16000_OPC_UA_TRIGGER_ALARM".CLIENT.U1_STA3_COAXIAL.ALARMS.CAM_START_NOZZLE_CALIB_METHOD_WORKING_BLOCKED_A )
      I_Contact( "DB2120_MPP_ITC_IPC".RESET_FAULTS )
   END_RUNG wire#w1
   RUNG wire#w2
      Coil( "DB426_ALARMS_WARNINGS".ALARMS.UNIT_01.STATION_3_COAXIAL."716729" )
   END_RUNG
   // the same network as SCL:
   "DB16000_OPC_UA_TRIGGER_ALARM".CLIENT.U1_STA3_COAXIAL.ALARMS.CAM_START_NOZZLE_CALIB_METHOD_WORKING_BLOCKED_A := (("DB16312_U1_STA3_CAM_NOZZLE_CALIBRATE_TRIG".Done AND ("DB16002_U1_STA3_COAXIAL_CLIENT_INTERFACE".U1_STA3_CAM_Calibrations."Calibrate nozzle".Outputs.Result <> 0)) OR ("DB16000_OPC_UA_TRIGGER_ALARM".CLIENT.U1_STA3_COAXIAL.ALARMS.CAM_START_NOZZLE_CALIB_METHOD_WORKING_BLOCKED_A AND NOT "DB2120_MPP_ITC_IPC".RESET_FAULTS)) AND "DB7254_UNIT_1_STA_3_COAXIAL_ENABLE_DISABLE".ENABLED;
   "DB426_ALARMS_WARNINGS".ALARMS.UNIT_01.STATION_3_COAXIAL."716729" := "DB16000_OPC_UA_TRIGGER_ALARM".CLIENT.U1_STA3_COAXIAL.ALARMS.CAM_START_NOZZLE_CALIB_METHOD_WORKING_BLOCKED_A;
END_REGION

REGION Network 60: UNIT 1 STATION 3 COAXIAL CAMERA START JET CALIBRATION METHOD CONNECTION ALARM
   RUNG wire#powerrail
      Contact( "DB16313_U1_STA3_CAM_JET_CALIBRATE_TRIG".Error )
      wire#w1
      Contact( "DB7254_UNIT_1_STA_3_COAXIAL_ENABLE_DISABLE".ENABLED )
      wire#w2
      Coil( "DB16000_OPC_UA_TRIGGER_ALARM".CLIENT.U1_STA3_COAXIAL.ALARMS.CAM_START_JET_CALIB_CONNECTION_A )
   END_RUNG
   RUNG wire#powerrail
      Contact( "DB16000_OPC_UA_TRIGGER_ALARM".CLIENT.U1_STA3_COAXIAL.ALARMS.CAM_START_JET_CALIB_CONNECTION_A )
      I_Contact( "DB2120_MPP_ITC_IPC".RESET_FAULTS )
   END_RUNG wire#w1
   RUNG wire#w2
      Coil( "DB426_ALARMS_WARNINGS".ALARMS.UNIT_01.STATION_3_COAXIAL."716736" )
   END_RUNG
   // the same network as SCL:
   "DB16000_OPC_UA_TRIGGER_ALARM".CLIENT.U1_STA3_COAXIAL.ALARMS.CAM_START_JET_CALIB_CONNECTION_A := ("DB16313_U1_STA3_CAM_JET_CALIBRATE_TRIG".Error OR ("DB16000_OPC_UA_TRIGGER_ALARM".CLIENT.U1_STA3_COAXIAL.ALARMS.CAM_START_JET_CALIB_CONNECTION_A AND NOT "DB2120_MPP_ITC_IPC".RESET_FAULTS)) AND "DB7254_UNIT_1_STA_3_COAXIAL_ENABLE_DISABLE".ENABLED;
   "DB426_ALARMS_WARNINGS".ALARMS.UNIT_01.STATION_3_COAXIAL."716736" := "DB16000_OPC_UA_TRIGGER_ALARM".CLIENT.U1_STA3_COAXIAL.ALARMS.CAM_START_JET_CALIB_CONNECTION_A;
END_REGION

REGION Network 61: UNIT 1 STATION 3 COAXIAL CAMERA START JET CALIBRATION METHOD WORKING OR BLOCKED ALARM
   RUNG wire#powerrail
      Contact( "DB16313_U1_STA3_CAM_JET_CALIBRATE_TRIG".Done )
      { S7_Templates := "SrcType := Int" } NE_Contact(in1 := "DB16002_U1_STA3_COAXIAL_CLIENT_INTERFACE".U1_STA3_CAM_Calibrations."Calibrate jet".Outputs.Result, in2 := 0)
      wire#w1
      Contact( "DB7254_UNIT_1_STA_3_COAXIAL_ENABLE_DISABLE".ENABLED )
      wire#w2
      Coil( "DB16000_OPC_UA_TRIGGER_ALARM".CLIENT.U1_STA3_COAXIAL.ALARMS.CAM_START_JET_CALIB_METHOD_WORKING_BLOCKED_A )
   END_RUNG
   RUNG wire#powerrail
      Contact( "DB16000_OPC_UA_TRIGGER_ALARM".CLIENT.U1_STA3_COAXIAL.ALARMS.CAM_START_JET_CALIB_METHOD_WORKING_BLOCKED_A )
      I_Contact( "DB2120_MPP_ITC_IPC".RESET_FAULTS )
   END_RUNG wire#w1
   RUNG wire#w2
      Coil( "DB426_ALARMS_WARNINGS".ALARMS.UNIT_01.STATION_3_COAXIAL."716737" )
   END_RUNG
   // the same network as SCL:
   "DB16000_OPC_UA_TRIGGER_ALARM".CLIENT.U1_STA3_COAXIAL.ALARMS.CAM_START_JET_CALIB_METHOD_WORKING_BLOCKED_A := (("DB16313_U1_STA3_CAM_JET_CALIBRATE_TRIG".Done AND ("DB16002_U1_STA3_COAXIAL_CLIENT_INTERFACE".U1_STA3_CAM_Calibrations."Calibrate jet".Outputs.Result <> 0)) OR ("DB16000_OPC_UA_TRIGGER_ALARM".CLIENT.U1_STA3_COAXIAL.ALARMS.CAM_START_JET_CALIB_METHOD_WORKING_BLOCKED_A AND NOT "DB2120_MPP_ITC_IPC".RESET_FAULTS)) AND "DB7254_UNIT_1_STA_3_COAXIAL_ENABLE_DISABLE".ENABLED;
   "DB426_ALARMS_WARNINGS".ALARMS.UNIT_01.STATION_3_COAXIAL."716737" := "DB16000_OPC_UA_TRIGGER_ALARM".CLIENT.U1_STA3_COAXIAL.ALARMS.CAM_START_JET_CALIB_METHOD_WORKING_BLOCKED_A;
END_REGION

REGION Network 62: UNIT 1 STATION 3 COAXIAL CAMERA START CLADDING CALIBRATION METHOD CONNECTION ALARM
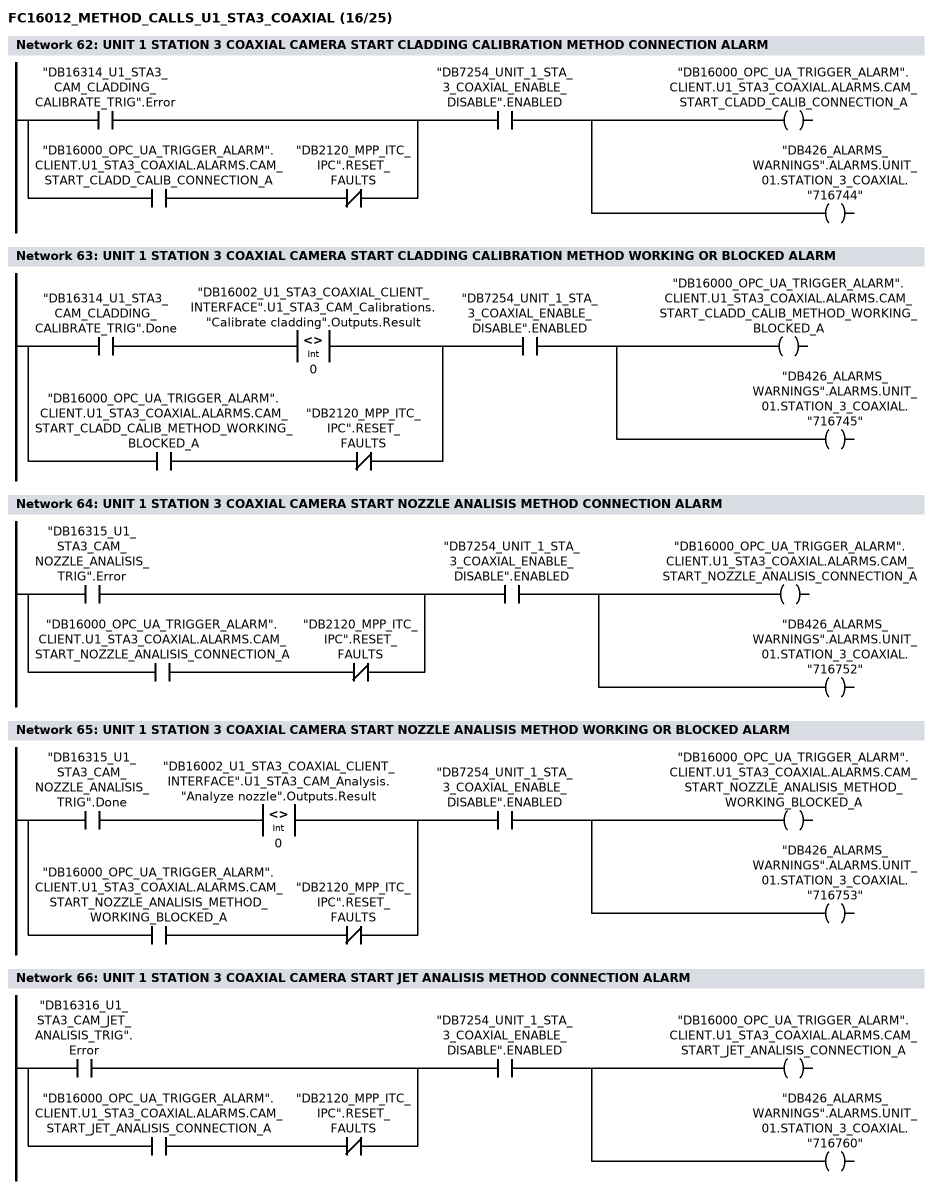
   RUNG wire#powerrail
      Contact( "DB16314_U1_STA3_CAM_CLADDING_CALIBRATE_TRIG".Error )
      wire#w1
      Contact( "DB7254_UNIT_1_STA_3_COAXIAL_ENABLE_DISABLE".ENABLED )
      wire#w2
      Coil( "DB16000_OPC_UA_TRIGGER_ALARM".CLIENT.U1_STA3_COAXIAL.ALARMS.CAM_START_CLADD_CALIB_CONNECTION_A )
   END_RUNG
   RUNG wire#powerrail
      Contact( "DB16000_OPC_UA_TRIGGER_ALARM".CLIENT.U1_STA3_COAXIAL.ALARMS.CAM_START_CLADD_CALIB_CONNECTION_A )
      I_Contact( "DB2120_MPP_ITC_IPC".RESET_FAULTS )
   END_RUNG wire#w1
   RUNG wire#w2
      Coil( "DB426_ALARMS_WARNINGS".ALARMS.UNIT_01.STATION_3_COAXIAL."716744" )
   END_RUNG
   // the same network as SCL:
   "DB16000_OPC_UA_TRIGGER_ALARM".CLIENT.U1_STA3_COAXIAL.ALARMS.CAM_START_CLADD_CALIB_CONNECTION_A := ("DB16314_U1_STA3_CAM_CLADDING_CALIBRATE_TRIG".Error OR ("DB16000_OPC_UA_TRIGGER_ALARM".CLIENT.U1_STA3_COAXIAL.ALARMS.CAM_START_CLADD_CALIB_CONNECTION_A AND NOT "DB2120_MPP_ITC_IPC".RESET_FAULTS)) AND "DB7254_UNIT_1_STA_3_COAXIAL_ENABLE_DISABLE".ENABLED;
   "DB426_ALARMS_WARNINGS".ALARMS.UNIT_01.STATION_3_COAXIAL."716744" := "DB16000_OPC_UA_TRIGGER_ALARM".CLIENT.U1_STA3_COAXIAL.ALARMS.CAM_START_CLADD_CALIB_CONNECTION_A;
END_REGION

REGION Network 63: UNIT 1 STATION 3 COAXIAL CAMERA START CLADDING CALIBRATION METHOD WORKING OR BLOCKED ALARM
   RUNG wire#powerrail
      Contact( "DB16314_U1_STA3_CAM_CLADDING_CALIBRATE_TRIG".Done )
      { S7_Templates := "SrcType := Int" } NE_Contact(in1 := "DB16002_U1_STA3_COAXIAL_CLIENT_INTERFACE".U1_STA3_CAM_Calibrations."Calibrate cladding".Outputs.Result, in2 := 0)
      wire#w1
      Contact( "DB7254_UNIT_1_STA_3_COAXIAL_ENABLE_DISABLE".ENABLED )
      wire#w2
      Coil( "DB16000_OPC_UA_TRIGGER_ALARM".CLIENT.U1_STA3_COAXIAL.ALARMS.CAM_START_CLADD_CALIB_METHOD_WORKING_BLOCKED_A )
   END_RUNG
   RUNG wire#powerrail
      Contact( "DB16000_OPC_UA_TRIGGER_ALARM".CLIENT.U1_STA3_COAXIAL.ALARMS.CAM_START_CLADD_CALIB_METHOD_WORKING_BLOCKED_A )
      I_Contact( "DB2120_MPP_ITC_IPC".RESET_FAULTS )
   END_RUNG wire#w1
   RUNG wire#w2
      Coil( "DB426_ALARMS_WARNINGS".ALARMS.UNIT_01.STATION_3_COAXIAL."716745" )
   END_RUNG
   // the same network as SCL:
   "DB16000_OPC_UA_TRIGGER_ALARM".CLIENT.U1_STA3_COAXIAL.ALARMS.CAM_START_CLADD_CALIB_METHOD_WORKING_BLOCKED_A := (("DB16314_U1_STA3_CAM_CLADDING_CALIBRATE_TRIG".Done AND ("DB16002_U1_STA3_COAXIAL_CLIENT_INTERFACE".U1_STA3_CAM_Calibrations."Calibrate cladding".Outputs.Result <> 0)) OR ("DB16000_OPC_UA_TRIGGER_ALARM".CLIENT.U1_STA3_COAXIAL.ALARMS.CAM_START_CLADD_CALIB_METHOD_WORKING_BLOCKED_A AND NOT "DB2120_MPP_ITC_IPC".RESET_FAULTS)) AND "DB7254_UNIT_1_STA_3_COAXIAL_ENABLE_DISABLE".ENABLED;
   "DB426_ALARMS_WARNINGS".ALARMS.UNIT_01.STATION_3_COAXIAL."716745" := "DB16000_OPC_UA_TRIGGER_ALARM".CLIENT.U1_STA3_COAXIAL.ALARMS.CAM_START_CLADD_CALIB_METHOD_WORKING_BLOCKED_A;
END_REGION

REGION Network 64: UNIT 1 STATION 3 COAXIAL CAMERA START NOZZLE ANALISIS METHOD CONNECTION ALARM
   RUNG wire#powerrail
      Contact( "DB16315_U1_STA3_CAM_NOZZLE_ANALISIS_TRIG".Error )
      wire#w1
      Contact( "DB7254_UNIT_1_STA_3_COAXIAL_ENABLE_DISABLE".ENABLED )
      wire#w2
      Coil( "DB16000_OPC_UA_TRIGGER_ALARM".CLIENT.U1_STA3_COAXIAL.ALARMS.CAM_START_NOZZLE_ANALISIS_CONNECTION_A )
   END_RUNG
   RUNG wire#powerrail
      Contact( "DB16000_OPC_UA_TRIGGER_ALARM".CLIENT.U1_STA3_COAXIAL.ALARMS.CAM_START_NOZZLE_ANALISIS_CONNECTION_A )
      I_Contact( "DB2120_MPP_ITC_IPC".RESET_FAULTS )
   END_RUNG wire#w1
   RUNG wire#w2
      Coil( "DB426_ALARMS_WARNINGS".ALARMS.UNIT_01.STATION_3_COAXIAL."716752" )
   END_RUNG
   // the same network as SCL:
   "DB16000_OPC_UA_TRIGGER_ALARM".CLIENT.U1_STA3_COAXIAL.ALARMS.CAM_START_NOZZLE_ANALISIS_CONNECTION_A := ("DB16315_U1_STA3_CAM_NOZZLE_ANALISIS_TRIG".Error OR ("DB16000_OPC_UA_TRIGGER_ALARM".CLIENT.U1_STA3_COAXIAL.ALARMS.CAM_START_NOZZLE_ANALISIS_CONNECTION_A AND NOT "DB2120_MPP_ITC_IPC".RESET_FAULTS)) AND "DB7254_UNIT_1_STA_3_COAXIAL_ENABLE_DISABLE".ENABLED;
   "DB426_ALARMS_WARNINGS".ALARMS.UNIT_01.STATION_3_COAXIAL."716752" := "DB16000_OPC_UA_TRIGGER_ALARM".CLIENT.U1_STA3_COAXIAL.ALARMS.CAM_START_NOZZLE_ANALISIS_CONNECTION_A;
END_REGION

REGION Network 65: UNIT 1 STATION 3 COAXIAL CAMERA START NOZZLE ANALISIS METHOD WORKING OR BLOCKED ALARM
   RUNG wire#powerrail
      Contact( "DB16315_U1_STA3_CAM_NOZZLE_ANALISIS_TRIG".Done )
      { S7_Templates := "SrcType := Int" } NE_Contact(in1 := "DB16002_U1_STA3_COAXIAL_CLIENT_INTERFACE".U1_STA3_CAM_Analysis."Analyze nozzle".Outputs.Result, in2 := 0)
      wire#w1
      Contact( "DB7254_UNIT_1_STA_3_COAXIAL_ENABLE_DISABLE".ENABLED )
      wire#w2
      Coil( "DB16000_OPC_UA_TRIGGER_ALARM".CLIENT.U1_STA3_COAXIAL.ALARMS.CAM_START_NOZZLE_ANALISIS_METHOD_WORKING_BLOCKED_A )
   END_RUNG
   RUNG wire#powerrail
      Contact( "DB16000_OPC_UA_TRIGGER_ALARM".CLIENT.U1_STA3_COAXIAL.ALARMS.CAM_START_NOZZLE_ANALISIS_METHOD_WORKING_BLOCKED_A )
      I_Contact( "DB2120_MPP_ITC_IPC".RESET_FAULTS )
   END_RUNG wire#w1
   RUNG wire#w2
      Coil( "DB426_ALARMS_WARNINGS".ALARMS.UNIT_01.STATION_3_COAXIAL."716753" )
   END_RUNG
   // the same network as SCL:
   "DB16000_OPC_UA_TRIGGER_ALARM".CLIENT.U1_STA3_COAXIAL.ALARMS.CAM_START_NOZZLE_ANALISIS_METHOD_WORKING_BLOCKED_A := (("DB16315_U1_STA3_CAM_NOZZLE_ANALISIS_TRIG".Done AND ("DB16002_U1_STA3_COAXIAL_CLIENT_INTERFACE".U1_STA3_CAM_Analysis."Analyze nozzle".Outputs.Result <> 0)) OR ("DB16000_OPC_UA_TRIGGER_ALARM".CLIENT.U1_STA3_COAXIAL.ALARMS.CAM_START_NOZZLE_ANALISIS_METHOD_WORKING_BLOCKED_A AND NOT "DB2120_MPP_ITC_IPC".RESET_FAULTS)) AND "DB7254_UNIT_1_STA_3_COAXIAL_ENABLE_DISABLE".ENABLED;
   "DB426_ALARMS_WARNINGS".ALARMS.UNIT_01.STATION_3_COAXIAL."716753" := "DB16000_OPC_UA_TRIGGER_ALARM".CLIENT.U1_STA3_COAXIAL.ALARMS.CAM_START_NOZZLE_ANALISIS_METHOD_WORKING_BLOCKED_A;
END_REGION

